// TIA Portal V19 export
FUNCTION_BLOCK "A0301_Manager_FB"   // FB45, LAD
TITLE = == A03 STATION RECIVE PRODUCT ==
// stored: MemoryReserve 100, SetENOAutomatically false
   VAR_INPUT
      AreaInterface : "AreaInterface";
      DataIn : Struct
         SemiAut_Pb : Bool;
         P1 : Struct
            Sens_Ing : Array[1..3] of Bool;
            Sens_Out : Array[1..3] of Bool;
         END_STRUCT;
         P2 : Struct
            Sens_Ing : Array[1..3] of Bool;
            Sens_Out : Array[1..3] of Bool;
         END_STRUCT;
         P3 : Struct
            Sens_Ing : Array[1..3] of Bool;
            Sens_Out : Array[1..3] of Bool;
         END_STRUCT;
         P4 : Struct
            Sens_Ing : Array[1..3] of Bool;
            Sens_Out : Array[1..3] of Bool;
         END_STRUCT;
         P5 : Struct
            Sens_Fuori_Ingombro_A0301 : Bool;
         END_STRUCT;
      END_STRUCT;
      CIn : Struct
         Trasporto : "SpeedMachine_COut";
         P1 : Struct
            Fermi : "ValveMachine_COut";
            Sfalsatore : "ValveMachine_COut";
         END_STRUCT;
         P2 : Struct
            Fermi : "ValveMachine_COut";
            Sollevatore : "ValveMachine_COut";
         END_STRUCT;
         P3 : Struct
            Fermi : "ValveMachine_COut";
         END_STRUCT;
         P4 : Struct
            Fermi : "ValveMachine_COut";
         END_STRUCT;
         P5 : Struct
            Sollevatori { ExternalAccessible := 'False'; ExternalVisible := 'False'; ExternalWritable := 'False'} : "ValveMachine_COut";
            Spintore_Lat : Struct
               Spin_Lat1 : Struct
                  Standstill : Bool;
                  Rest_CheckNext : Bool;
                  Work_CheckNext : Bool;
                  Rest : Bool;
                  Work : Bool;
               END_STRUCT;
               Spin_Lat2 : Struct
                  Standstill : Bool;
                  Rest_CheckNext : Bool;
                  Work_CheckNext : Bool;
                  Rest : Bool;
                  Work : Bool;
               END_STRUCT;
               Vrt_1 : "ValveMachine_COut";
               Orz_1 : "ValveMachine_COut";
               Vrt_2 : "ValveMachine_COut";
               Orz_2 : "ValveMachine_COut";
            END_STRUCT;
            SpintoreLong { ExternalAccessible := 'False'; ExternalVisible := 'False'; ExternalWritable := 'False'} : Struct   // Spintore Longitudinale
               Ax : "Positioning_EPOS_Machine_COut";
               Vert : "ValveMachine_COut";
            END_STRUCT;
            SensUscitaBanco : Bool;
         END_STRUCT;
         Ribaltatore : Struct
            Solleva_Rib : "ValveMachine_COut";
            Ax : "Positioning_EPOS_Machine_COut";
            Sts_Ribaltatore : Struct
               Pos0_Reached : Bool;
               Pos1_Reached : Bool;
               Pos2_Reached : Bool;
               Pos3_Reached : Bool;
            END_STRUCT;
         END_STRUCT;
         SpintoreLong : Struct
            Ax_Sts { ExternalAccessible := 'False'; ExternalVisible := 'False'; ExternalWritable := 'False'} : Struct
               PosAttesa_Reached : Bool;
               PosFineSpinta_Reached : Bool;
            END_STRUCT;
            Spin_Ev : "ValveMachine_COut";
         END_STRUCT;
         ProdManager : "Prod_Beam_Ctrl";
      END_STRUCT;
   END_VAR
   VAR_OUTPUT
      MachineInterface : "MachineInterface";
      COut : Struct
         P1 : Struct
            Fermi : "ValveMachine_Manager";
            Pareggiatore : "ValveMachine_Manager";
            ReqPTrk_A02 : Bool;   // Richiesta pezzo ad Area 02
         END_STRUCT;
         P2 : Struct
            Fermi : "ValveMachine_Manager";
            Sollevatore : "ValveMachine_Manager";
         END_STRUCT;
         P3 : Struct
            Fermi : "ValveMachine_Manager";
         END_STRUCT;
         P4 : Struct
            Fermi : "ValveMachine_Manager";
         END_STRUCT;
         P5 : Struct
            Spintore_Lat_1 { ExternalAccessible := 'False'; ExternalVisible := 'False'; ExternalWritable := 'False'} : "ValveMachine_Manager";
            Spintore_Lat_2 { ExternalAccessible := 'False'; ExternalVisible := 'False'; ExternalWritable := 'False'} : "ValveMachine_Manager";
            Sollevatori : "ValveMachine_Manager";
         END_STRUCT;
         Trasporto : "SpeedMachine_CIn_Manager";
         Trasporto_Brw_Req : Bool;
         Trasporto_Frw_Req : Bool;
         Ribaltatore : Struct
            Solleva : "ValveMachine_Manager";
            Ax : "Positioning_EPOS_Machine_Manager";
            Ax_Req : Struct
               Pos0 : Bool;
               Pos1 : Bool;
               Pos2 : Bool;
               Pos3 : Bool;
            END_STRUCT;
            Solleva_REST_Req : Bool;
            Solleva_WORK_Req : Bool;
         END_STRUCT;
      END_STRUCT;
   END_VAR
   VAR_IN_OUT
      Par : Struct
         DlySensorsON : Time;   // [ms] Ritrado ON sensori prima e dopo fermi
         DlySensorsOFF : Time;   // [ms] Ritrado OFF sensori prima e dopo fermi
         TRK : Struct
            BTrk_MoveP4Exit : Time;
            BTrk_MoveToP5 : Time;
         END_STRUCT;
      END_STRUCT;
      Data : Struct
         LastCounter_PartMove_P2toP4 : LReal;
         LastCounter_PartMove_P1toP2 : LReal;
         LastCounter_PartMove_P1toP3 : LReal;
      END_STRUCT;
   END_VAR
   VAR
      Alarm : Struct
         WrongShiftDone { S7_SetPoint := 'True'} : Bool;
         P2toP4_NotReached : Bool;
         P1toP2_NotReached : Bool;
         P1toP3_NotReached : Bool;
         PTrk_TO_BTrk : Struct
            Status : USInt;
         END_STRUCT;
         STOP_FineTurno : Bool;
         STOP_End_Of_Proroduction : Bool;
         STOP_ControlloQualita : Bool;
      END_STRUCT;
      Sts : Struct
         SemiAut : Struct
            ON : Bool;
            Request : Bool;
            MaterialFrw : Bool;
         END_STRUCT;
         P1 : Struct
            Fermi : Struct
               Sens_Ing : Bool;   // 1= Sensori attivati in base alla selezione attiva in base alla lunghezza del pezzo
               Sens_Out : Bool;   // 1= Sensori attivati in base alla selezione attiva in base alla lunghezza del pezzo
            END_STRUCT;
            Sfalsatura_OK : Bool;
         END_STRUCT;
         P2 : Struct
            Fermi : Struct
               Some_Sens_Ing : Bool;   // 1= Alcuni sensori in ingresso alla stanzione sono attivi, ma non tutti
               Sens_Ing : Bool;   // 1= Sensori attivati in base alla selezione attiva in base alla lunghezza del pezzo
               Sens_Out : Bool;   // 1= Sensori attivati in base alla selezione attiva in base alla lunghezza del pezzo
            END_STRUCT;
         END_STRUCT;
         P3 : Struct
            Fermi : Struct
               Some_Sens_Ing : Bool;   // 1= Alcuni sensori in ingresso alla stanzione sono attivi, ma non tutti
               Sens_Ing : Bool;   // 1= Sensori attivati in base alla selezione attiva in base alla lunghezza del pezzo
               Sens_Out : Bool;   // 1= Sensori attivati in base alla selezione attiva in base alla lunghezza del pezzo
            END_STRUCT;
         END_STRUCT;
         P4 : Struct
            Fermi : Struct
               Some_Sens_Ing : Bool;   // 1= Alcuni sensori in ingresso alla stanzione sono attivi, ma non tutti
               Sens_Ing : Bool;   // 1= Sensori attivati in base alla selezione attiva in base alla lunghezza del pezzo
               Sens_Out : Bool;   // 1= Sensori attivati in base alla selezione attiva in base alla lunghezza del pezzo
            END_STRUCT;
         END_STRUCT;
         A0301_Station1 : Struct
            ZoneEmpty { ExternalAccessible := 'False'; ExternalVisible := 'False'; ExternalWritable := 'False'} : Bool;
            Trk { ExternalAccessible := 'False'; ExternalVisible := 'False'; ExternalWritable := 'False'} : Struct
               Actual_O_ID : DInt;
               OLD_OID : DInt;
               A0301_PTrk_Absence : Bool;
               A0301_BTrk_Absence : Bool;
               Wait_A0301_Recive : Bool;   // Attesa ricevimento nuovo O_ID in ingresso su Pos.1 fino a che la Stazione non è vuota dal OLD_ID
            END_STRUCT;
         END_STRUCT;
         Attrezzamento : Struct
            Ready : Bool;
            FindNewID : Bool;
            RequestNewPosition : Bool;
            OLD_OID : DInt;
         END_STRUCT;
         AlarmsPresence : Bool;
         WarningsPresence : Bool;
         IsStandstill : Bool;
      END_STRUCT;
      Ctrl : Struct
         Stop : Bool;
         TRK : Struct
            PTrk : Struct
               Start_Brw : Bool;
               Start_Frw : Bool;
               Pos1_TO_Pos3 : Bool;
               Pos1_TO_Pos2 : Bool;
               Pos2Entry_TO_Pos2Solleva : Bool;
               Paregg_Pos1_to_Pos2 : Bool;
               Paregg_Pos1_to_Pos3 : Bool;
            END_STRUCT;
            BTrk : Struct
               Pos2Up_TO_Pos2Down : Bool;
               WritePos2Up_TO_Pos2Down : Bool;
               Pos4_Entry_TO_Pos4_Exit : Bool;
               Pos4_Entry_Cndz_To_Exit : Bool;
               Pos4_Exit_TO_Pos4_to_Pos5 : Bool;
               Pos4_to_Pos5_TO_Pos5_Lat_Spin_Orz : Struct
                  Exe : Bool;
                  Solleva : Bool;
                  Trasla : Bool;
               END_STRUCT;
               Pos5_SpinLat_TO_Pos5_SpinLong : Bool;
            END_STRUCT;
            Ribaltatore : Struct
               MoveToPos0 : Bool;
               MoveToPos1 : Bool;
               MoveToPos2 : Bool;
               MoveToPos3 : Bool;
            END_STRUCT;
         END_STRUCT;
         P1 : Struct
            Fermi : Struct
               Rest : Bool;
               Work : Bool;
            END_STRUCT;
            Pareggiatore : Struct
               Rest : Bool;
               Work : Bool;
            END_STRUCT;
            PartMove_P1toP3_Init : Bool;
            PartMove_P1toP2_Init : Bool;
         END_STRUCT;
         P2 : Struct
            Fermi : Struct
               Rest : Bool;
               Work : Bool;
            END_STRUCT;
            Sollevatore : Struct
               EnableMove : Bool;
               Rest : Bool;
               Work : Bool;
            END_STRUCT;
            PartMove_P2toP4_Init : Bool;
         END_STRUCT;
         P3 : Struct
            Fermi : Struct
               Rest : Bool;
               Work : Bool;
            END_STRUCT;
         END_STRUCT;
         P4 : Struct
            Fermi : Struct
               Rest : Bool;
               Work : Bool;
            END_STRUCT;
            Part_Move_P2toP4_Init : Bool;
         END_STRUCT;
         P5 : Struct
            Spintore_Lat_1 : Struct
               Rest : Bool;
               Work : Bool;
            END_STRUCT;
            Spintore_Lat_2 : Struct
               Rest : Bool;
               Work : Bool;
            END_STRUCT;
            Sollevatori : Struct
               Rest : Bool;
               Work : Bool;
            END_STRUCT;
         END_STRUCT;
         Ribaltatore : Struct
            Solleva : Struct
               EnableMove : Bool;
               Rest : Bool;
               Work : Bool;
            END_STRUCT;
         END_STRUCT;
      END_STRUCT;
      Ctrl_Part_Move_P1toP2 : "Check_Part_Movement";
      Ctrl_Part_Move_P1toP3 { S7_SetPoint := 'True'} : "Check_Part_Movement";
      Ctrl_Part_Move_P2toP4 : "Check_Part_Movement";
      TON_Stop { S7_SetPoint := 'True'} : IEC_TIMER;
      TON : Struct
         BTrk_MoveP4Exit : TON_TIME;
         BTrk_MoveToP5 : TON_TIME;
         Delay_Pos1Ribalta { S7_SetPoint := 'True'} : TON_TIME;
         P1 : Struct
            Sens_Ing : Struct
               DelayOn : TON_TIME;
            END_STRUCT;
            Sens_Out : Struct
               DelayOff : TOF_TIME;
            END_STRUCT;
         END_STRUCT;
         P2 : Struct
            Sens_Ing : Struct
               DelayOn : TON_TIME;
            END_STRUCT;
            Sens_Out : Struct
               DelayOff : TOF_TIME;
            END_STRUCT;
         END_STRUCT;
         P3 : Struct
            Sens_Ing : Struct
               DelayOn : TON_TIME;
            END_STRUCT;
            Sens_Out : Struct
               DelayOff : TOF_TIME;
            END_STRUCT;
         END_STRUCT;
         P4 : Struct
            Sens_Ing : Struct
               DelayOn : TON_TIME;
            END_STRUCT;
            Sens_Out : Struct
               DelayOff : TOF_TIME;
            END_STRUCT;
         END_STRUCT;
         P1_Exit_P3 : IEC_TIMER;
         P1_Exit_P2 : IEC_TIMER;
      END_STRUCT;
      HMI : Struct
         B_ResetShiftDone : Bool;
      END_STRUCT;
      AUX : Struct
         SemiAut_Pb : Bool;
         B_ResetShiftDone : Bool;
      END_STRUCT;
      BTrk_Item : Struct   // Appoggio dati che servolo alla Stazione dopo lettura dal MES
         O_ID : DInt;
         BLean : Real;
         W_A : Real;
         H_B : Real;
         Tol_Max : Real;
         Tol_Min : Real;
         Good { ExternalAccessible := 'False'; ExternalVisible := 'False'; ExternalWritable := 'False'} : Bool;
         Bad { ExternalAccessible := 'False'; ExternalVisible := 'False'; ExternalWritable := 'False'} : Bool;
      END_STRUCT;
      PLen_Pos1 : Real;
      PLen_Pos3 : Real;
   END_VAR
   VAR_TEMP
      i : Int;   // Indice BTrk
      j : Int;   // Indice PTrk
      SensorToUse : Struct
         P1_In : Array[1..3] of Bool;
         P1_Out : Array[1..3] of Bool;   // Sensori presenza
         P2_In : Array[1..3] of Bool;
         P2_Out : Array[1..3] of Bool;   // Fotocellule
         P3_In : Array[1..3] of Bool;
         P3_Out : Array[1..3] of Bool;   // Fotocellule
         P4_In : Array[1..3] of Bool;
         P4_Out : Array[1..3] of Bool;   // Fotocellule
      END_STRUCT;
      P1 : Struct
         Cndz1_P1toP3 : Bool;
         Cndz2_P1toP3 : Bool;
      END_STRUCT;
      Trk_GetData : Struct   // Struttura dati per lettura dal MES di tutti i dati
         indx : Int;   // Se trovato tra i TODO / ENDING / OUT questo è l'indice dove sono stati prelevati i dati
         Sts : Int;   // 0 = Non Trovato; 0 = ACT; 1 = TODO; 2=ENDING; 3 = OUT
         Item : "Prod_Item_small";
      END_STRUCT;
      Sens : Struct
         P1_IngOn : Bool;
         P1_OutOn : Bool;
         P2_IngOn : Bool;
         P3_IngOn : Bool;
         P3_OutOn : Bool;
         P4_IngOn : Bool;
         P4_OutOn : Bool;
      END_STRUCT;
   END_VAR
   VAR_TEMP   // added for the SCL form of the ladder/FBD networks
      _w1 : Bool;
      _w2 : Bool;
      _w3 : Bool;
      _w4 : Bool;
      _w5 : Bool;
      _w6 : Bool;
      _w7 : Bool;
      _w8 : Bool;
      _w9 : Bool;
      _w10 : Bool;
      _w11 : Bool;
      _w12 : Bool;
      _w13 : Bool;
      _w14 : Bool;
      _w15 : Bool;
      _w16 : Bool;
      _w17 : Bool;
      _w18 : Bool;
      _w19 : Bool;
      _w20 : Bool;
      _w21 : Bool;
      _w22 : Bool;
      _w23 : Bool;
      _w24 : Bool;
      _w25 : Bool;
   END_VAR
BEGIN

REGION Network 1: °°°°°° FORZATURA PTrk °°°°°°°°°
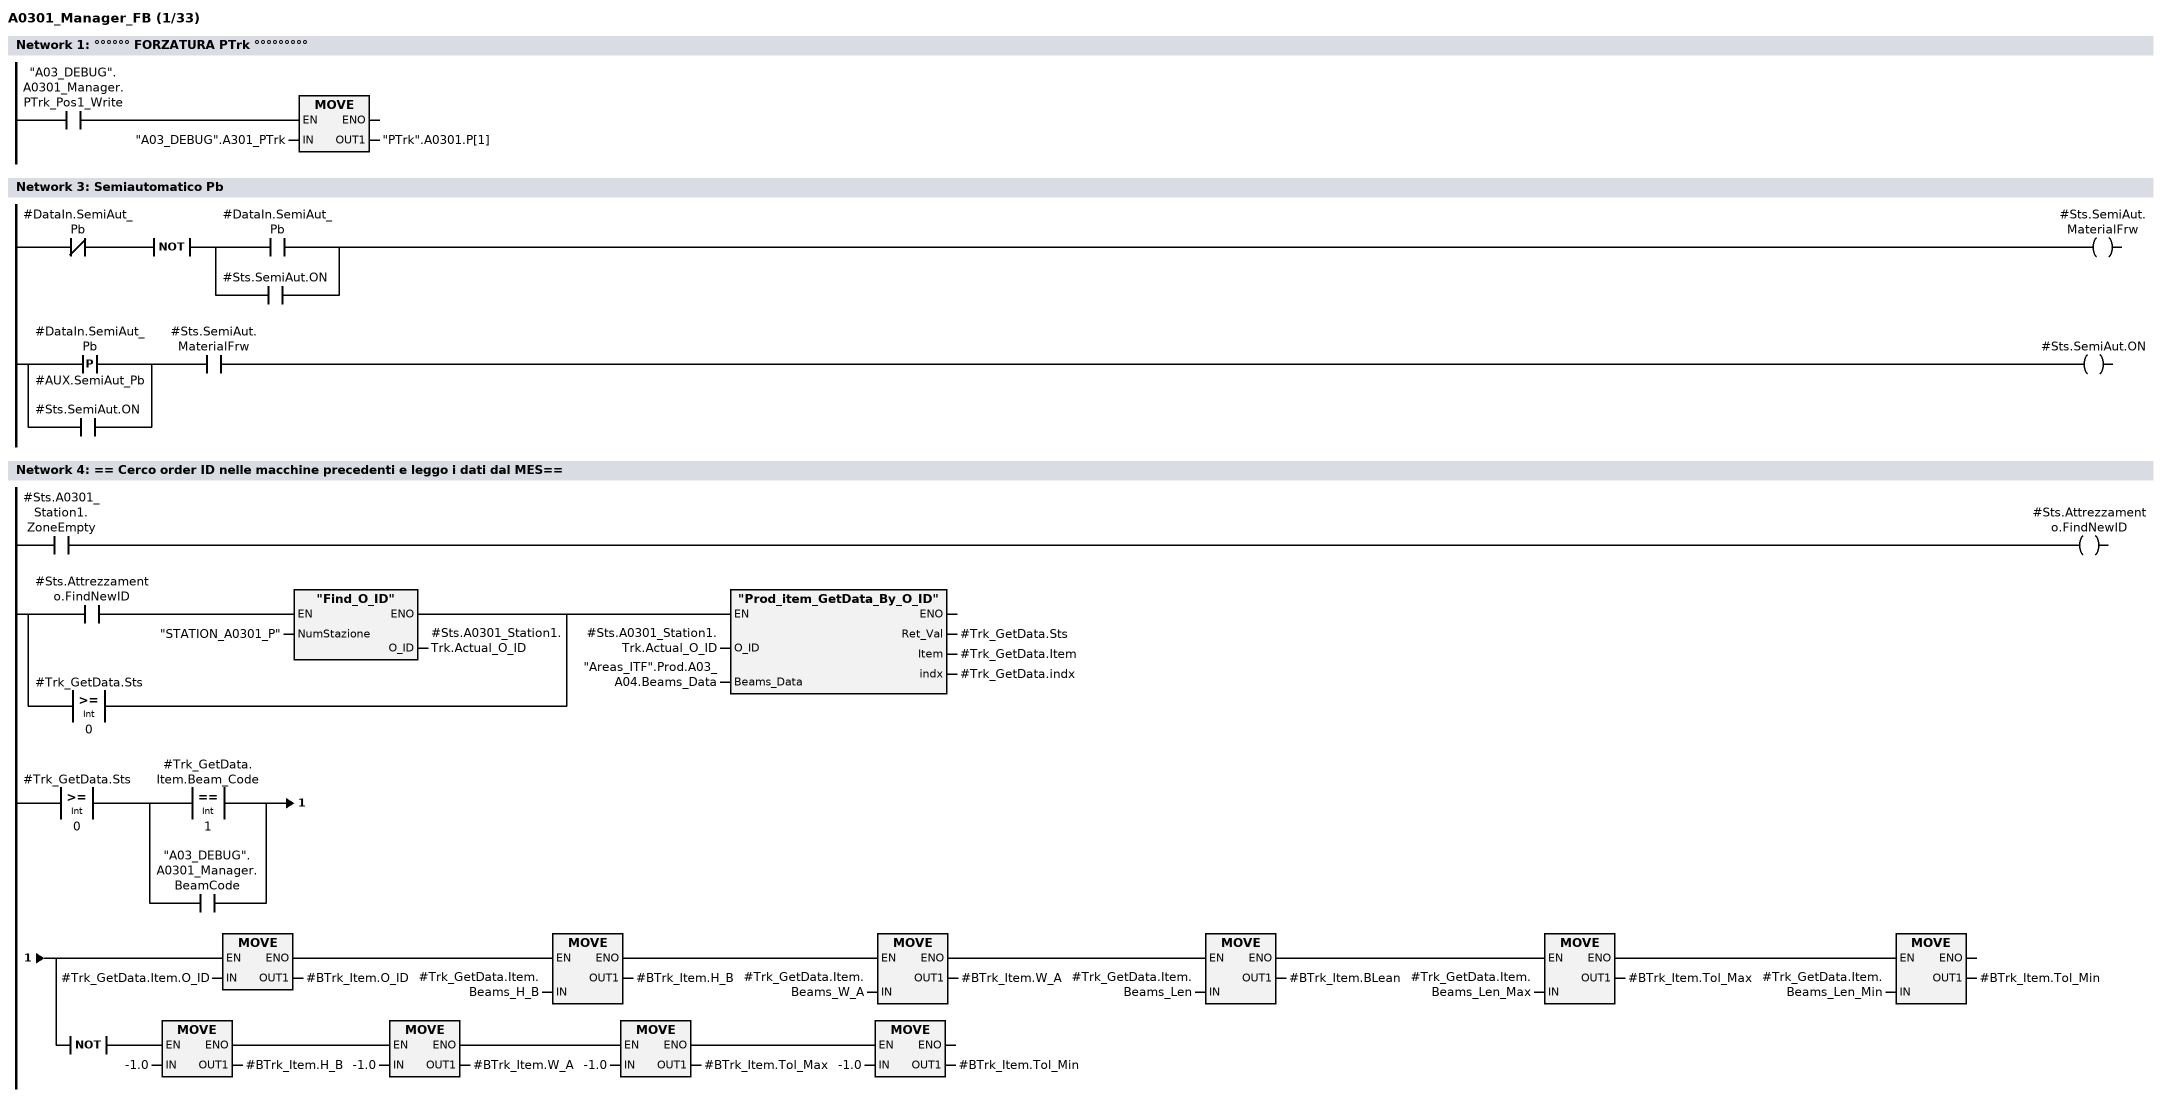
   RUNG wire#powerrail
      Contact( "A03_DEBUG".A0301_Manager.PTrk_Pos1_Write )
      Move(in := "A03_DEBUG".A301_PTrk, out1 => "PTrk".A0301.P[1])
   END_RUNG
   // the same network as SCL:
   IF "A03_DEBUG".A0301_Manager.PTrk_Pos1_Write THEN "PTrk".A0301.P[1] := "A03_DEBUG".A301_PTrk; END_IF;
END_REGION

REGION Network 2 (SCL): = Area - Rst =
   IF #AreaInterface.RstAlarms THEN
       #Alarm.WrongShiftDone := FALSE;
       #Alarm.P2toP4_NotReached:= FALSE;
       #Alarm.P1toP2_NotReached:=FALSE;
       #Alarm.P1toP3_NotReached := FALSE;
       //
       #Alarm.STOP_ControlloQualita := FALSE;
       #Alarm.STOP_FineTurno := FALSE;
       #Alarm.STOP_End_Of_Proroduction := FALSE;
   END_IF;
END_REGION

REGION Network 3: Semiautomatico Pb
   RUNG wire#powerrail
      I_Contact( #DataIn.SemiAut_Pb )
      Not()
      wire#w1
      Contact( #DataIn.SemiAut_Pb )
      wire#w2
      Coil( #Sts.SemiAut.MaterialFrw )
   END_RUNG
   RUNG wire#w1
      Contact( #Sts.SemiAut.ON )
   END_RUNG wire#w2
   RUNG wire#powerrail
      P_Contact(operand := #DataIn.SemiAut_Pb, bit := #AUX.SemiAut_Pb)
      wire#w3
      Contact( #Sts.SemiAut.MaterialFrw )
      Coil( #Sts.SemiAut.ON )
   END_RUNG
   RUNG wire#powerrail
      Contact( #Sts.SemiAut.ON )
   END_RUNG wire#w3
   // the same network as SCL:
   #Sts.SemiAut.MaterialFrw := NOT (NOT #DataIn.SemiAut_Pb) AND (#DataIn.SemiAut_Pb OR #Sts.SemiAut.ON);
   #_w1 := #DataIn.SemiAut_Pb AND NOT #AUX.SemiAut_Pb;   // rising edge of #DataIn.SemiAut_Pb
   #AUX.SemiAut_Pb := #DataIn.SemiAut_Pb;
   #Sts.SemiAut.ON := (#_w1 OR #Sts.SemiAut.ON) AND #Sts.SemiAut.MaterialFrw;
END_REGION

REGION Network 4: == Cerco order ID nelle macchine precedenti e leggo i dati dal MES==
   RUNG wire#powerrail
      Contact( #Sts.A0301_Station1.ZoneEmpty )
      Coil( #Sts.Attrezzamento.FindNewID )
   END_RUNG
   RUNG wire#powerrail
      Contact( #Sts.Attrezzamento.FindNewID )
      "Find_O_ID"(NumStazione := "STATION_A0301_P", O_ID => #Sts.A0301_Station1.Trk.Actual_O_ID)
      wire#w1
      "Prod_item_GetData_By_O_ID"(O_ID := #Sts.A0301_Station1.Trk.Actual_O_ID, Beams_Data := "Areas_ITF".Prod.A03_A04.Beams_Data, Ret_Val => #Trk_GetData.Sts, Item => #Trk_GetData.Item, indx => #Trk_GetData.indx)
   END_RUNG
   RUNG wire#powerrail
      { S7_Templates := "SrcType := Int" } GE_Contact(in1 := #Trk_GetData.Sts, in2 := 0)
   END_RUNG wire#w1
   RUNG wire#powerrail
      { S7_Templates := "SrcType := Int" } GE_Contact(in1 := #Trk_GetData.Sts, in2 := 0)
      wire#w2
      { S7_Templates := "SrcType := Int" } EQ_Contact(in1 := #Trk_GetData.Item.Beam_Code, in2 := 1)
      wire#w3
      Move(in := #Trk_GetData.Item.O_ID, out1 => #BTrk_Item.O_ID)
      Move(in := #Trk_GetData.Item.Beams_H_B, out1 => #BTrk_Item.H_B)
      Move(in := #Trk_GetData.Item.Beams_W_A, out1 => #BTrk_Item.W_A)
      Move(in := #Trk_GetData.Item.Beams_Len, out1 => #BTrk_Item.BLean)
      Move(in := #Trk_GetData.Item.Beams_Len_Max, out1 => #BTrk_Item.Tol_Max)
      Move(in := #Trk_GetData.Item.Beams_Len_Min, out1 => #BTrk_Item.Tol_Min)
   END_RUNG
   RUNG wire#w2
      Contact( "A03_DEBUG".A0301_Manager.BeamCode )
   END_RUNG wire#w3
   RUNG wire#w3
      Not()
      Move(in := -1.0, out1 => #BTrk_Item.H_B)
      Move(in := -1.0, out1 => #BTrk_Item.W_A)
      Move(in := -1.0, out1 => #BTrk_Item.Tol_Max)
      Move(in := -1.0, out1 => #BTrk_Item.Tol_Min)
   END_RUNG
   // the same network as SCL:
   #Sts.Attrezzamento.FindNewID := #Sts.A0301_Station1.ZoneEmpty;
   "Find_O_ID"(EN := #Sts.Attrezzamento.FindNewID,
               NumStazione := "STATION_A0301_P",
               O_ID => #Sts.A0301_Station1.Trk.Actual_O_ID,
               ENO => #_w1);
   IF #_w1 OR (#Trk_GetData.Sts >= 0) THEN
       #Trk_GetData.Sts := "Prod_item_GetData_By_O_ID"(O_ID := #Sts.A0301_Station1.Trk.Actual_O_ID,
                               Beams_Data := "Areas_ITF".Prod.A03_A04.Beams_Data,
                               Item => #Trk_GetData.Item,
                               indx => #Trk_GetData.indx);
   END_IF;
   #_w2 := (#Trk_GetData.Sts >= 0) AND ((#Trk_GetData.Item.Beam_Code = 1) OR "A03_DEBUG".A0301_Manager.BeamCode);
   IF #_w2 THEN
       #BTrk_Item.O_ID := #Trk_GetData.Item.O_ID;
       #BTrk_Item.H_B := #Trk_GetData.Item.Beams_H_B;
       #BTrk_Item.W_A := #Trk_GetData.Item.Beams_W_A;
       #BTrk_Item.BLean := #Trk_GetData.Item.Beams_Len;
       #BTrk_Item.Tol_Max := #Trk_GetData.Item.Beams_Len_Max;
       #BTrk_Item.Tol_Min := #Trk_GetData.Item.Beams_Len_Min;
   END_IF;
   IF NOT #_w2 THEN
       #BTrk_Item.H_B := -1.0;
       #BTrk_Item.W_A := -1.0;
       #BTrk_Item.Tol_Max := -1.0;
       #BTrk_Item.Tol_Min := -1.0;
   END_IF;
END_REGION

REGION Network 5 (SCL): == CONTROLLO TRACKING E STAZIONE PER AVANZAMENTO O_ID ==
   REGION CONTROLLO (TRK EMPTY) SU STAZIONE 1 RIBALTAMENTO A0301 
       // Controllo zona libera dai traking e sensori non in lettura su stazione A0301
       // 
       FOR #i := 1 TO "BTRK_A0301_ITEMS" DO
           IF "BTrk".A0301.B[#i].B_ID = 0 THEN
               #Sts.A0301_Station1.Trk.A0301_BTrk_Absence := TRUE;
           ELSE
               #Sts.A0301_Station1.Trk.A0301_BTrk_Absence := FALSE;
               EXIT;
           END_IF;
       END_FOR;
       //
       FOR #j := 2 TO "PTRK_A0301_ITEMS" DO
           IF "PTrk".A0301.P[#j].P_ID = 0 THEN
               #Sts.A0301_Station1.Trk.A0301_PTrk_Absence := TRUE;
           ELSE
               #Sts.A0301_Station1.Trk.A0301_PTrk_Absence := FALSE;
               EXIT;
           END_IF;
       END_FOR;

   END_REGION

   REGION CONTROLLO CHE CI SIANO LE CONDIZIONI PER MANDARE AVANTI IL NUOVO ID SU STAZIONE 1 RIBALTAMENTO A0301 (TRK EMPTY)

       // Verifica A0301 VUOTA se PTrk o BTrk assente e sensori su Stazione 1 non in lettura
       #Sts.A0301_Station1.ZoneEmpty := #Sts.A0301_Station1.Trk.A0301_PTrk_Absence AND #Sts.A0301_Station1.Trk.A0301_BTrk_Absence AND
       (NOT #Sts.P1.Fermi.Sens_Out AND
       NOT #Sts.P2.Fermi.Sens_Ing AND NOT #Sts.P1.Fermi.Sens_Out AND
       NOT #Sts.P3.Fermi.Sens_Ing AND NOT #Sts.P3.Fermi.Sens_Out AND
       NOT #Sts.P4.Fermi.Sens_Ing AND NOT #Sts.P4.Fermi.Sens_Out);


       //Se ho O_ID <> e non sono vuoto attivo avviso di attesa zona A0302 vuota
       IF (#Sts.A0301_Station1.Trk.Actual_O_ID <> #Sts.A0301_Station1.Trk.OLD_OID) OR NOT #Sts.A0301_Station1.ZoneEmpty THEN
           #Sts.A0301_Station1.Trk.Wait_A0301_Recive := TRUE;
       ELSIF (#Sts.A0301_Station1.Trk.Actual_O_ID = #Sts.A0301_Station1.Trk.OLD_OID) OR #Sts.A0301_Station1.ZoneEmpty THEN
           #Sts.A0301_Station1.Trk.Wait_A0301_Recive := FALSE;
       END_IF;

       //Se ho O_ID <> e sono vuoto aggiorno vecchio O_ID 
       IF (#Sts.A0301_Station1.Trk.Actual_O_ID <> #Sts.A0301_Station1.Trk.OLD_OID) AND #Sts.A0301_Station1.ZoneEmpty THEN
           #Sts.A0301_Station1.Trk.OLD_OID := #Sts.A0301_Station1.Trk.Actual_O_ID;
       END_IF;

   END_REGION
END_REGION

REGION Network 6 (SCL): == Compilo i dati del BTrk in base all'order ID in arrivo ==

   IF #Trk_GetData.Sts >= 0 THEN

       "BTrk".A0301.O_ID :=   #Sts.A0301_Station1.Trk.OLD_OID;
       "BTrk".A0301.Beam_Len := #BTrk_Item.BLean;
       "BTrk".A0301.Beam_W_A := #BTrk_Item.W_A;
       "BTrk".A0301.Beam_H_B := #BTrk_Item.H_B;

   ELSE
            "BTrk".A0301.O_ID := -1;
            "BTrk".A0301.Beam_Len := -1.0;
            "BTrk".A0301.Beam_W_A := -1.0;
            "BTrk".A0301.Beam_H_B := -1.0;
   END_IF;
END_REGION

REGION Network 8: <<< GESTIONE DEI SENSORI SULLE STAZIONI IN BASE ALLA LUNGHEZZA DEL PEZZO >>>
END_REGION

REGION Network 9: [P1] = Enable/Disable Sensors Pin & Controllo e Stato dei sensori ==
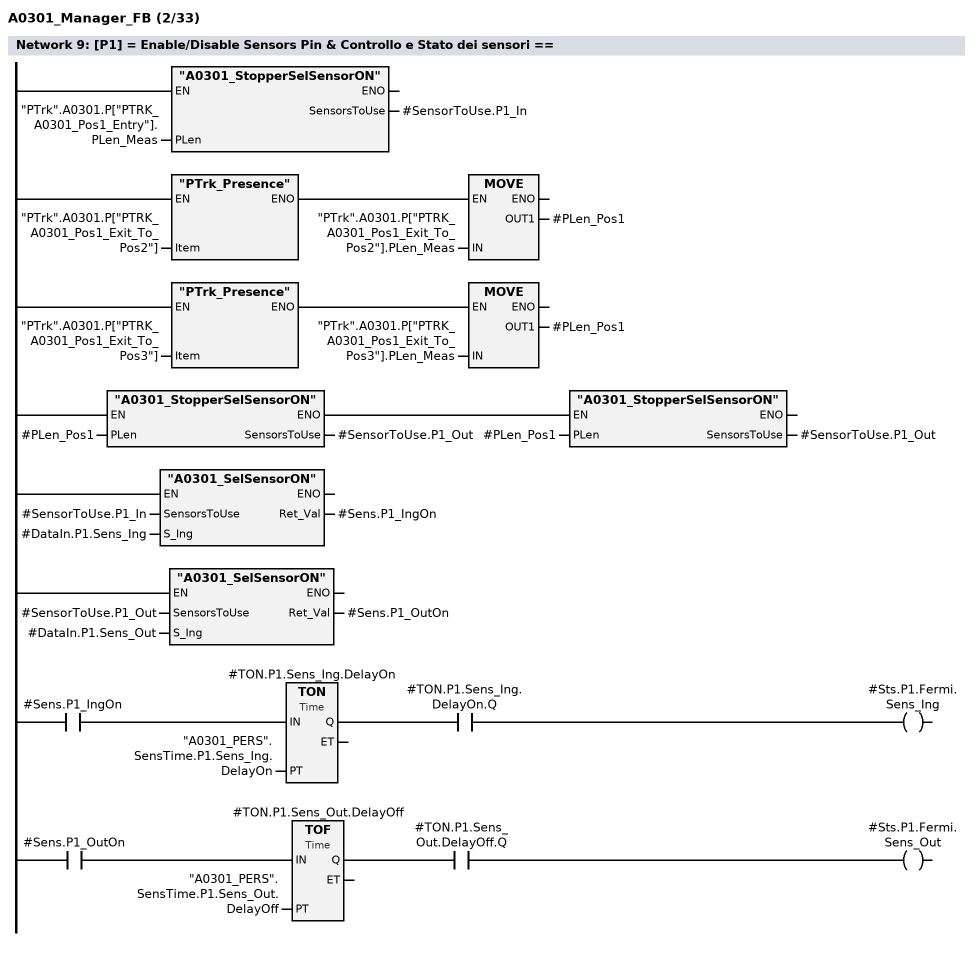
   RUNG wire#powerrail
      "A0301_StopperSelSensorON"(PLen := "PTrk".A0301.P["PTRK_A0301_Pos1_Entry"].PLen_Meas, SensorsToUse => #SensorToUse.P1_In)
   END_RUNG
   RUNG wire#powerrail
      "PTrk_Presence"(Item := "PTrk".A0301.P["PTRK_A0301_Pos1_Exit_To_Pos2"])
      Move(in := "PTrk".A0301.P["PTRK_A0301_Pos1_Exit_To_Pos2"].PLen_Meas, out1 => #PLen_Pos1)
   END_RUNG
   RUNG wire#powerrail
      "PTrk_Presence"(Item := "PTrk".A0301.P["PTRK_A0301_Pos1_Exit_To_Pos3"])
      Move(in := "PTrk".A0301.P["PTRK_A0301_Pos1_Exit_To_Pos3"].PLen_Meas, out1 => #PLen_Pos1)
   END_RUNG
   RUNG wire#powerrail
      "A0301_StopperSelSensorON"(PLen := #PLen_Pos1, SensorsToUse => #SensorToUse.P1_Out)
      "A0301_StopperSelSensorON"(PLen := #PLen_Pos1, SensorsToUse => #SensorToUse.P1_Out)
   END_RUNG
   RUNG wire#powerrail
      "A0301_SelSensorON"(SensorsToUse := #SensorToUse.P1_In, S_Ing := #DataIn.P1.Sens_Ing, Ret_Val => #Sens.P1_IngOn)
   END_RUNG
   RUNG wire#powerrail
      "A0301_SelSensorON"(SensorsToUse := #SensorToUse.P1_Out, S_Ing := #DataIn.P1.Sens_Out, Ret_Val => #Sens.P1_OutOn)
   END_RUNG
   RUNG wire#powerrail
      Contact( #Sens.P1_IngOn )
      { S7_Templates := "time_type := Time" } #TON.P1.Sens_Ing.DelayOn.TON(pt := "A0301_PERS".SensTime.P1.Sens_Ing.DelayOn, et =>)
      Contact( #TON.P1.Sens_Ing.DelayOn.Q )
      Coil( #Sts.P1.Fermi.Sens_Ing )
   END_RUNG
   RUNG wire#powerrail
      Contact( #Sens.P1_OutOn )
      { S7_Templates := "time_type := Time" } #TON.P1.Sens_Out.DelayOff.TOF(pt := "A0301_PERS".SensTime.P1.Sens_Out.DelayOff, et =>)
      Contact( #TON.P1.Sens_Out.DelayOff.Q )
      Coil( #Sts.P1.Fermi.Sens_Out )
   END_RUNG
   // the same network as SCL:
   "A0301_StopperSelSensorON"(PLen := "PTrk".A0301.P["PTRK_A0301_Pos1_Entry"].PLen_Meas,
                           SensorsToUse => #SensorToUse.P1_In);
   "PTrk_Presence"(Item := "PTrk".A0301.P["PTRK_A0301_Pos1_Exit_To_Pos2"], ENO => #_w1);
   IF #_w1 THEN #PLen_Pos1 := "PTrk".A0301.P["PTRK_A0301_Pos1_Exit_To_Pos2"].PLen_Meas; END_IF;
   "PTrk_Presence"(Item := "PTrk".A0301.P["PTRK_A0301_Pos1_Exit_To_Pos3"], ENO => #_w2);
   IF #_w2 THEN #PLen_Pos1 := "PTrk".A0301.P["PTRK_A0301_Pos1_Exit_To_Pos3"].PLen_Meas; END_IF;
   "A0301_StopperSelSensorON"(PLen := #PLen_Pos1, SensorsToUse => #SensorToUse.P1_Out, ENO => #_w3);
   IF #_w3 THEN "A0301_StopperSelSensorON"(PLen := #PLen_Pos1, SensorsToUse => #SensorToUse.P1_Out); END_IF;
   #Sens.P1_IngOn := "A0301_SelSensorON"(SensorsToUse := #SensorToUse.P1_In, S_Ing := #DataIn.P1.Sens_Ing);
   #Sens.P1_OutOn := "A0301_SelSensorON"(SensorsToUse := #SensorToUse.P1_Out, S_Ing := #DataIn.P1.Sens_Out);
   #TON.P1.Sens_Ing.DelayOn.TON(IN := #Sens.P1_IngOn, PT := "A0301_PERS".SensTime.P1.Sens_Ing.DelayOn);
   #Sts.P1.Fermi.Sens_Ing := #TON.P1.Sens_Ing.DelayOn.Q AND #TON.P1.Sens_Ing.DelayOn.Q;
   #TON.P1.Sens_Out.DelayOff.TOF(IN := #Sens.P1_OutOn, PT := "A0301_PERS".SensTime.P1.Sens_Out.DelayOff);
   #Sts.P1.Fermi.Sens_Out := #TON.P1.Sens_Out.DelayOff.Q AND #TON.P1.Sens_Out.DelayOff.Q;
END_REGION

REGION Network 10: [P2] = Enable/Disable Sensors Pin & Controllo e Stato dei sensori ==
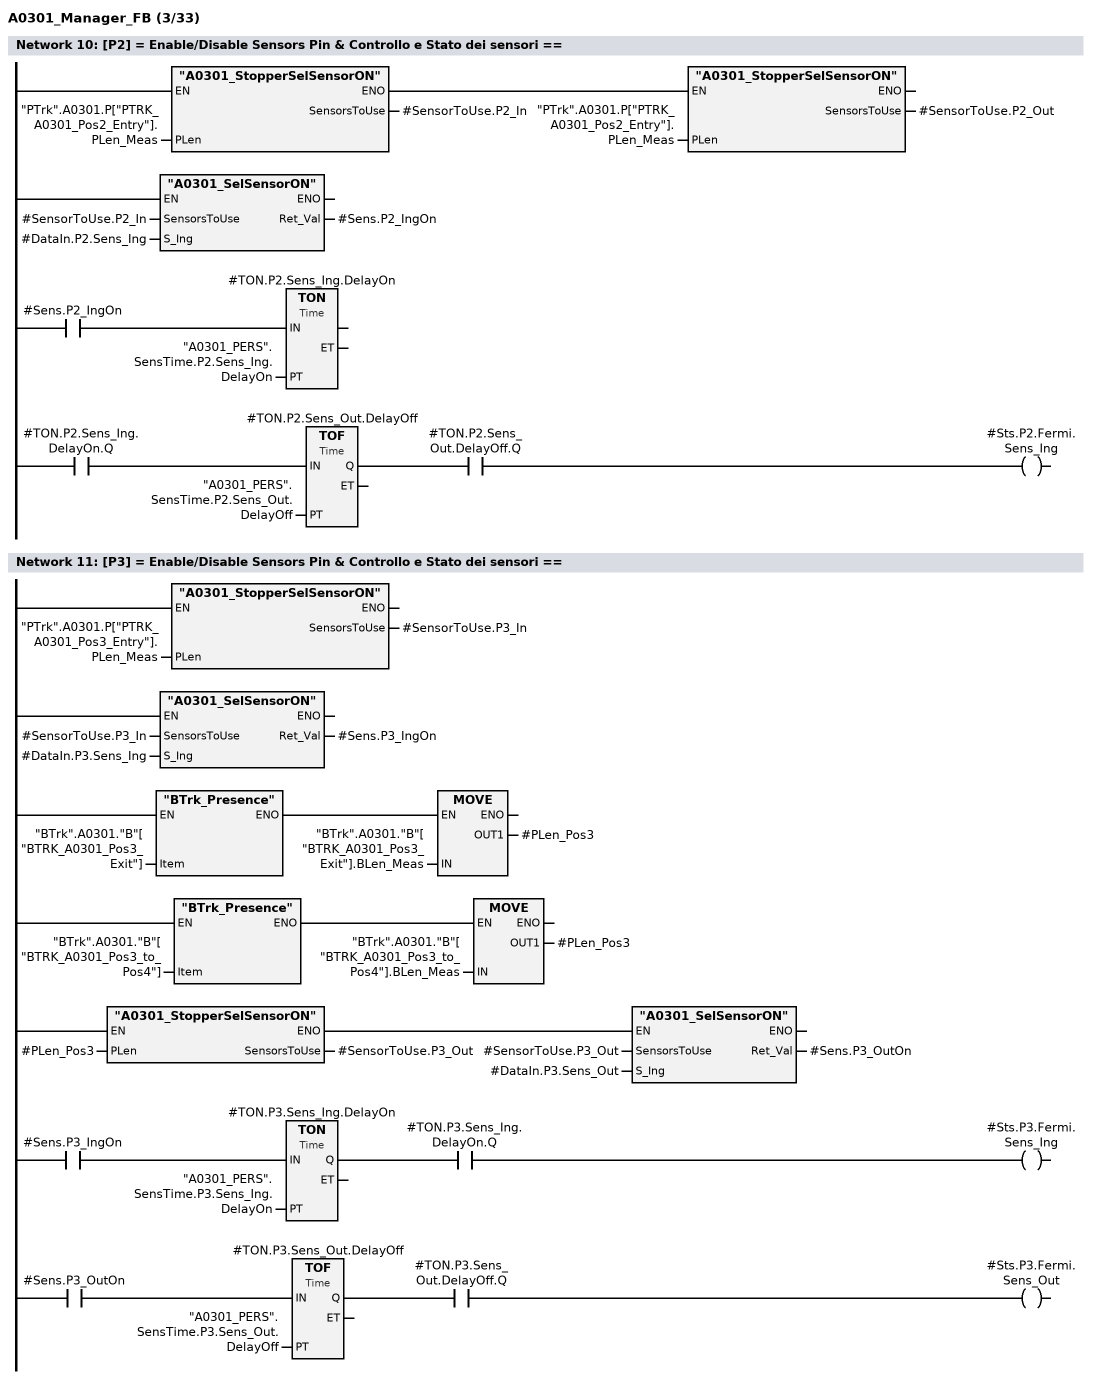
   RUNG wire#powerrail
      "A0301_StopperSelSensorON"(PLen := "PTrk".A0301.P["PTRK_A0301_Pos2_Entry"].PLen_Meas, SensorsToUse => #SensorToUse.P2_In)
      "A0301_StopperSelSensorON"(PLen := "PTrk".A0301.P["PTRK_A0301_Pos2_Entry"].PLen_Meas, SensorsToUse => #SensorToUse.P2_Out)
   END_RUNG
   RUNG wire#powerrail
      "A0301_SelSensorON"(SensorsToUse := #SensorToUse.P2_In, S_Ing := #DataIn.P2.Sens_Ing, Ret_Val => #Sens.P2_IngOn)
   END_RUNG
   RUNG wire#powerrail
      Contact( #Sens.P2_IngOn )
      { S7_Templates := "time_type := Time" } #TON.P2.Sens_Ing.DelayOn.TON(pt := "A0301_PERS".SensTime.P2.Sens_Ing.DelayOn, et =>)
   END_RUNG
   RUNG wire#powerrail
      Contact( #TON.P2.Sens_Ing.DelayOn.Q )
      { S7_Templates := "time_type := Time" } #TON.P2.Sens_Out.DelayOff.TOF(pt := "A0301_PERS".SensTime.P2.Sens_Out.DelayOff, et =>)
      Contact( #TON.P2.Sens_Out.DelayOff.Q )
      Coil( #Sts.P2.Fermi.Sens_Ing )
   END_RUNG
   // the same network as SCL:
   "A0301_StopperSelSensorON"(PLen := "PTrk".A0301.P["PTRK_A0301_Pos2_Entry"].PLen_Meas,
                           SensorsToUse => #SensorToUse.P2_In,
                           ENO => #_w1);
   IF #_w1 THEN
       "A0301_StopperSelSensorON"(PLen := "PTrk".A0301.P["PTRK_A0301_Pos2_Entry"].PLen_Meas,
                               SensorsToUse => #SensorToUse.P2_Out);
   END_IF;
   #Sens.P2_IngOn := "A0301_SelSensorON"(SensorsToUse := #SensorToUse.P2_In, S_Ing := #DataIn.P2.Sens_Ing);
   #TON.P2.Sens_Ing.DelayOn.TON(IN := #Sens.P2_IngOn, PT := "A0301_PERS".SensTime.P2.Sens_Ing.DelayOn);
   #TON.P2.Sens_Out.DelayOff.TOF(IN := #TON.P2.Sens_Ing.DelayOn.Q,
                           PT := "A0301_PERS".SensTime.P2.Sens_Out.DelayOff);
   #Sts.P2.Fermi.Sens_Ing := #TON.P2.Sens_Out.DelayOff.Q AND #TON.P2.Sens_Out.DelayOff.Q;
END_REGION

REGION Network 11: [P3] = Enable/Disable Sensors Pin & Controllo e Stato dei sensori ==
   RUNG wire#powerrail
      "A0301_StopperSelSensorON"(PLen := "PTrk".A0301.P["PTRK_A0301_Pos3_Entry"].PLen_Meas, SensorsToUse => #SensorToUse.P3_In)
   END_RUNG
   RUNG wire#powerrail
      "A0301_SelSensorON"(SensorsToUse := #SensorToUse.P3_In, S_Ing := #DataIn.P3.Sens_Ing, Ret_Val => #Sens.P3_IngOn)
   END_RUNG
   RUNG wire#powerrail
      "BTrk_Presence"(Item := "BTrk".A0301."B"["BTRK_A0301_Pos3_Exit"])
      Move(in := "BTrk".A0301."B"["BTRK_A0301_Pos3_Exit"].BLen_Meas, out1 => #PLen_Pos3)
   END_RUNG
   RUNG wire#powerrail
      "BTrk_Presence"(Item := "BTrk".A0301."B"["BTRK_A0301_Pos3_to_Pos4"])
      Move(in := "BTrk".A0301."B"["BTRK_A0301_Pos3_to_Pos4"].BLen_Meas, out1 => #PLen_Pos3)
   END_RUNG
   RUNG wire#powerrail
      "A0301_StopperSelSensorON"(PLen := #PLen_Pos3, SensorsToUse => #SensorToUse.P3_Out)
      "A0301_SelSensorON"(SensorsToUse := #SensorToUse.P3_Out, S_Ing := #DataIn.P3.Sens_Out, Ret_Val => #Sens.P3_OutOn)
   END_RUNG
   RUNG wire#powerrail
      Contact( #Sens.P3_IngOn )
      { S7_Templates := "time_type := Time" } #TON.P3.Sens_Ing.DelayOn.TON(pt := "A0301_PERS".SensTime.P3.Sens_Ing.DelayOn, et =>)
      Contact( #TON.P3.Sens_Ing.DelayOn.Q )
      Coil( #Sts.P3.Fermi.Sens_Ing )
   END_RUNG
   RUNG wire#powerrail
      Contact( #Sens.P3_OutOn )
      { S7_Templates := "time_type := Time" } #TON.P3.Sens_Out.DelayOff.TOF(pt := "A0301_PERS".SensTime.P3.Sens_Out.DelayOff, et =>)
      Contact( #TON.P3.Sens_Out.DelayOff.Q )
      Coil( #Sts.P3.Fermi.Sens_Out )
   END_RUNG
   // the same network as SCL:
   "A0301_StopperSelSensorON"(PLen := "PTrk".A0301.P["PTRK_A0301_Pos3_Entry"].PLen_Meas,
                           SensorsToUse => #SensorToUse.P3_In);
   #Sens.P3_IngOn := "A0301_SelSensorON"(SensorsToUse := #SensorToUse.P3_In, S_Ing := #DataIn.P3.Sens_Ing);
   "BTrk_Presence"(Item := "BTrk".A0301."B"["BTRK_A0301_Pos3_Exit"], ENO => #_w1);
   IF #_w1 THEN #PLen_Pos3 := "BTrk".A0301."B"["BTRK_A0301_Pos3_Exit"].BLen_Meas; END_IF;
   "BTrk_Presence"(Item := "BTrk".A0301."B"["BTRK_A0301_Pos3_to_Pos4"], ENO => #_w2);
   IF #_w2 THEN #PLen_Pos3 := "BTrk".A0301."B"["BTRK_A0301_Pos3_to_Pos4"].BLen_Meas; END_IF;
   "A0301_StopperSelSensorON"(PLen := #PLen_Pos3, SensorsToUse => #SensorToUse.P3_Out, ENO => #_w3);
   IF #_w3 THEN
       #Sens.P3_OutOn := "A0301_SelSensorON"(SensorsToUse := #SensorToUse.P3_Out, S_Ing := #DataIn.P3.Sens_Out);
   END_IF;
   #TON.P3.Sens_Ing.DelayOn.TON(IN := #Sens.P3_IngOn, PT := "A0301_PERS".SensTime.P3.Sens_Ing.DelayOn);
   #Sts.P3.Fermi.Sens_Ing := #TON.P3.Sens_Ing.DelayOn.Q AND #TON.P3.Sens_Ing.DelayOn.Q;
   #TON.P3.Sens_Out.DelayOff.TOF(IN := #Sens.P3_OutOn, PT := "A0301_PERS".SensTime.P3.Sens_Out.DelayOff);
   #Sts.P3.Fermi.Sens_Out := #TON.P3.Sens_Out.DelayOff.Q AND #TON.P3.Sens_Out.DelayOff.Q;
END_REGION

REGION Network 12: [P4] = Enable/Disable Sensors Pin & Controllo e Stato dei sensori ==
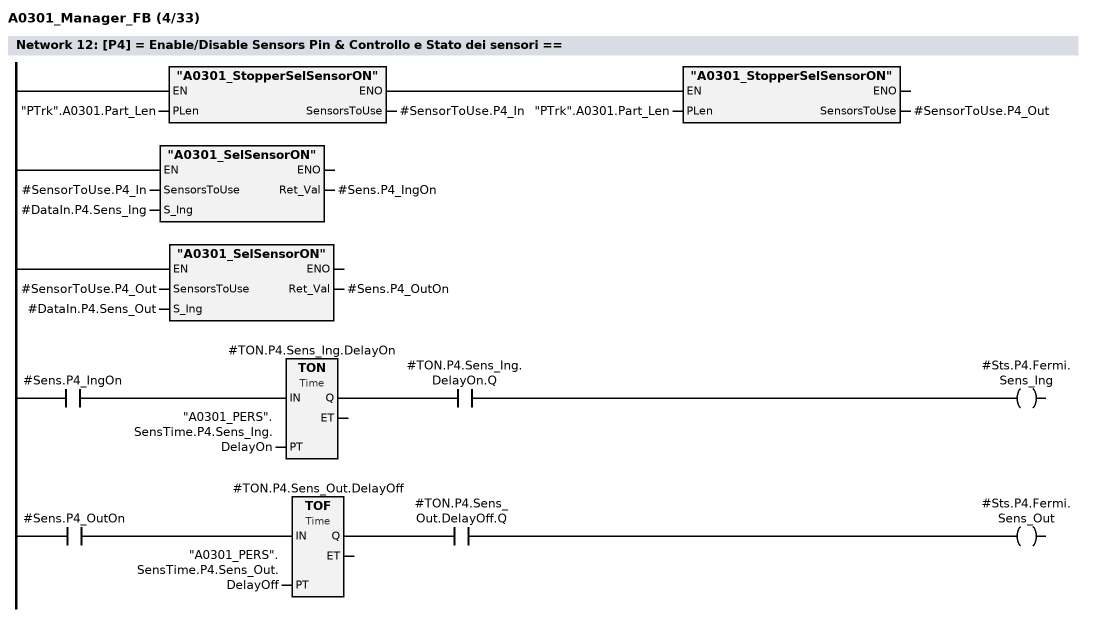
   RUNG wire#powerrail
      "A0301_StopperSelSensorON"(PLen := "PTrk".A0301.Part_Len, SensorsToUse => #SensorToUse.P4_In)
      "A0301_StopperSelSensorON"(PLen := "PTrk".A0301.Part_Len, SensorsToUse => #SensorToUse.P4_Out)
   END_RUNG
   RUNG wire#powerrail
      "A0301_SelSensorON"(SensorsToUse := #SensorToUse.P4_In, S_Ing := #DataIn.P4.Sens_Ing, Ret_Val => #Sens.P4_IngOn)
   END_RUNG
   RUNG wire#powerrail
      "A0301_SelSensorON"(SensorsToUse := #SensorToUse.P4_Out, S_Ing := #DataIn.P4.Sens_Out, Ret_Val => #Sens.P4_OutOn)
   END_RUNG
   RUNG wire#powerrail
      Contact( #Sens.P4_IngOn )
      { S7_Templates := "time_type := Time" } #TON.P4.Sens_Ing.DelayOn.TON(pt := "A0301_PERS".SensTime.P4.Sens_Ing.DelayOn, et =>)
      Contact( #TON.P4.Sens_Ing.DelayOn.Q )
      Coil( #Sts.P4.Fermi.Sens_Ing )
   END_RUNG
   RUNG wire#powerrail
      Contact( #Sens.P4_OutOn )
      { S7_Templates := "time_type := Time" } #TON.P4.Sens_Out.DelayOff.TOF(pt := "A0301_PERS".SensTime.P4.Sens_Out.DelayOff, et =>)
      Contact( #TON.P4.Sens_Out.DelayOff.Q )
      Coil( #Sts.P4.Fermi.Sens_Out )
   END_RUNG
   // the same network as SCL:
   "A0301_StopperSelSensorON"(PLen := "PTrk".A0301.Part_Len, SensorsToUse => #SensorToUse.P4_In, ENO => #_w1);
   IF #_w1 THEN
       "A0301_StopperSelSensorON"(PLen := "PTrk".A0301.Part_Len, SensorsToUse => #SensorToUse.P4_Out);
   END_IF;
   #Sens.P4_IngOn := "A0301_SelSensorON"(SensorsToUse := #SensorToUse.P4_In, S_Ing := #DataIn.P4.Sens_Ing);
   #Sens.P4_OutOn := "A0301_SelSensorON"(SensorsToUse := #SensorToUse.P4_Out, S_Ing := #DataIn.P4.Sens_Out);
   #TON.P4.Sens_Ing.DelayOn.TON(IN := #Sens.P4_IngOn, PT := "A0301_PERS".SensTime.P4.Sens_Ing.DelayOn);
   #Sts.P4.Fermi.Sens_Ing := #TON.P4.Sens_Ing.DelayOn.Q AND #TON.P4.Sens_Ing.DelayOn.Q;
   #TON.P4.Sens_Out.DelayOff.TOF(IN := #Sens.P4_OutOn, PT := "A0301_PERS".SensTime.P4.Sens_Out.DelayOff);
   #Sts.P4.Fermi.Sens_Out := #TON.P4.Sens_Out.DelayOff.Q AND #TON.P4.Sens_Out.DelayOff.Q;
END_REGION

REGION Network 14: <<<<<<<<<<<<<<< TRASPORTO >>>>>>>>>>>>>
END_REGION

REGION Network 15: [Ax] Trasporto - Controllo condizioni di START - Fwd
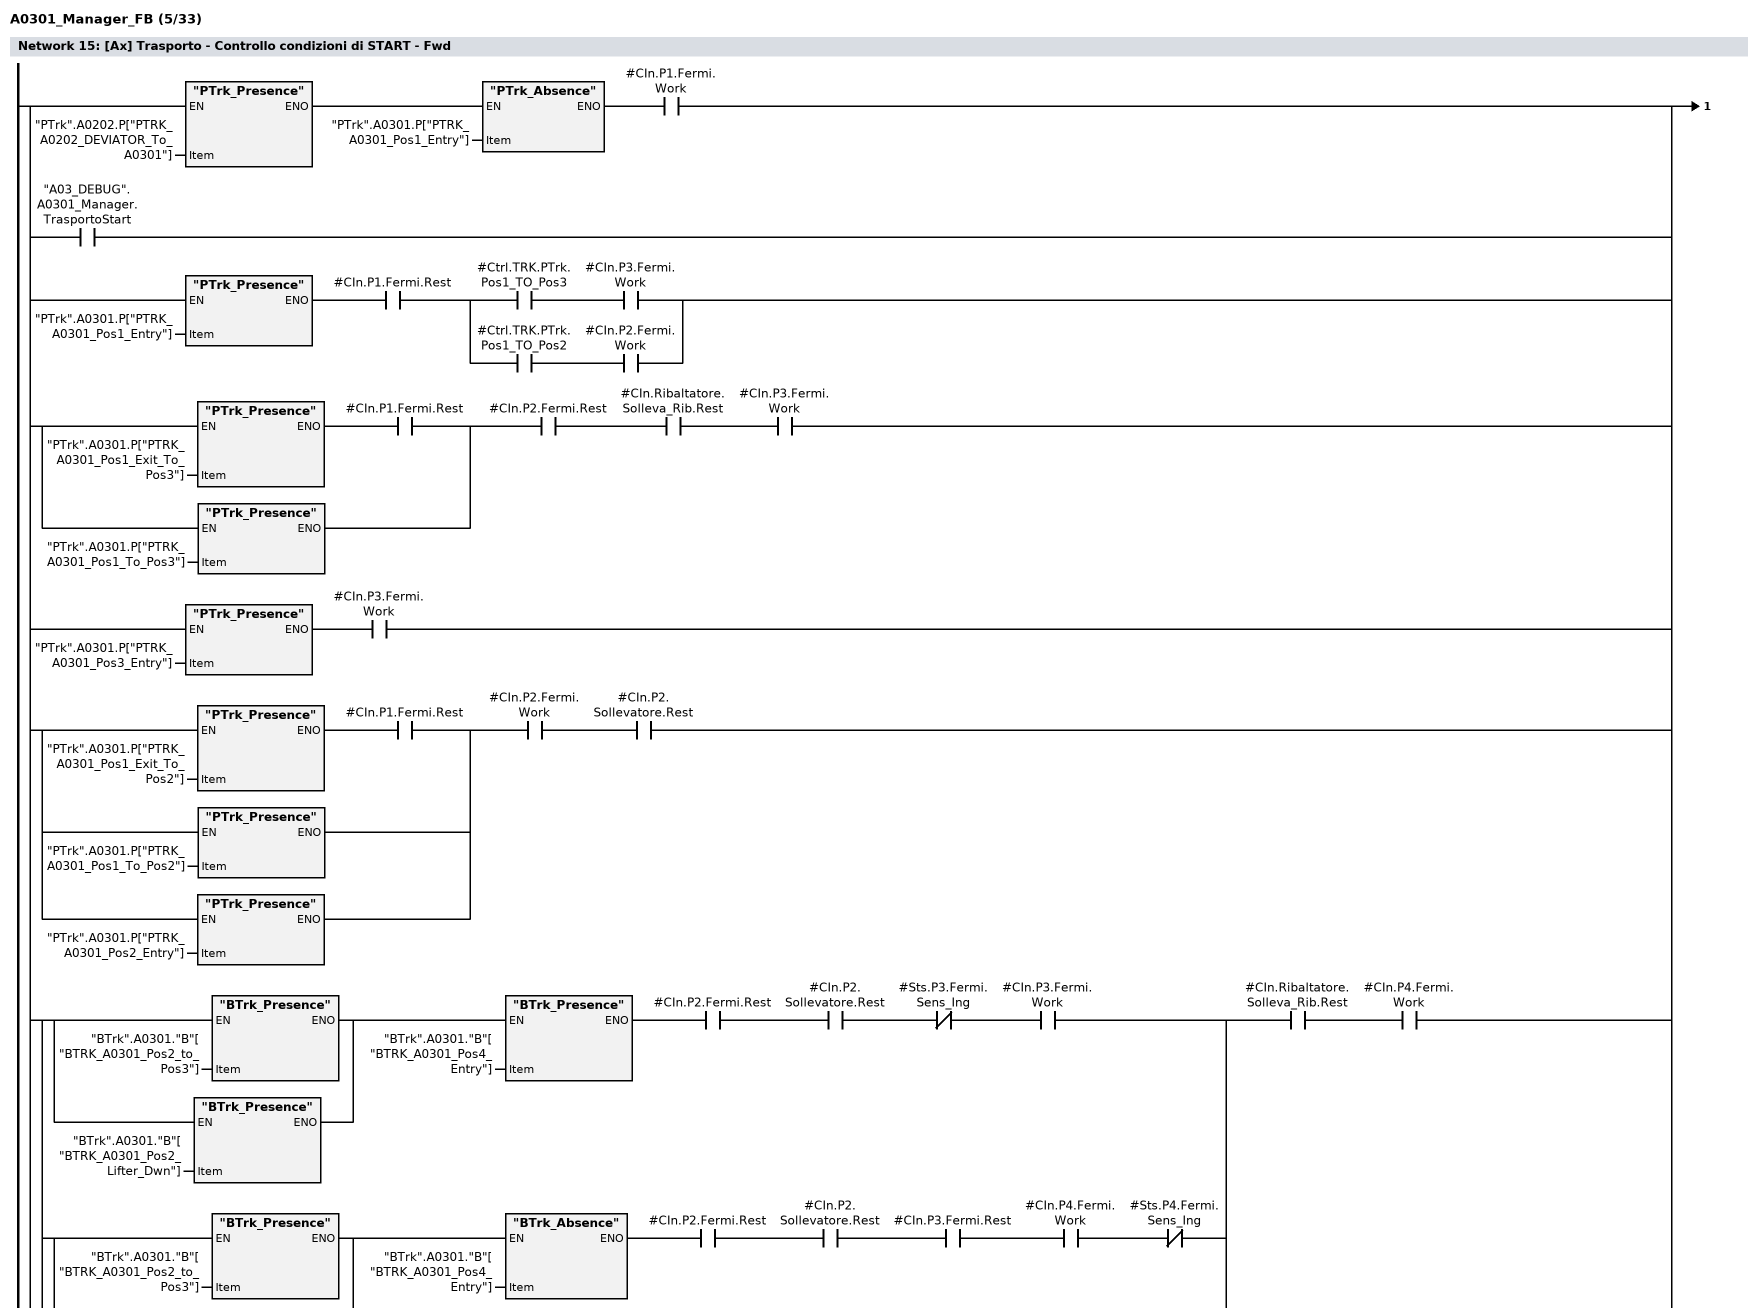
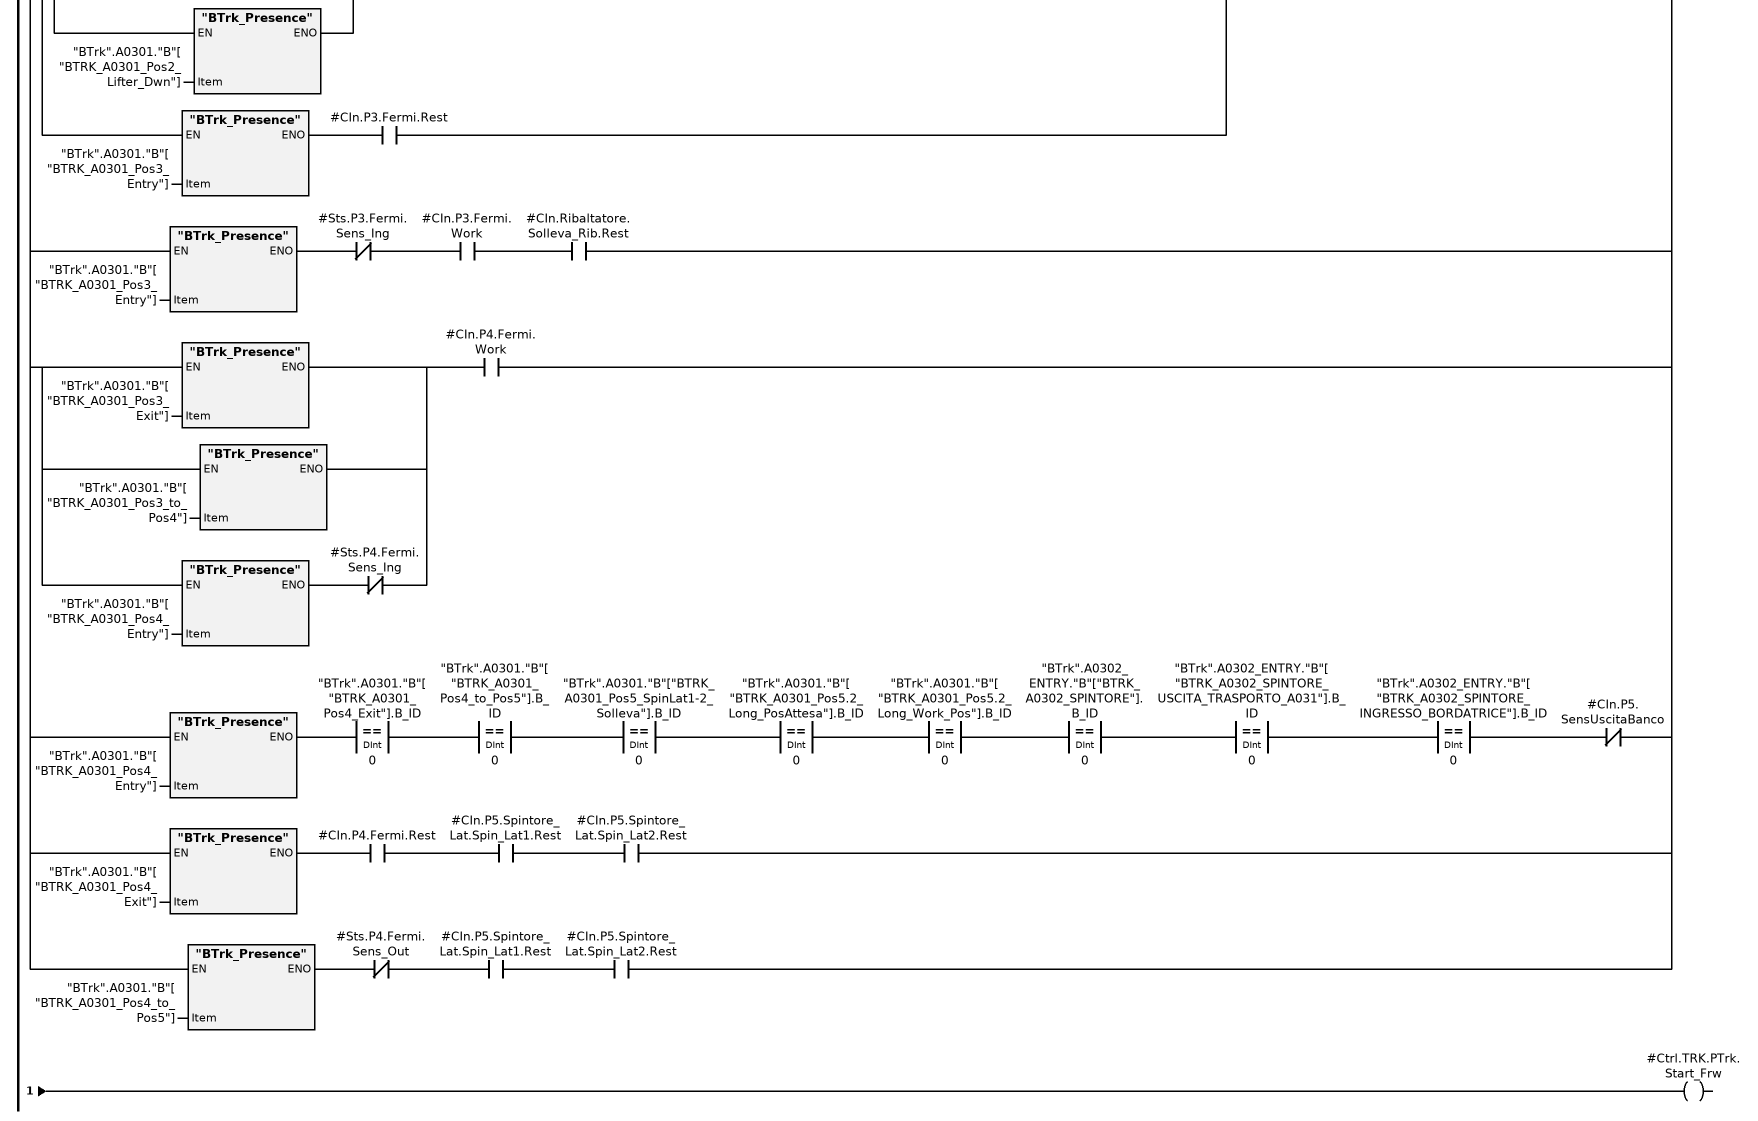
   RUNG wire#powerrail
      "PTrk_Presence"(Item := "PTrk".A0202.P["PTRK_A0202_DEVIATOR_To_A0301"])
      "PTrk_Absence"(Item := "PTrk".A0301.P["PTRK_A0301_Pos1_Entry"])
      Contact( #CIn.P1.Fermi.Work )
      wire#w1
      Coil( #Ctrl.TRK.PTrk.Start_Frw )
   END_RUNG
   RUNG wire#powerrail
      Contact( "A03_DEBUG".A0301_Manager.TrasportoStart )
   END_RUNG wire#w1
   RUNG wire#powerrail
      "PTrk_Presence"(Item := "PTrk".A0301.P["PTRK_A0301_Pos1_Entry"])
      Contact( #CIn.P1.Fermi.Rest )
      wire#w2
      Contact( #Ctrl.TRK.PTrk.Pos1_TO_Pos3 )
      Contact( #CIn.P3.Fermi.Work )
   END_RUNG wire#w1
   RUNG wire#w2
      Contact( #Ctrl.TRK.PTrk.Pos1_TO_Pos2 )
      Contact( #CIn.P2.Fermi.Work )
   END_RUNG wire#w1
   RUNG wire#powerrail
      "PTrk_Presence"(Item := "PTrk".A0301.P["PTRK_A0301_Pos1_Exit_To_Pos3"])
      Contact( #CIn.P1.Fermi.Rest )
      wire#w3
      Contact( #CIn.P2.Fermi.Rest )
      Contact( #CIn.Ribaltatore.Solleva_Rib.Rest )
      Contact( #CIn.P3.Fermi.Work )
   END_RUNG wire#w1
   RUNG wire#powerrail
      "PTrk_Presence"(Item := "PTrk".A0301.P["PTRK_A0301_Pos1_To_Pos3"])
   END_RUNG wire#w3
   RUNG wire#powerrail
      "PTrk_Presence"(Item := "PTrk".A0301.P["PTRK_A0301_Pos3_Entry"])
      Contact( #CIn.P3.Fermi.Work )
   END_RUNG wire#w1
   RUNG wire#powerrail
      "PTrk_Presence"(Item := "PTrk".A0301.P["PTRK_A0301_Pos1_Exit_To_Pos2"])
      Contact( #CIn.P1.Fermi.Rest )
      wire#w4
      Contact( #CIn.P2.Fermi.Work )
      Contact( #CIn.P2.Sollevatore.Rest )
   END_RUNG wire#w1
   RUNG wire#powerrail
      "PTrk_Presence"(Item := "PTrk".A0301.P["PTRK_A0301_Pos1_To_Pos2"])
   END_RUNG wire#w4
   RUNG wire#powerrail
      "PTrk_Presence"(Item := "PTrk".A0301.P["PTRK_A0301_Pos2_Entry"])
   END_RUNG wire#w4
   RUNG wire#powerrail
      "BTrk_Presence"(Item := "BTrk".A0301."B"["BTRK_A0301_Pos2_to_Pos3"])
      wire#w5
      "BTrk_Presence"(Item := "BTrk".A0301."B"["BTRK_A0301_Pos4_Entry"])
      Contact( #CIn.P2.Fermi.Rest )
      Contact( #CIn.P2.Sollevatore.Rest )
      I_Contact( #Sts.P3.Fermi.Sens_Ing )
      Contact( #CIn.P3.Fermi.Work )
      wire#w6
      Contact( #CIn.Ribaltatore.Solleva_Rib.Rest )
      Contact( #CIn.P4.Fermi.Work )
   END_RUNG wire#w1
   RUNG wire#powerrail
      "BTrk_Presence"(Item := "BTrk".A0301."B"["BTRK_A0301_Pos2_Lifter_Dwn"])
   END_RUNG wire#w5
   RUNG wire#powerrail
      "BTrk_Presence"(Item := "BTrk".A0301."B"["BTRK_A0301_Pos2_to_Pos3"])
      wire#w7
      "BTrk_Absence"(Item := "BTrk".A0301."B"["BTRK_A0301_Pos4_Entry"])
      Contact( #CIn.P2.Fermi.Rest )
      Contact( #CIn.P2.Sollevatore.Rest )
      Contact( #CIn.P3.Fermi.Rest )
      Contact( #CIn.P4.Fermi.Work )
      I_Contact( #Sts.P4.Fermi.Sens_Ing )
   END_RUNG wire#w6
   RUNG wire#powerrail
      "BTrk_Presence"(Item := "BTrk".A0301."B"["BTRK_A0301_Pos2_Lifter_Dwn"])
   END_RUNG wire#w7
   RUNG wire#powerrail
      "BTrk_Presence"(Item := "BTrk".A0301."B"["BTRK_A0301_Pos3_Entry"])
      Contact( #CIn.P3.Fermi.Rest )
   END_RUNG wire#w6
   RUNG wire#powerrail
      "BTrk_Presence"(Item := "BTrk".A0301."B"["BTRK_A0301_Pos3_Entry"])
      I_Contact( #Sts.P3.Fermi.Sens_Ing )
      Contact( #CIn.P3.Fermi.Work )
      Contact( #CIn.Ribaltatore.Solleva_Rib.Rest )
   END_RUNG wire#w1
   RUNG wire#powerrail
      "BTrk_Presence"(Item := "BTrk".A0301."B"["BTRK_A0301_Pos3_Exit"])
      wire#w8
      Contact( #CIn.P4.Fermi.Work )
   END_RUNG wire#w1
   RUNG wire#powerrail
      "BTrk_Presence"(Item := "BTrk".A0301."B"["BTRK_A0301_Pos3_to_Pos4"])
   END_RUNG wire#w8
   RUNG wire#powerrail
      "BTrk_Presence"(Item := "BTrk".A0301."B"["BTRK_A0301_Pos4_Entry"])
      I_Contact( #Sts.P4.Fermi.Sens_Ing )
   END_RUNG wire#w8
   RUNG wire#powerrail
      "BTrk_Presence"(Item := "BTrk".A0301."B"["BTRK_A0301_Pos4_Entry"])
      { S7_Templates := "SrcType := DInt" } EQ_Contact(in1 := "BTrk".A0301."B"["BTRK_A0301_Pos4_Exit"].B_ID, in2 := 0)
      { S7_Templates := "SrcType := DInt" } EQ_Contact(in1 := "BTrk".A0301."B"["BTRK_A0301_Pos4_to_Pos5"].B_ID, in2 := 0)
      { S7_Templates := "SrcType := DInt" } EQ_Contact(in1 := "BTrk".A0301."B"["BTRK_A0301_Pos5_SpinLat1-2_Solleva"].B_ID, in2 := 0)
      { S7_Templates := "SrcType := DInt" } EQ_Contact(in1 := "BTrk".A0301."B"["BTRK_A0301_Pos5.2_Long_PosAttesa"].B_ID, in2 := 0)
      { S7_Templates := "SrcType := DInt" } EQ_Contact(in1 := "BTrk".A0301."B"["BTRK_A0301_Pos5.2_Long_Work_Pos"].B_ID, in2 := 0)
      { S7_Templates := "SrcType := DInt" } EQ_Contact(in1 := "BTrk".A0302_ENTRY."B"["BTRK_A0302_SPINTORE"].B_ID, in2 := 0)
      { S7_Templates := "SrcType := DInt" } EQ_Contact(in1 := "BTrk".A0302_ENTRY."B"["BTRK_A0302_SPINTORE_USCITA_TRASPORTO_A031"].B_ID, in2 := 0)
      { S7_Templates := "SrcType := DInt" } EQ_Contact(in1 := "BTrk".A0302_ENTRY."B"["BTRK_A0302_SPINTORE_INGRESSO_BORDATRICE"].B_ID, in2 := 0)
      I_Contact( #CIn.P5.SensUscitaBanco )
   END_RUNG wire#w1
   RUNG wire#powerrail
      "BTrk_Presence"(Item := "BTrk".A0301."B"["BTRK_A0301_Pos4_Exit"])
      Contact( #CIn.P4.Fermi.Rest )
      Contact( #CIn.P5.Spintore_Lat.Spin_Lat1.Rest )
      Contact( #CIn.P5.Spintore_Lat.Spin_Lat2.Rest )
   END_RUNG wire#w1
   RUNG wire#powerrail
      "BTrk_Presence"(Item := "BTrk".A0301."B"["BTRK_A0301_Pos4_to_Pos5"])
      I_Contact( #Sts.P4.Fermi.Sens_Out )
      Contact( #CIn.P5.Spintore_Lat.Spin_Lat1.Rest )
      Contact( #CIn.P5.Spintore_Lat.Spin_Lat2.Rest )
   END_RUNG wire#w1
   // the same network as SCL:
   "PTrk_Presence"(Item := "PTrk".A0202.P["PTRK_A0202_DEVIATOR_To_A0301"], ENO => #_w1);
   "PTrk_Absence"(EN := #_w1, Item := "PTrk".A0301.P["PTRK_A0301_Pos1_Entry"], ENO => #_w2);
   #_w4 := "A03_DEBUG".A0301_Manager.TrasportoStart;
   "PTrk_Presence"(Item := "PTrk".A0301.P["PTRK_A0301_Pos1_Entry"], ENO => #_w3);
   "PTrk_Presence"(Item := "PTrk".A0301.P["PTRK_A0301_Pos1_Exit_To_Pos3"], ENO => #_w5);
   "PTrk_Presence"(Item := "PTrk".A0301.P["PTRK_A0301_Pos1_To_Pos3"], ENO => #_w6);
   "PTrk_Presence"(Item := "PTrk".A0301.P["PTRK_A0301_Pos3_Entry"], ENO => #_w7);
   "PTrk_Presence"(Item := "PTrk".A0301.P["PTRK_A0301_Pos1_Exit_To_Pos2"], ENO => #_w8);
   "PTrk_Presence"(Item := "PTrk".A0301.P["PTRK_A0301_Pos1_To_Pos2"], ENO => #_w9);
   "PTrk_Presence"(Item := "PTrk".A0301.P["PTRK_A0301_Pos2_Entry"], ENO => #_w10);
   "BTrk_Presence"(Item := "BTrk".A0301."B"["BTRK_A0301_Pos2_to_Pos3"], ENO => #_w11);
   "BTrk_Presence"(Item := "BTrk".A0301."B"["BTRK_A0301_Pos2_Lifter_Dwn"], ENO => #_w12);
   "BTrk_Presence"(EN := #_w11 OR #_w12, Item := "BTrk".A0301."B"["BTRK_A0301_Pos4_Entry"], ENO => #_w13);
   "BTrk_Presence"(Item := "BTrk".A0301."B"["BTRK_A0301_Pos2_to_Pos3"], ENO => #_w14);
   "BTrk_Presence"(Item := "BTrk".A0301."B"["BTRK_A0301_Pos2_Lifter_Dwn"], ENO => #_w15);
   "BTrk_Absence"(EN := #_w14 OR #_w15, Item := "BTrk".A0301."B"["BTRK_A0301_Pos4_Entry"], ENO => #_w16);
   "BTrk_Presence"(Item := "BTrk".A0301."B"["BTRK_A0301_Pos3_Entry"], ENO => #_w17);
   "BTrk_Presence"(Item := "BTrk".A0301."B"["BTRK_A0301_Pos3_Entry"], ENO => #_w18);
   "BTrk_Presence"(Item := "BTrk".A0301."B"["BTRK_A0301_Pos3_Exit"], ENO => #_w19);
   "BTrk_Presence"(Item := "BTrk".A0301."B"["BTRK_A0301_Pos3_to_Pos4"], ENO => #_w20);
   "BTrk_Presence"(Item := "BTrk".A0301."B"["BTRK_A0301_Pos4_Entry"], ENO => #_w21);
   "BTrk_Presence"(Item := "BTrk".A0301."B"["BTRK_A0301_Pos4_Entry"], ENO => #_w22);
   #_w24 := #_w22 AND ("BTrk".A0301."B"["BTRK_A0301_Pos4_Exit"].B_ID = 0) AND ("BTrk".A0301."B"["BTRK_A0301_Pos4_to_Pos5"].B_ID = 0) AND ("BTrk".A0301."B"["BTRK_A0301_Pos5_SpinLat1-2_Solleva"].B_ID = 0) AND ("BTrk".A0301."B"["BTRK_A0301_Pos5.2_Long_PosAttesa"].B_ID = 0) AND ("BTrk".A0301."B"["BTRK_A0301_Pos5.2_Long_Work_Pos"].B_ID = 0) AND ("BTrk".A0302_ENTRY."B"["BTRK_A0302_SPINTORE"].B_ID = 0) AND ("BTrk".A0302_ENTRY."B"["BTRK_A0302_SPINTORE_USCITA_TRASPORTO_A031"].B_ID = 0) AND ("BTrk".A0302_ENTRY."B"["BTRK_A0302_SPINTORE_INGRESSO_BORDATRICE"].B_ID = 0) AND NOT #CIn.P5.SensUscitaBanco;
   "BTrk_Presence"(Item := "BTrk".A0301."B"["BTRK_A0301_Pos4_Exit"], ENO => #_w23);
   "BTrk_Presence"(Item := "BTrk".A0301."B"["BTRK_A0301_Pos4_to_Pos5"], ENO => #_w25);
   #Ctrl.TRK.PTrk.Start_Frw := (#_w2 AND #CIn.P1.Fermi.Work) OR #_w4 OR (#_w3 AND #CIn.P1.Fermi.Rest AND ((#Ctrl.TRK.PTrk.Pos1_TO_Pos3 AND #CIn.P3.Fermi.Work) OR (#Ctrl.TRK.PTrk.Pos1_TO_Pos2 AND #CIn.P2.Fermi.Work))) OR (((#_w5 AND #CIn.P1.Fermi.Rest) OR #_w6) AND #CIn.P2.Fermi.Rest AND #CIn.Ribaltatore.Solleva_Rib.Rest AND #CIn.P3.Fermi.Work) OR (#_w7 AND #CIn.P3.Fermi.Work) OR (((#_w8 AND #CIn.P1.Fermi.Rest) OR #_w9 OR #_w10) AND #CIn.P2.Fermi.Work AND #CIn.P2.Sollevatore.Rest) OR (((#_w13 AND #CIn.P2.Fermi.Rest AND #CIn.P2.Sollevatore.Rest AND NOT #Sts.P3.Fermi.Sens_Ing AND #CIn.P3.Fermi.Work) OR (#_w16 AND #CIn.P2.Fermi.Rest AND #CIn.P2.Sollevatore.Rest AND #CIn.P3.Fermi.Rest AND #CIn.P4.Fermi.Work AND NOT #Sts.P4.Fermi.Sens_Ing) OR (#_w17 AND #CIn.P3.Fermi.Rest)) AND #CIn.Ribaltatore.Solleva_Rib.Rest AND #CIn.P4.Fermi.Work) OR (#_w18 AND NOT #Sts.P3.Fermi.Sens_Ing AND #CIn.P3.Fermi.Work AND #CIn.Ribaltatore.Solleva_Rib.Rest) OR ((#_w19 OR #_w20 OR (#_w21 AND NOT #Sts.P4.Fermi.Sens_Ing)) AND #CIn.P4.Fermi.Work) OR #_w24 OR (#_w23 AND #CIn.P4.Fermi.Rest AND #CIn.P5.Spintore_Lat.Spin_Lat1.Rest AND #CIn.P5.Spintore_Lat.Spin_Lat2.Rest) OR (#_w25 AND NOT #Sts.P4.Fermi.Sens_Out AND #CIn.P5.Spintore_Lat.Spin_Lat1.Rest AND #CIn.P5.Spintore_Lat.Spin_Lat2.Rest);
END_REGION

REGION Network 16: [Ax] Trasporto - COut Manager
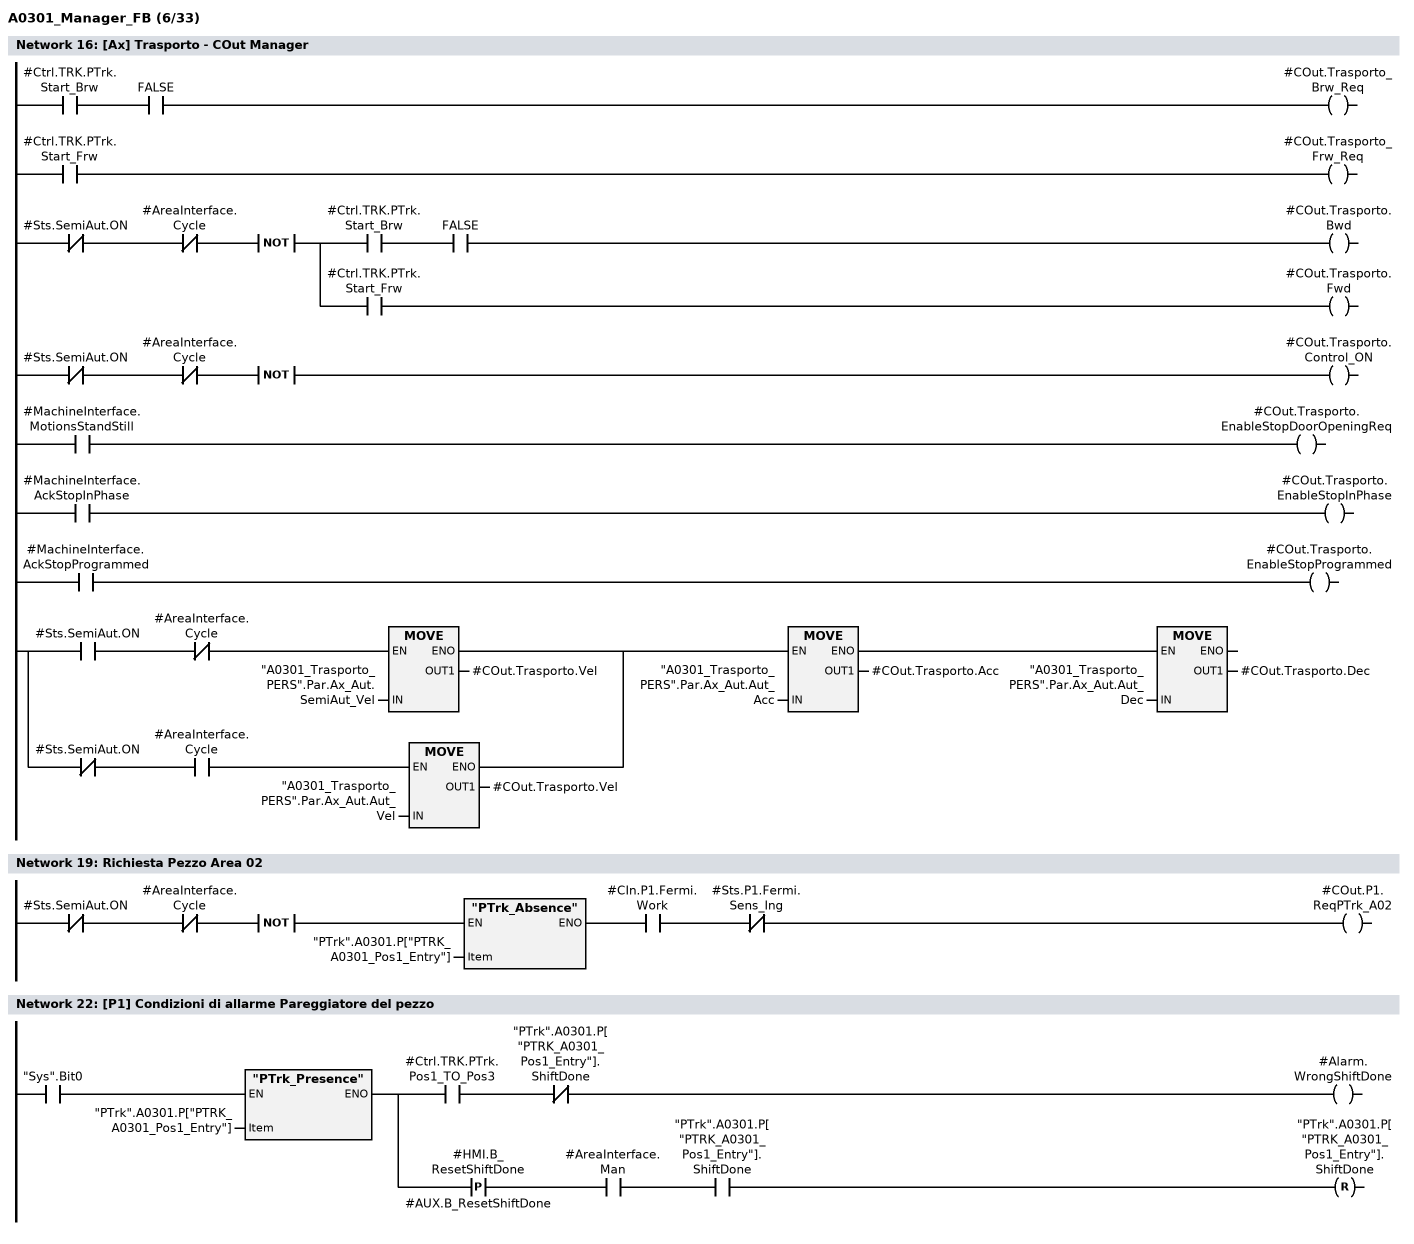
   RUNG wire#powerrail
      Contact( #Ctrl.TRK.PTrk.Start_Brw )
      Contact( FALSE )
      Coil( #COut.Trasporto_Brw_Req )
   END_RUNG
   RUNG wire#powerrail
      Contact( #Ctrl.TRK.PTrk.Start_Frw )
      Coil( #COut.Trasporto_Frw_Req )
   END_RUNG
   RUNG wire#powerrail
      I_Contact( #Sts.SemiAut.ON )
      I_Contact( #AreaInterface.Cycle )
      Not()
      wire#w1
      Contact( #Ctrl.TRK.PTrk.Start_Brw )
      Contact( FALSE )
      Coil( #COut.Trasporto.Bwd )
   END_RUNG
   RUNG wire#w1
      Contact( #Ctrl.TRK.PTrk.Start_Frw )
      Coil( #COut.Trasporto.Fwd )
   END_RUNG
   RUNG wire#powerrail
      I_Contact( #Sts.SemiAut.ON )
      I_Contact( #AreaInterface.Cycle )
      Not()
      Coil( #COut.Trasporto.Control_ON )
   END_RUNG
   RUNG wire#powerrail
      Contact( #MachineInterface.MotionsStandStill )
      Coil( #COut.Trasporto.EnableStopDoorOpeningReq )
   END_RUNG
   RUNG wire#powerrail
      Contact( #MachineInterface.AckStopInPhase )
      Coil( #COut.Trasporto.EnableStopInPhase )
   END_RUNG
   RUNG wire#powerrail
      Contact( #MachineInterface.AckStopProgrammed )
      Coil( #COut.Trasporto.EnableStopProgrammed )
   END_RUNG
   RUNG wire#powerrail
      Contact( #Sts.SemiAut.ON )
      I_Contact( #AreaInterface.Cycle )
      Move(in := "A0301_Trasporto_PERS".Par.Ax_Aut.SemiAut_Vel, out1 => #COut.Trasporto.Vel)
      wire#w2
      Move(in := "A0301_Trasporto_PERS".Par.Ax_Aut.Aut_Acc, out1 => #COut.Trasporto.Acc)
      Move(in := "A0301_Trasporto_PERS".Par.Ax_Aut.Aut_Dec, out1 => #COut.Trasporto.Dec)
   END_RUNG
   RUNG wire#powerrail
      I_Contact( #Sts.SemiAut.ON )
      Contact( #AreaInterface.Cycle )
      Move(in := "A0301_Trasporto_PERS".Par.Ax_Aut.Aut_Vel, out1 => #COut.Trasporto.Vel)
   END_RUNG wire#w2
   // the same network as SCL:
   #COut.Trasporto_Brw_Req := #Ctrl.TRK.PTrk.Start_Brw AND FALSE;
   #COut.Trasporto_Frw_Req := #Ctrl.TRK.PTrk.Start_Frw;
   #_w1 := NOT (NOT #Sts.SemiAut.ON AND NOT #AreaInterface.Cycle);
   #COut.Trasporto.Bwd := #_w1 AND #Ctrl.TRK.PTrk.Start_Brw AND FALSE;
   #COut.Trasporto.Fwd := #_w1 AND #Ctrl.TRK.PTrk.Start_Frw;
   #COut.Trasporto.Control_ON := NOT (NOT #Sts.SemiAut.ON AND NOT #AreaInterface.Cycle);
   #COut.Trasporto.EnableStopDoorOpeningReq := #MachineInterface.MotionsStandStill;
   #COut.Trasporto.EnableStopInPhase := #MachineInterface.AckStopInPhase;
   #COut.Trasporto.EnableStopProgrammed := #MachineInterface.AckStopProgrammed;
   #_w2 := #Sts.SemiAut.ON AND NOT #AreaInterface.Cycle;
   IF #_w2 THEN #COut.Trasporto.Vel := "A0301_Trasporto_PERS".Par.Ax_Aut.SemiAut_Vel; END_IF;
   #_w3 := NOT #Sts.SemiAut.ON AND #AreaInterface.Cycle;
   IF #_w3 THEN #COut.Trasporto.Vel := "A0301_Trasporto_PERS".Par.Ax_Aut.Aut_Vel; END_IF;
   IF #_w2 OR #_w3 THEN
       #COut.Trasporto.Acc := "A0301_Trasporto_PERS".Par.Ax_Aut.Aut_Acc;
       #COut.Trasporto.Dec := "A0301_Trasporto_PERS".Par.Ax_Aut.Aut_Dec;
   END_IF;
END_REGION

REGION Network 18: <<<<<<<<< MOVIMENTO TRAKING >>>>>>>>>
END_REGION

REGION Network 19: Richiesta Pezzo Area 02
   RUNG wire#powerrail
      I_Contact( #Sts.SemiAut.ON )
      I_Contact( #AreaInterface.Cycle )
      Not()
      "PTrk_Absence"(Item := "PTrk".A0301.P["PTRK_A0301_Pos1_Entry"])
      Contact( #CIn.P1.Fermi.Work )
      I_Contact( #Sts.P1.Fermi.Sens_Ing )
      Coil( #COut.P1.ReqPTrk_A02 )
   END_RUNG
   // the same network as SCL:
   "PTrk_Absence"(EN := NOT (NOT #Sts.SemiAut.ON AND NOT #AreaInterface.Cycle),
                  Item := "PTrk".A0301.P["PTRK_A0301_Pos1_Entry"],
                  ENO => #_w1);
   #COut.P1.ReqPTrk_A02 := #_w1 AND #CIn.P1.Fermi.Work AND NOT #Sts.P1.Fermi.Sens_Ing;
END_REGION

REGION Network 21: <<<<<<<<<<< POSIZIONE 1 >>>>>>>>>>>>>>
END_REGION

REGION Network 22: [P1] Condizioni di allarme Pareggiatore del pezzo
   RUNG wire#powerrail
      Contact( "Sys".Bit0 )
      "PTrk_Presence"(Item := "PTrk".A0301.P["PTRK_A0301_Pos1_Entry"])
      wire#w1
      Contact( #Ctrl.TRK.PTrk.Pos1_TO_Pos3 )
      I_Contact( "PTrk".A0301.P["PTRK_A0301_Pos1_Entry"].ShiftDone )
      Coil( #Alarm.WrongShiftDone )
   END_RUNG
   RUNG wire#w1
      P_Contact(operand := #HMI.B_ResetShiftDone, bit := #AUX.B_ResetShiftDone)
      Contact( #AreaInterface.Man )
      Contact( "PTrk".A0301.P["PTRK_A0301_Pos1_Entry"].ShiftDone )
      R_Coil( "PTrk".A0301.P["PTRK_A0301_Pos1_Entry"].ShiftDone )
   END_RUNG
   // the same network as SCL:
   "PTrk_Presence"(EN := "Sys".Bit0, Item := "PTrk".A0301.P["PTRK_A0301_Pos1_Entry"], ENO => #_w1);
   #Alarm.WrongShiftDone := #_w1 AND #Ctrl.TRK.PTrk.Pos1_TO_Pos3 AND NOT "PTrk".A0301.P["PTRK_A0301_Pos1_Entry"].ShiftDone;
   #_w2 := #_w1 AND #HMI.B_ResetShiftDone AND NOT #AUX.B_ResetShiftDone;   // rising edge of #HMI.B_ResetShiftDone
   #AUX.B_ResetShiftDone := #HMI.B_ResetShiftDone;
   IF #_w2 AND #AreaInterface.Man AND "PTrk".A0301.P["PTRK_A0301_Pos1_Entry"].ShiftDone THEN
       "PTrk".A0301.P["PTRK_A0301_Pos1_Entry"].ShiftDone := FALSE;
   END_IF;
END_REGION

REGION Network 24: << CONTROLLO RICHIESTE MOVIMENTO TRAKING PTrk >>
END_REGION

REGION Network 25: [P1] Richiesta movimento Part agli stopper P2
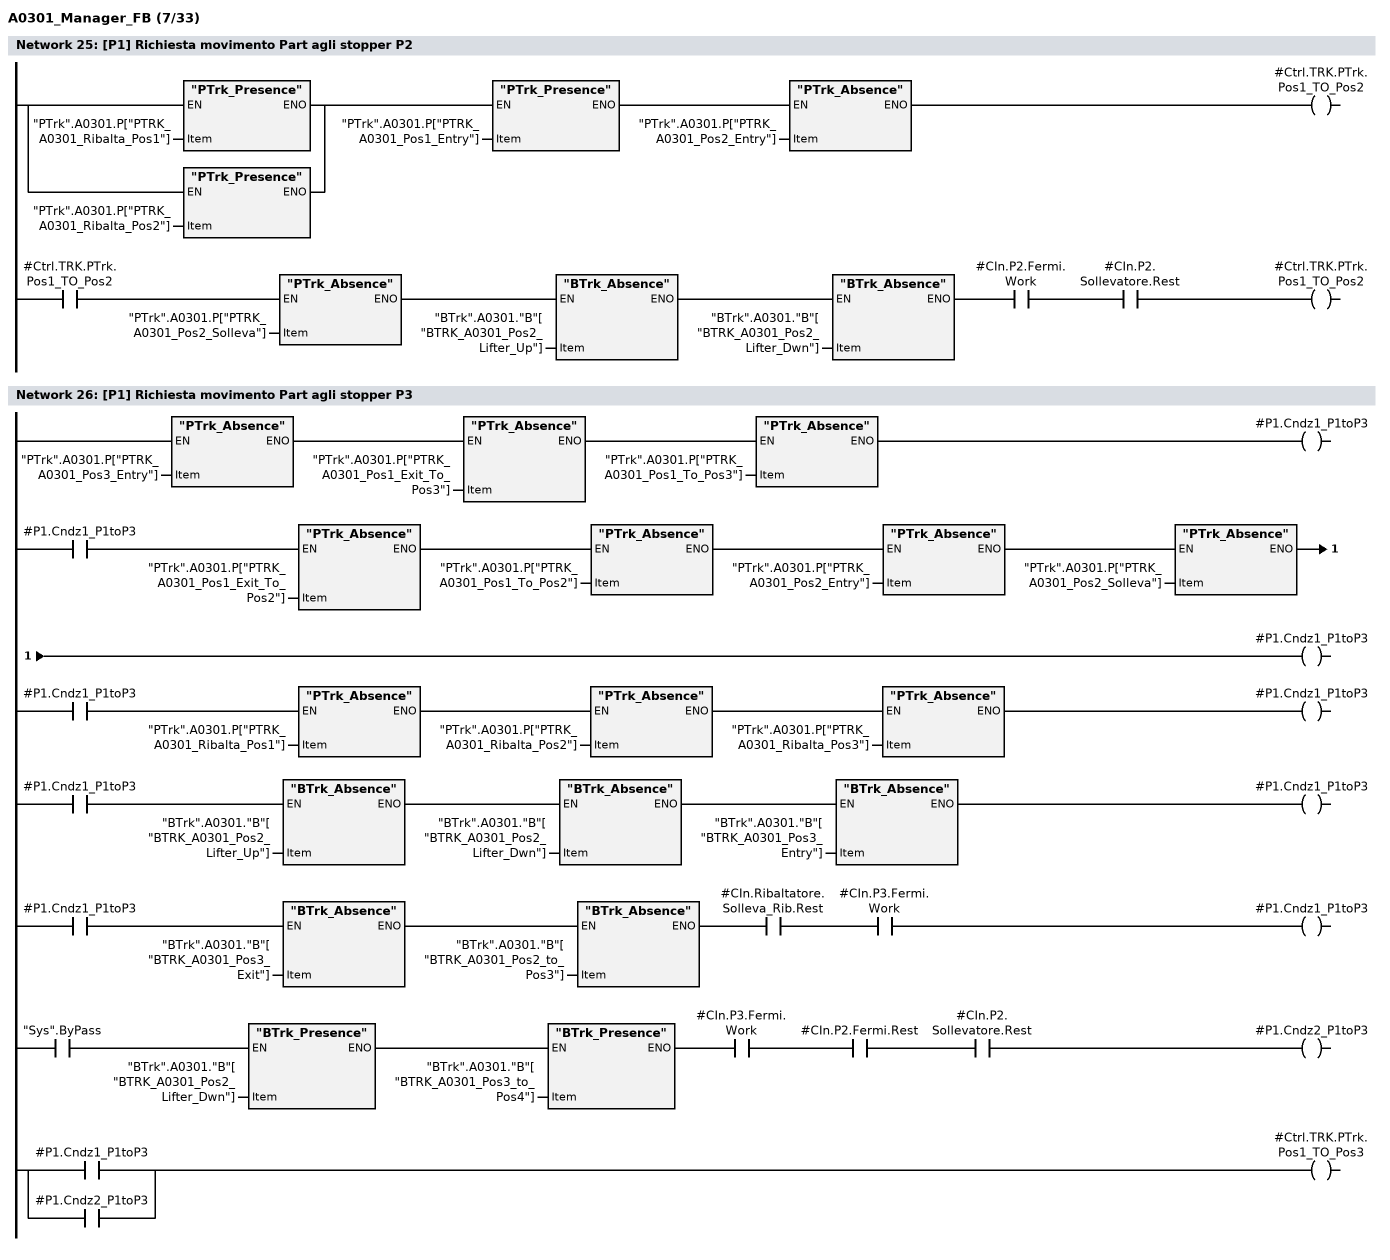
   RUNG wire#powerrail
      "PTrk_Presence"(Item := "PTrk".A0301.P["PTRK_A0301_Ribalta_Pos1"])
      wire#w1
      "PTrk_Presence"(Item := "PTrk".A0301.P["PTRK_A0301_Pos1_Entry"])
      "PTrk_Absence"(Item := "PTrk".A0301.P["PTRK_A0301_Pos2_Entry"])
      Coil( #Ctrl.TRK.PTrk.Pos1_TO_Pos2 )
   END_RUNG
   RUNG wire#powerrail
      "PTrk_Presence"(Item := "PTrk".A0301.P["PTRK_A0301_Ribalta_Pos2"])
   END_RUNG wire#w1
   RUNG wire#powerrail
      Contact( #Ctrl.TRK.PTrk.Pos1_TO_Pos2 )
      "PTrk_Absence"(Item := "PTrk".A0301.P["PTRK_A0301_Pos2_Solleva"])
      "BTrk_Absence"(Item := "BTrk".A0301."B"["BTRK_A0301_Pos2_Lifter_Up"])
      "BTrk_Absence"(Item := "BTrk".A0301."B"["BTRK_A0301_Pos2_Lifter_Dwn"])
      Contact( #CIn.P2.Fermi.Work )
      Contact( #CIn.P2.Sollevatore.Rest )
      Coil( #Ctrl.TRK.PTrk.Pos1_TO_Pos2 )
   END_RUNG
   // the same network as SCL:
   "PTrk_Presence"(Item := "PTrk".A0301.P["PTRK_A0301_Ribalta_Pos1"], ENO => #_w1);
   "PTrk_Presence"(Item := "PTrk".A0301.P["PTRK_A0301_Ribalta_Pos2"], ENO => #_w2);
   "PTrk_Presence"(EN := #_w1 OR #_w2, Item := "PTrk".A0301.P["PTRK_A0301_Pos1_Entry"], ENO => #_w3);
   "PTrk_Absence"(EN := #_w3, Item := "PTrk".A0301.P["PTRK_A0301_Pos2_Entry"], ENO => #_w4);
   #Ctrl.TRK.PTrk.Pos1_TO_Pos2 := #_w4;
   "PTrk_Absence"(EN := #Ctrl.TRK.PTrk.Pos1_TO_Pos2,
                  Item := "PTrk".A0301.P["PTRK_A0301_Pos2_Solleva"],
                  ENO => #_w5);
   "BTrk_Absence"(EN := #_w5, Item := "BTrk".A0301."B"["BTRK_A0301_Pos2_Lifter_Up"], ENO => #_w6);
   "BTrk_Absence"(EN := #_w6, Item := "BTrk".A0301."B"["BTRK_A0301_Pos2_Lifter_Dwn"], ENO => #_w7);
   #Ctrl.TRK.PTrk.Pos1_TO_Pos2 := #_w7 AND #CIn.P2.Fermi.Work AND #CIn.P2.Sollevatore.Rest;
END_REGION

REGION Network 26: [P1] Richiesta movimento Part agli stopper P3
   RUNG wire#powerrail
      "PTrk_Absence"(Item := "PTrk".A0301.P["PTRK_A0301_Pos3_Entry"])
      "PTrk_Absence"(Item := "PTrk".A0301.P["PTRK_A0301_Pos1_Exit_To_Pos3"])
      "PTrk_Absence"(Item := "PTrk".A0301.P["PTRK_A0301_Pos1_To_Pos3"])
      Coil( #P1.Cndz1_P1toP3 )
   END_RUNG
   RUNG wire#powerrail
      Contact( #P1.Cndz1_P1toP3 )
      "PTrk_Absence"(Item := "PTrk".A0301.P["PTRK_A0301_Pos1_Exit_To_Pos2"])
      "PTrk_Absence"(Item := "PTrk".A0301.P["PTRK_A0301_Pos1_To_Pos2"])
      "PTrk_Absence"(Item := "PTrk".A0301.P["PTRK_A0301_Pos2_Entry"])
      "PTrk_Absence"(Item := "PTrk".A0301.P["PTRK_A0301_Pos2_Solleva"])
      Coil( #P1.Cndz1_P1toP3 )
   END_RUNG
   RUNG wire#powerrail
      Contact( #P1.Cndz1_P1toP3 )
      "PTrk_Absence"(Item := "PTrk".A0301.P["PTRK_A0301_Ribalta_Pos1"])
      "PTrk_Absence"(Item := "PTrk".A0301.P["PTRK_A0301_Ribalta_Pos2"])
      "PTrk_Absence"(Item := "PTrk".A0301.P["PTRK_A0301_Ribalta_Pos3"])
      Coil( #P1.Cndz1_P1toP3 )
   END_RUNG
   RUNG wire#powerrail
      Contact( #P1.Cndz1_P1toP3 )
      "BTrk_Absence"(Item := "BTrk".A0301."B"["BTRK_A0301_Pos2_Lifter_Up"])
      "BTrk_Absence"(Item := "BTrk".A0301."B"["BTRK_A0301_Pos2_Lifter_Dwn"])
      "BTrk_Absence"(Item := "BTrk".A0301."B"["BTRK_A0301_Pos3_Entry"])
      Coil( #P1.Cndz1_P1toP3 )
   END_RUNG
   RUNG wire#powerrail
      Contact( #P1.Cndz1_P1toP3 )
      "BTrk_Absence"(Item := "BTrk".A0301."B"["BTRK_A0301_Pos3_Exit"])
      "BTrk_Absence"(Item := "BTrk".A0301."B"["BTRK_A0301_Pos2_to_Pos3"])
      Contact( #CIn.Ribaltatore.Solleva_Rib.Rest )
      Contact( #CIn.P3.Fermi.Work )
      Coil( #P1.Cndz1_P1toP3 )
   END_RUNG
   RUNG wire#powerrail
      Contact( "Sys".ByPass )
      "BTrk_Presence"(Item := "BTrk".A0301."B"["BTRK_A0301_Pos2_Lifter_Dwn"])
      "BTrk_Presence"(Item := "BTrk".A0301."B"["BTRK_A0301_Pos3_to_Pos4"])
      Contact( #CIn.P3.Fermi.Work )
      Contact( #CIn.P2.Fermi.Rest )
      Contact( #CIn.P2.Sollevatore.Rest )
      Coil( #P1.Cndz2_P1toP3 )
   END_RUNG
   RUNG wire#powerrail
      Contact( #P1.Cndz1_P1toP3 )
      wire#w1
      Coil( #Ctrl.TRK.PTrk.Pos1_TO_Pos3 )
   END_RUNG
   RUNG wire#powerrail
      Contact( #P1.Cndz2_P1toP3 )
   END_RUNG wire#w1
   // the same network as SCL:
   "PTrk_Absence"(Item := "PTrk".A0301.P["PTRK_A0301_Pos3_Entry"], ENO => #_w1);
   "PTrk_Absence"(EN := #_w1, Item := "PTrk".A0301.P["PTRK_A0301_Pos1_Exit_To_Pos3"], ENO => #_w2);
   "PTrk_Absence"(EN := #_w2, Item := "PTrk".A0301.P["PTRK_A0301_Pos1_To_Pos3"], ENO => #_w3);
   #P1.Cndz1_P1toP3 := #_w3;
   "PTrk_Absence"(EN := #P1.Cndz1_P1toP3, Item := "PTrk".A0301.P["PTRK_A0301_Pos1_Exit_To_Pos2"], ENO => #_w4);
   "PTrk_Absence"(EN := #_w4, Item := "PTrk".A0301.P["PTRK_A0301_Pos1_To_Pos2"], ENO => #_w5);
   "PTrk_Absence"(EN := #_w5, Item := "PTrk".A0301.P["PTRK_A0301_Pos2_Entry"], ENO => #_w6);
   "PTrk_Absence"(EN := #_w6, Item := "PTrk".A0301.P["PTRK_A0301_Pos2_Solleva"], ENO => #_w7);
   #P1.Cndz1_P1toP3 := #_w7;
   "PTrk_Absence"(EN := #P1.Cndz1_P1toP3, Item := "PTrk".A0301.P["PTRK_A0301_Ribalta_Pos1"], ENO => #_w8);
   "PTrk_Absence"(EN := #_w8, Item := "PTrk".A0301.P["PTRK_A0301_Ribalta_Pos2"], ENO => #_w9);
   "PTrk_Absence"(EN := #_w9, Item := "PTrk".A0301.P["PTRK_A0301_Ribalta_Pos3"], ENO => #_w10);
   #P1.Cndz1_P1toP3 := #_w10;
   "BTrk_Absence"(EN := #P1.Cndz1_P1toP3, Item := "BTrk".A0301."B"["BTRK_A0301_Pos2_Lifter_Up"], ENO => #_w11);
   "BTrk_Absence"(EN := #_w11, Item := "BTrk".A0301."B"["BTRK_A0301_Pos2_Lifter_Dwn"], ENO => #_w12);
   "BTrk_Absence"(EN := #_w12, Item := "BTrk".A0301."B"["BTRK_A0301_Pos3_Entry"], ENO => #_w13);
   #P1.Cndz1_P1toP3 := #_w13;
   "BTrk_Absence"(EN := #P1.Cndz1_P1toP3, Item := "BTrk".A0301."B"["BTRK_A0301_Pos3_Exit"], ENO => #_w14);
   "BTrk_Absence"(EN := #_w14, Item := "BTrk".A0301."B"["BTRK_A0301_Pos2_to_Pos3"], ENO => #_w15);
   #P1.Cndz1_P1toP3 := #_w15 AND #CIn.Ribaltatore.Solleva_Rib.Rest AND #CIn.P3.Fermi.Work;
   "BTrk_Presence"(EN := "Sys".ByPass, Item := "BTrk".A0301."B"["BTRK_A0301_Pos2_Lifter_Dwn"], ENO => #_w16);
   "BTrk_Presence"(EN := #_w16, Item := "BTrk".A0301."B"["BTRK_A0301_Pos3_to_Pos4"], ENO => #_w17);
   #P1.Cndz2_P1toP3 := #_w17 AND #CIn.P3.Fermi.Work AND #CIn.P2.Fermi.Rest AND #CIn.P2.Sollevatore.Rest;
   #Ctrl.TRK.PTrk.Pos1_TO_Pos3 := #P1.Cndz1_P1toP3 OR #P1.Cndz2_P1toP3;
END_REGION

REGION Network 28: <<<<< SPOSTAMENTO TRAKING PTrk >>>>>>
END_REGION

REGION Network 30: P[Pareggiatore] Pareggiamento su A03 Pos.1 eseguito
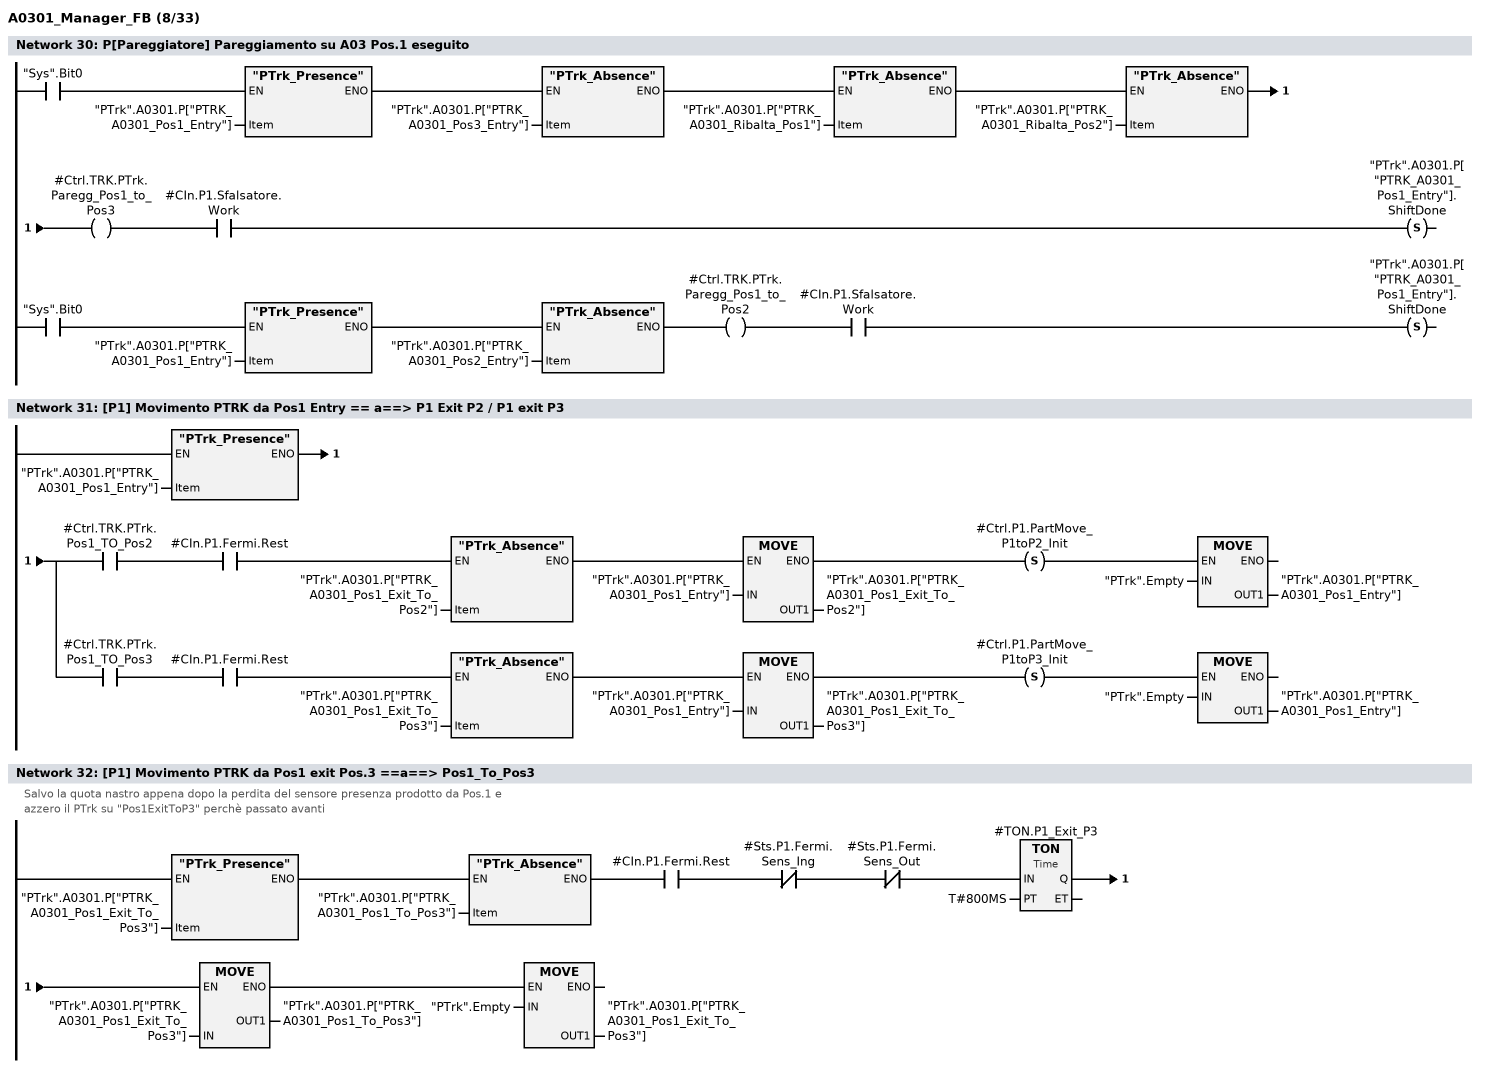
   RUNG wire#powerrail
      Contact( "Sys".Bit0 )
      "PTrk_Presence"(Item := "PTrk".A0301.P["PTRK_A0301_Pos1_Entry"])
      "PTrk_Absence"(Item := "PTrk".A0301.P["PTRK_A0301_Pos3_Entry"])
      "PTrk_Absence"(Item := "PTrk".A0301.P["PTRK_A0301_Ribalta_Pos1"])
      "PTrk_Absence"(Item := "PTrk".A0301.P["PTRK_A0301_Ribalta_Pos2"])
      Coil( #Ctrl.TRK.PTrk.Paregg_Pos1_to_Pos3 )
      Contact( #CIn.P1.Sfalsatore.Work )
      S_Coil( "PTrk".A0301.P["PTRK_A0301_Pos1_Entry"].ShiftDone )
   END_RUNG
   RUNG wire#powerrail
      Contact( "Sys".Bit0 )
      "PTrk_Presence"(Item := "PTrk".A0301.P["PTRK_A0301_Pos1_Entry"])
      "PTrk_Absence"(Item := "PTrk".A0301.P["PTRK_A0301_Pos2_Entry"])
      Coil( #Ctrl.TRK.PTrk.Paregg_Pos1_to_Pos2 )
      Contact( #CIn.P1.Sfalsatore.Work )
      S_Coil( "PTrk".A0301.P["PTRK_A0301_Pos1_Entry"].ShiftDone )
   END_RUNG
   // the same network as SCL:
   "PTrk_Presence"(EN := "Sys".Bit0, Item := "PTrk".A0301.P["PTRK_A0301_Pos1_Entry"], ENO => #_w1);
   "PTrk_Absence"(EN := #_w1, Item := "PTrk".A0301.P["PTRK_A0301_Pos3_Entry"], ENO => #_w2);
   "PTrk_Absence"(EN := #_w2, Item := "PTrk".A0301.P["PTRK_A0301_Ribalta_Pos1"], ENO => #_w3);
   "PTrk_Absence"(EN := #_w3, Item := "PTrk".A0301.P["PTRK_A0301_Ribalta_Pos2"], ENO => #_w4);
   #Ctrl.TRK.PTrk.Paregg_Pos1_to_Pos3 := #_w4;
   IF #_w4 AND #CIn.P1.Sfalsatore.Work THEN
       "PTrk".A0301.P["PTRK_A0301_Pos1_Entry"].ShiftDone := TRUE;
   END_IF;
   "PTrk_Presence"(EN := "Sys".Bit0, Item := "PTrk".A0301.P["PTRK_A0301_Pos1_Entry"], ENO => #_w5);
   "PTrk_Absence"(EN := #_w5, Item := "PTrk".A0301.P["PTRK_A0301_Pos2_Entry"], ENO => #_w6);
   #Ctrl.TRK.PTrk.Paregg_Pos1_to_Pos2 := #_w6;
   IF #_w6 AND #CIn.P1.Sfalsatore.Work THEN
       "PTrk".A0301.P["PTRK_A0301_Pos1_Entry"].ShiftDone := TRUE;
   END_IF;
END_REGION

REGION Network 31: [P1] Movimento PTRK da Pos1 Entry == a==> P1 Exit P2 / P1 exit P3
   RUNG wire#powerrail
      "PTrk_Presence"(Item := "PTrk".A0301.P["PTRK_A0301_Pos1_Entry"])
      wire#w1
      Contact( #Ctrl.TRK.PTrk.Pos1_TO_Pos2 )
      Contact( #CIn.P1.Fermi.Rest )
      "PTrk_Absence"(Item := "PTrk".A0301.P["PTRK_A0301_Pos1_Exit_To_Pos2"])
      Move(in := "PTrk".A0301.P["PTRK_A0301_Pos1_Entry"], out1 => "PTrk".A0301.P["PTRK_A0301_Pos1_Exit_To_Pos2"])
      S_Coil( #Ctrl.P1.PartMove_P1toP2_Init )
      Move(in := "PTrk".Empty, out1 => "PTrk".A0301.P["PTRK_A0301_Pos1_Entry"])
   END_RUNG
   RUNG wire#w1
      Contact( #Ctrl.TRK.PTrk.Pos1_TO_Pos3 )
      Contact( #CIn.P1.Fermi.Rest )
      "PTrk_Absence"(Item := "PTrk".A0301.P["PTRK_A0301_Pos1_Exit_To_Pos3"])
      Move(in := "PTrk".A0301.P["PTRK_A0301_Pos1_Entry"], out1 => "PTrk".A0301.P["PTRK_A0301_Pos1_Exit_To_Pos3"])
      S_Coil( #Ctrl.P1.PartMove_P1toP3_Init )
      Move(in := "PTrk".Empty, out1 => "PTrk".A0301.P["PTRK_A0301_Pos1_Entry"])
   END_RUNG
   // the same network as SCL:
   "PTrk_Presence"(Item := "PTrk".A0301.P["PTRK_A0301_Pos1_Entry"], ENO => #_w1);
   "PTrk_Absence"(EN := #_w1 AND #Ctrl.TRK.PTrk.Pos1_TO_Pos2 AND #CIn.P1.Fermi.Rest,
                  Item := "PTrk".A0301.P["PTRK_A0301_Pos1_Exit_To_Pos2"],
                  ENO => #_w2);
   IF #_w2 THEN
       "PTrk".A0301.P["PTRK_A0301_Pos1_Exit_To_Pos2"] := "PTrk".A0301.P["PTRK_A0301_Pos1_Entry"];
       #Ctrl.P1.PartMove_P1toP2_Init := TRUE;
       "PTrk".A0301.P["PTRK_A0301_Pos1_Entry"] := "PTrk".Empty;
   END_IF;
   "PTrk_Absence"(EN := #_w1 AND #Ctrl.TRK.PTrk.Pos1_TO_Pos3 AND #CIn.P1.Fermi.Rest,
                  Item := "PTrk".A0301.P["PTRK_A0301_Pos1_Exit_To_Pos3"],
                  ENO => #_w3);
   IF #_w3 THEN
       "PTrk".A0301.P["PTRK_A0301_Pos1_Exit_To_Pos3"] := "PTrk".A0301.P["PTRK_A0301_Pos1_Entry"];
       #Ctrl.P1.PartMove_P1toP3_Init := TRUE;
       "PTrk".A0301.P["PTRK_A0301_Pos1_Entry"] := "PTrk".Empty;
   END_IF;
END_REGION

REGION Network 32: [P1] Movimento PTRK da Pos1 exit Pos.3 ==a==> Pos1_To_Pos3
   // Salvo la quota nastro appena dopo la perdita del sensore presenza prodotto da Pos.1 e
   // azzero il PTrk su "Pos1ExitToP3" perchè passato avanti
   RUNG wire#powerrail
      "PTrk_Presence"(Item := "PTrk".A0301.P["PTRK_A0301_Pos1_Exit_To_Pos3"])
      "PTrk_Absence"(Item := "PTrk".A0301.P["PTRK_A0301_Pos1_To_Pos3"])
      Contact( #CIn.P1.Fermi.Rest )
      I_Contact( #Sts.P1.Fermi.Sens_Ing )
      I_Contact( #Sts.P1.Fermi.Sens_Out )
      { S7_Templates := "time_type := Time" } #TON.P1_Exit_P3.TON(pt := T#800MS, et =>)
      Move(in := "PTrk".A0301.P["PTRK_A0301_Pos1_Exit_To_Pos3"], out1 => "PTrk".A0301.P["PTRK_A0301_Pos1_To_Pos3"])
      Move(in := "PTrk".Empty, out1 => "PTrk".A0301.P["PTRK_A0301_Pos1_Exit_To_Pos3"])
   END_RUNG
   // the same network as SCL:
   "PTrk_Presence"(Item := "PTrk".A0301.P["PTRK_A0301_Pos1_Exit_To_Pos3"], ENO => #_w1);
   "PTrk_Absence"(EN := #_w1, Item := "PTrk".A0301.P["PTRK_A0301_Pos1_To_Pos3"], ENO => #_w2);
   #TON.P1_Exit_P3.TON(IN := #_w2 AND #CIn.P1.Fermi.Rest AND NOT #Sts.P1.Fermi.Sens_Ing AND NOT #Sts.P1.Fermi.Sens_Out,
                       PT := T#800MS);
   IF #TON.P1_Exit_P3.Q THEN
       "PTrk".A0301.P["PTRK_A0301_Pos1_To_Pos3"] := "PTrk".A0301.P["PTRK_A0301_Pos1_Exit_To_Pos3"];
       "PTrk".A0301.P["PTRK_A0301_Pos1_Exit_To_Pos3"] := "PTrk".Empty;
   END_IF;
END_REGION

REGION Network 33: == Monitoraggio spazio di trasporto del movimento PTrk da Pos.1 a Pos.3 ==
   // Controllo la posizione salvata da Pos.1 exit + Distanza sensori Pos.1 / Pos.3 = Target da raggiungere
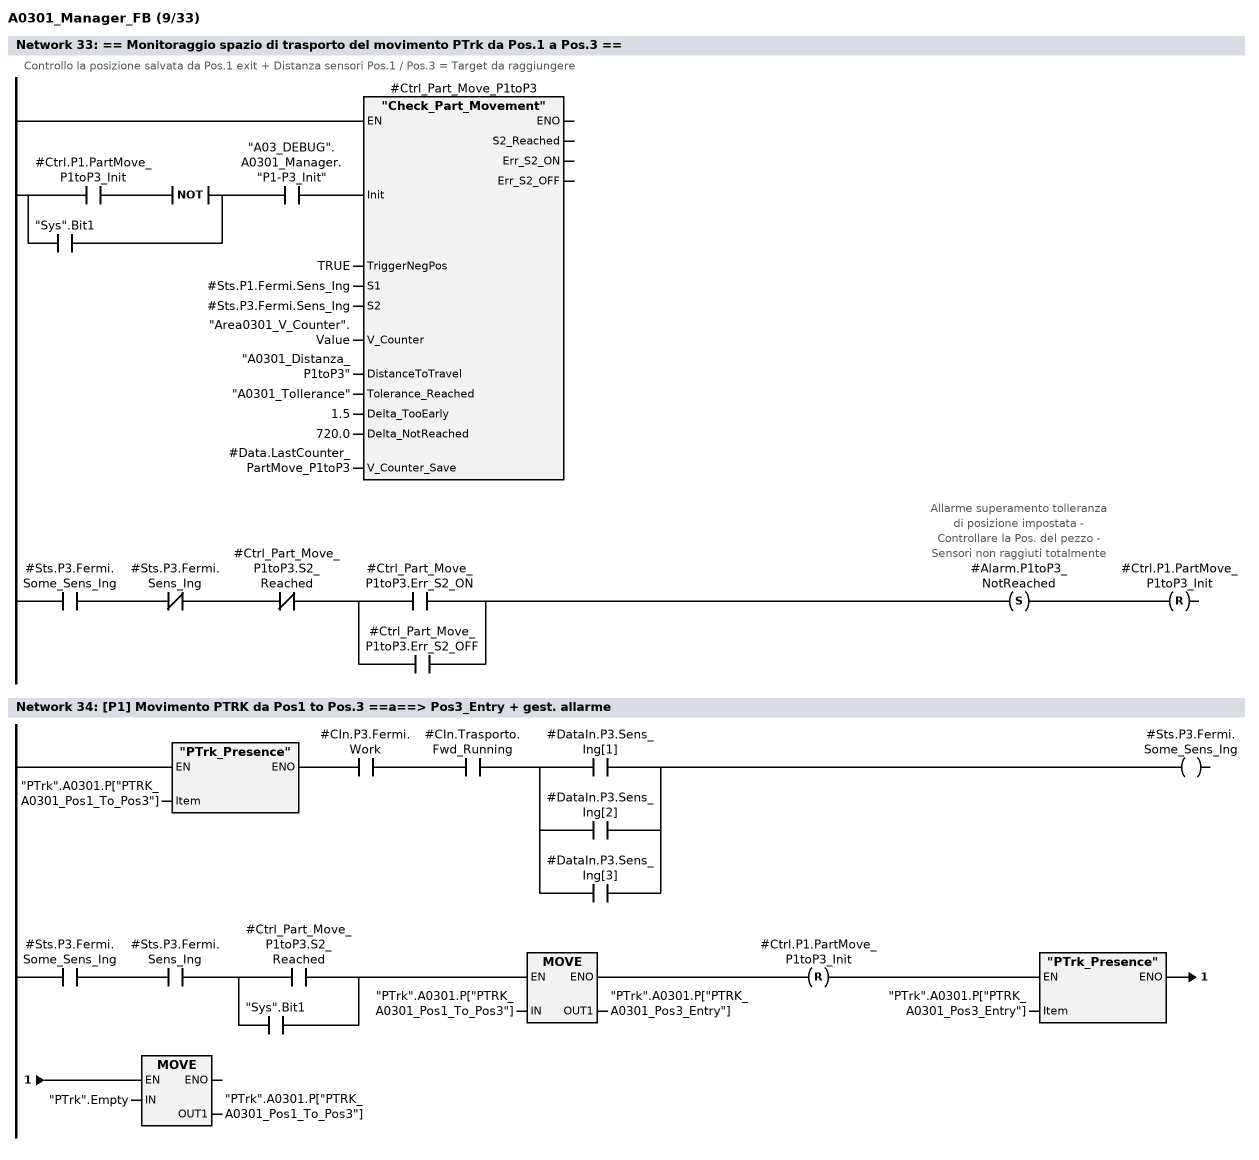
   RUNG wire#powerrail
      #Ctrl_Part_Move_P1toP3(Init := wire#w2, TriggerNegPos := TRUE, S1 := #Sts.P1.Fermi.Sens_Ing, S2 := #Sts.P3.Fermi.Sens_Ing, V_Counter := "Area0301_V_Counter".Value, DistanceToTravel := "A0301_Distanza_P1toP3", Tolerance_Reached := "A0301_Tollerance", Delta_TooEarly := 1.5, Delta_NotReached := 720.0, V_Counter_Save := #Data.LastCounter_PartMove_P1toP3, S2_Reached =>, Err_S2_ON =>, Err_S2_OFF =>)
   END_RUNG
   RUNG wire#powerrail
      Contact( #Ctrl.P1.PartMove_P1toP3_Init )
      Not()
      wire#w1
      Contact( "A03_DEBUG".A0301_Manager."P1-P3_Init" )
   END_RUNG wire#w2
   RUNG wire#powerrail
      Contact( "Sys".Bit1 )
   END_RUNG wire#w1
   RUNG wire#powerrail
      Contact( #Sts.P3.Fermi.Some_Sens_Ing )
      I_Contact( #Sts.P3.Fermi.Sens_Ing )
      I_Contact( #Ctrl_Part_Move_P1toP3.S2_Reached )
      wire#w3
      Contact( #Ctrl_Part_Move_P1toP3.Err_S2_ON )
      wire#w4
      S_Coil( #Alarm.P1toP3_NotReached )   // Allarme superamento tolleranza di posizione impostata - Controllare la Pos. del pezzo - Sensori non raggiuti totalmente
      R_Coil( #Ctrl.P1.PartMove_P1toP3_Init )
   END_RUNG
   RUNG wire#w3
      Contact( #Ctrl_Part_Move_P1toP3.Err_S2_OFF )
   END_RUNG wire#w4
   // the same network as SCL:
   #Ctrl_Part_Move_P1toP3(Init := (NOT #Ctrl.P1.PartMove_P1toP3_Init OR "Sys".Bit1) AND "A03_DEBUG".A0301_Manager."P1-P3_Init",   // "Check_Part_Movement"
                          TriggerNegPos := TRUE,
                          S1 := #Sts.P1.Fermi.Sens_Ing,
                          S2 := #Sts.P3.Fermi.Sens_Ing,
                          V_Counter := "Area0301_V_Counter".Value,
                          DistanceToTravel := "A0301_Distanza_P1toP3",
                          Tolerance_Reached := "A0301_Tollerance",
                          Delta_TooEarly := 1.5,
                          Delta_NotReached := 720.0,
                          V_Counter_Save := #Data.LastCounter_PartMove_P1toP3);
   IF #Sts.P3.Fermi.Some_Sens_Ing AND NOT #Sts.P3.Fermi.Sens_Ing AND NOT #Ctrl_Part_Move_P1toP3.S2_Reached AND (#Ctrl_Part_Move_P1toP3.Err_S2_ON OR #Ctrl_Part_Move_P1toP3.Err_S2_OFF) THEN
       #Alarm.P1toP3_NotReached := TRUE;   // Allarme superamento tolleranza di posizione impostata - Controllare la Pos. del pezzo - Sensori non raggiuti totalmente
       #Ctrl.P1.PartMove_P1toP3_Init := FALSE;
   END_IF;
END_REGION

REGION Network 34: [P1] Movimento PTRK da Pos1 to Pos.3 ==a==> Pos3_Entry + gest. allarme
   RUNG wire#powerrail
      "PTrk_Presence"(Item := "PTrk".A0301.P["PTRK_A0301_Pos1_To_Pos3"])
      Contact( #CIn.P3.Fermi.Work )
      Contact( #CIn.Trasporto.Fwd_Running )
      wire#w1
      Contact( #DataIn.P3.Sens_Ing[1] )
      wire#w2
      Coil( #Sts.P3.Fermi.Some_Sens_Ing )
   END_RUNG
   RUNG wire#w1
      Contact( #DataIn.P3.Sens_Ing[2] )
   END_RUNG wire#w2
   RUNG wire#w1
      Contact( #DataIn.P3.Sens_Ing[3] )
   END_RUNG wire#w2
   RUNG wire#powerrail
      Contact( #Sts.P3.Fermi.Some_Sens_Ing )
      Contact( #Sts.P3.Fermi.Sens_Ing )
      wire#w3
      Contact( #Ctrl_Part_Move_P1toP3.S2_Reached )
      wire#w4
      Move(in := "PTrk".A0301.P["PTRK_A0301_Pos1_To_Pos3"], out1 => "PTrk".A0301.P["PTRK_A0301_Pos3_Entry"])
      R_Coil( #Ctrl.P1.PartMove_P1toP3_Init )
      "PTrk_Presence"(Item := "PTrk".A0301.P["PTRK_A0301_Pos3_Entry"])
      Move(in := "PTrk".Empty, out1 => "PTrk".A0301.P["PTRK_A0301_Pos1_To_Pos3"])
   END_RUNG
   RUNG wire#w3
      Contact( "Sys".Bit1 )
   END_RUNG wire#w4
   // the same network as SCL:
   "PTrk_Presence"(Item := "PTrk".A0301.P["PTRK_A0301_Pos1_To_Pos3"], ENO => #_w1);
   #Sts.P3.Fermi.Some_Sens_Ing := #_w1 AND #CIn.P3.Fermi.Work AND #CIn.Trasporto.Fwd_Running AND (#DataIn.P3.Sens_Ing[1] OR #DataIn.P3.Sens_Ing[2] OR #DataIn.P3.Sens_Ing[3]);
   IF #Sts.P3.Fermi.Some_Sens_Ing AND #Sts.P3.Fermi.Sens_Ing AND (#Ctrl_Part_Move_P1toP3.S2_Reached OR "Sys".Bit1) THEN
       "PTrk".A0301.P["PTRK_A0301_Pos3_Entry"] := "PTrk".A0301.P["PTRK_A0301_Pos1_To_Pos3"];
       #Ctrl.P1.PartMove_P1toP3_Init := FALSE;
   END_IF;
   "PTrk_Presence"(EN := #Sts.P3.Fermi.Some_Sens_Ing AND #Sts.P3.Fermi.Sens_Ing AND (#Ctrl_Part_Move_P1toP3.S2_Reached OR "Sys".Bit1),
                   Item := "PTrk".A0301.P["PTRK_A0301_Pos3_Entry"],
                   ENO => #_w2);
   IF #_w2 THEN "PTrk".A0301.P["PTRK_A0301_Pos1_To_Pos3"] := "PTrk".Empty; END_IF;
END_REGION

REGION Network 35: [P1] Movimento PTRK da Pos1 exit Pos.2 ==a==> Pos1_To_Pos2
   // Salvo la quota nastro appena dopo la perdita del sensore presenza prodotto da Pos.1 e
   // azzero il PTrk su "Pos1ExitToP2" perchè passato avanti
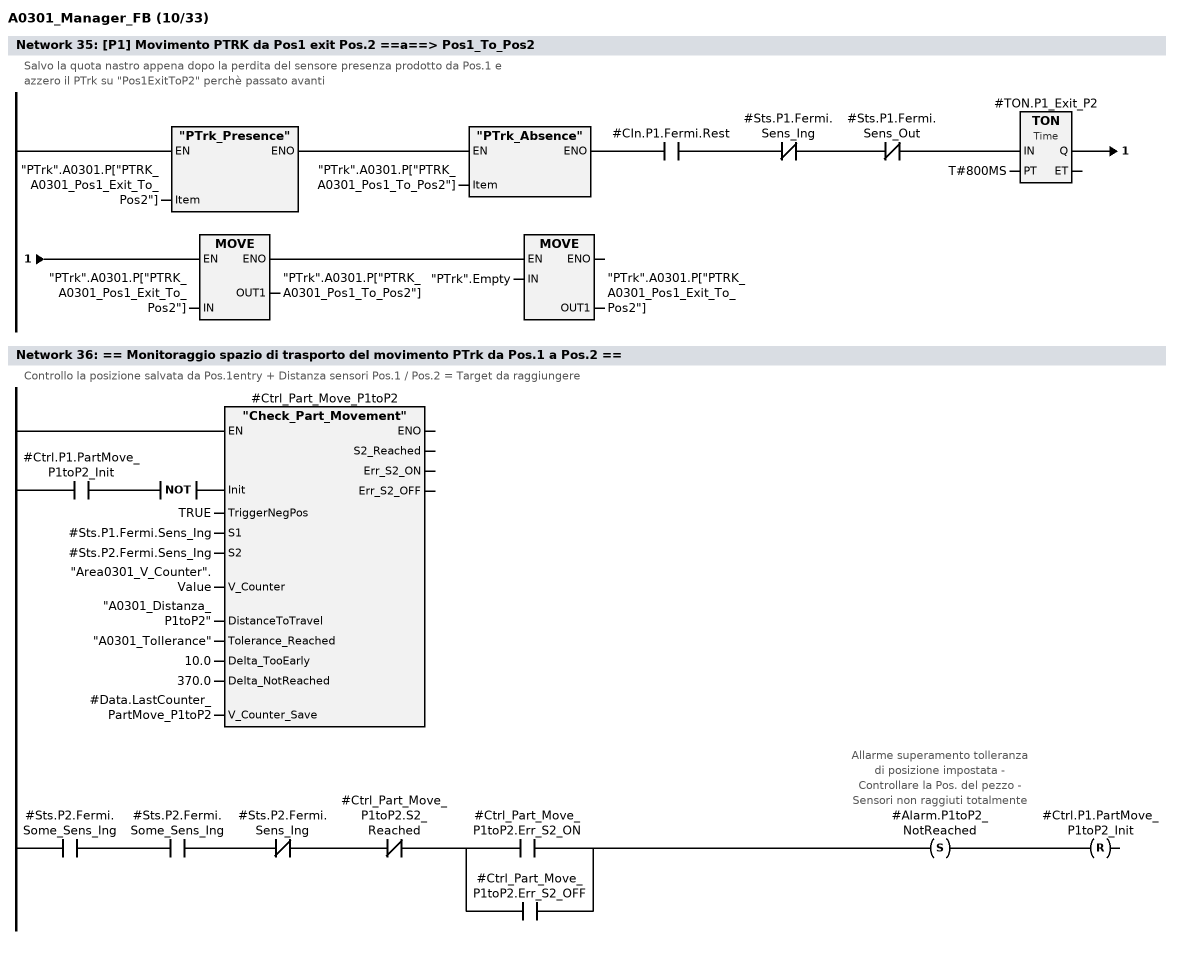
   RUNG wire#powerrail
      "PTrk_Presence"(Item := "PTrk".A0301.P["PTRK_A0301_Pos1_Exit_To_Pos2"])
      "PTrk_Absence"(Item := "PTrk".A0301.P["PTRK_A0301_Pos1_To_Pos2"])
      Contact( #CIn.P1.Fermi.Rest )
      I_Contact( #Sts.P1.Fermi.Sens_Ing )
      I_Contact( #Sts.P1.Fermi.Sens_Out )
      { S7_Templates := "time_type := Time" } #TON.P1_Exit_P2.TON(pt := T#800MS, et =>)
      Move(in := "PTrk".A0301.P["PTRK_A0301_Pos1_Exit_To_Pos2"], out1 => "PTrk".A0301.P["PTRK_A0301_Pos1_To_Pos2"])
      Move(in := "PTrk".Empty, out1 => "PTrk".A0301.P["PTRK_A0301_Pos1_Exit_To_Pos2"])
   END_RUNG
   // the same network as SCL:
   "PTrk_Presence"(Item := "PTrk".A0301.P["PTRK_A0301_Pos1_Exit_To_Pos2"], ENO => #_w1);
   "PTrk_Absence"(EN := #_w1, Item := "PTrk".A0301.P["PTRK_A0301_Pos1_To_Pos2"], ENO => #_w2);
   #TON.P1_Exit_P2.TON(IN := #_w2 AND #CIn.P1.Fermi.Rest AND NOT #Sts.P1.Fermi.Sens_Ing AND NOT #Sts.P1.Fermi.Sens_Out,
                       PT := T#800MS);
   IF #TON.P1_Exit_P2.Q THEN
       "PTrk".A0301.P["PTRK_A0301_Pos1_To_Pos2"] := "PTrk".A0301.P["PTRK_A0301_Pos1_Exit_To_Pos2"];
       "PTrk".A0301.P["PTRK_A0301_Pos1_Exit_To_Pos2"] := "PTrk".Empty;
   END_IF;
END_REGION

REGION Network 36: == Monitoraggio spazio di trasporto del movimento PTrk da Pos.1 a Pos.2 ==
   // Controllo la posizione salvata da Pos.1entry + Distanza sensori Pos.1 / Pos.2 = Target da raggiungere
   RUNG wire#powerrail
      #Ctrl_Part_Move_P1toP2(Init := wire#w1, TriggerNegPos := TRUE, S1 := #Sts.P1.Fermi.Sens_Ing, S2 := #Sts.P2.Fermi.Sens_Ing, V_Counter := "Area0301_V_Counter".Value, DistanceToTravel := "A0301_Distanza_P1toP2", Tolerance_Reached := "A0301_Tollerance", Delta_TooEarly := 10.0, Delta_NotReached := 370.0, V_Counter_Save := #Data.LastCounter_PartMove_P1toP2, S2_Reached =>, Err_S2_ON =>, Err_S2_OFF =>)
   END_RUNG
   RUNG wire#powerrail
      Contact( #Ctrl.P1.PartMove_P1toP2_Init )
      Not()
   END_RUNG wire#w1
   RUNG wire#powerrail
      Contact( #Sts.P2.Fermi.Some_Sens_Ing )
      Contact( #Sts.P2.Fermi.Some_Sens_Ing )
      I_Contact( #Sts.P2.Fermi.Sens_Ing )
      I_Contact( #Ctrl_Part_Move_P1toP2.S2_Reached )
      wire#w2
      Contact( #Ctrl_Part_Move_P1toP2.Err_S2_ON )
      wire#w3
      S_Coil( #Alarm.P1toP2_NotReached )   // Allarme superamento tolleranza di posizione impostata - Controllare la Pos. del pezzo - Sensori non raggiuti totalmente
      R_Coil( #Ctrl.P1.PartMove_P1toP2_Init )
   END_RUNG
   RUNG wire#w2
      Contact( #Ctrl_Part_Move_P1toP2.Err_S2_OFF )
   END_RUNG wire#w3
   // the same network as SCL:
   #Ctrl_Part_Move_P1toP2(Init := NOT #Ctrl.P1.PartMove_P1toP2_Init,   // "Check_Part_Movement"
                          TriggerNegPos := TRUE,
                          S1 := #Sts.P1.Fermi.Sens_Ing,
                          S2 := #Sts.P2.Fermi.Sens_Ing,
                          V_Counter := "Area0301_V_Counter".Value,
                          DistanceToTravel := "A0301_Distanza_P1toP2",
                          Tolerance_Reached := "A0301_Tollerance",
                          Delta_TooEarly := 10.0,
                          Delta_NotReached := 370.0,
                          V_Counter_Save := #Data.LastCounter_PartMove_P1toP2);
   IF #Sts.P2.Fermi.Some_Sens_Ing AND #Sts.P2.Fermi.Some_Sens_Ing AND NOT #Sts.P2.Fermi.Sens_Ing AND NOT #Ctrl_Part_Move_P1toP2.S2_Reached AND (#Ctrl_Part_Move_P1toP2.Err_S2_ON OR #Ctrl_Part_Move_P1toP2.Err_S2_OFF) THEN
       #Alarm.P1toP2_NotReached := TRUE;   // Allarme superamento tolleranza di posizione impostata - Controllare la Pos. del pezzo - Sensori non raggiuti totalmente
       #Ctrl.P1.PartMove_P1toP2_Init := FALSE;
   END_IF;
END_REGION

REGION Network 37: [P1] Movimento PTRK da Pos1 to Pos.2 ==a==> Pos2_Entry + gest. allarme
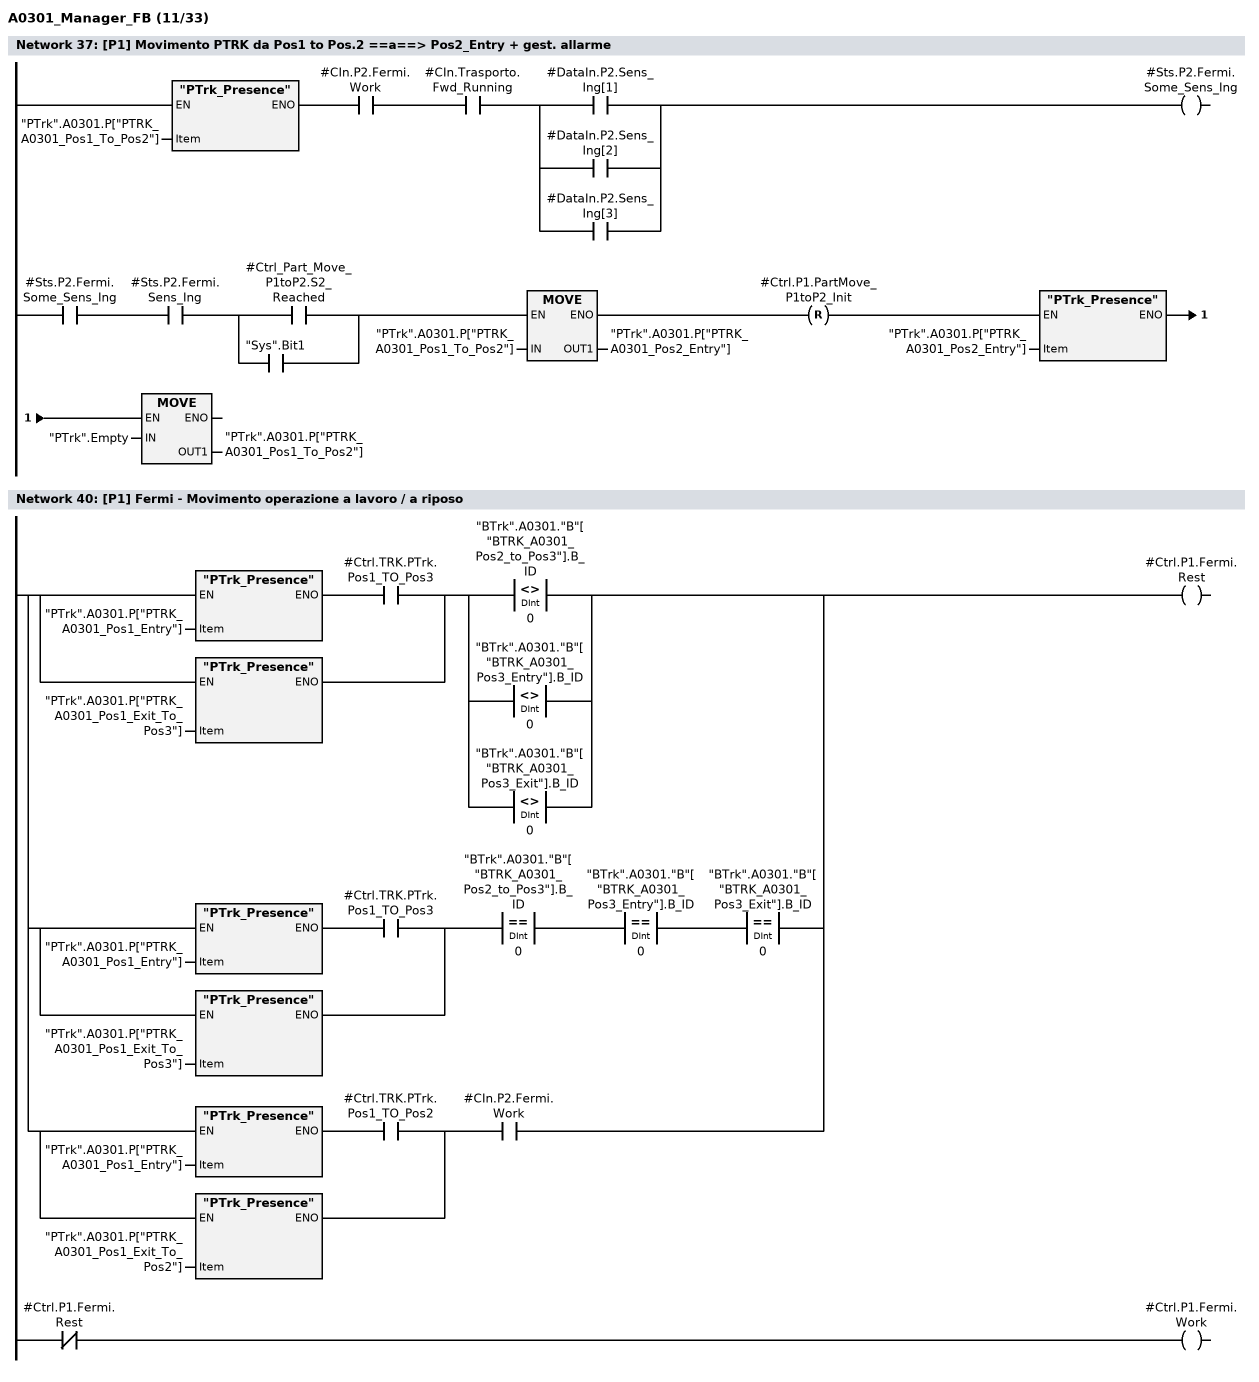
   RUNG wire#powerrail
      "PTrk_Presence"(Item := "PTrk".A0301.P["PTRK_A0301_Pos1_To_Pos2"])
      Contact( #CIn.P2.Fermi.Work )
      Contact( #CIn.Trasporto.Fwd_Running )
      wire#w1
      Contact( #DataIn.P2.Sens_Ing[1] )
      wire#w2
      Coil( #Sts.P2.Fermi.Some_Sens_Ing )
   END_RUNG
   RUNG wire#w1
      Contact( #DataIn.P2.Sens_Ing[2] )
   END_RUNG wire#w2
   RUNG wire#w1
      Contact( #DataIn.P2.Sens_Ing[3] )
   END_RUNG wire#w2
   RUNG wire#powerrail
      Contact( #Sts.P2.Fermi.Some_Sens_Ing )
      Contact( #Sts.P2.Fermi.Sens_Ing )
      wire#w3
      Contact( #Ctrl_Part_Move_P1toP2.S2_Reached )
      wire#w4
      Move(in := "PTrk".A0301.P["PTRK_A0301_Pos1_To_Pos2"], out1 => "PTrk".A0301.P["PTRK_A0301_Pos2_Entry"])
      R_Coil( #Ctrl.P1.PartMove_P1toP2_Init )
      "PTrk_Presence"(Item := "PTrk".A0301.P["PTRK_A0301_Pos2_Entry"])
      Move(in := "PTrk".Empty, out1 => "PTrk".A0301.P["PTRK_A0301_Pos1_To_Pos2"])
   END_RUNG
   RUNG wire#w3
      Contact( "Sys".Bit1 )
   END_RUNG wire#w4
   // the same network as SCL:
   "PTrk_Presence"(Item := "PTrk".A0301.P["PTRK_A0301_Pos1_To_Pos2"], ENO => #_w1);
   #Sts.P2.Fermi.Some_Sens_Ing := #_w1 AND #CIn.P2.Fermi.Work AND #CIn.Trasporto.Fwd_Running AND (#DataIn.P2.Sens_Ing[1] OR #DataIn.P2.Sens_Ing[2] OR #DataIn.P2.Sens_Ing[3]);
   IF #Sts.P2.Fermi.Some_Sens_Ing AND #Sts.P2.Fermi.Sens_Ing AND (#Ctrl_Part_Move_P1toP2.S2_Reached OR "Sys".Bit1) THEN
       "PTrk".A0301.P["PTRK_A0301_Pos2_Entry"] := "PTrk".A0301.P["PTRK_A0301_Pos1_To_Pos2"];
       #Ctrl.P1.PartMove_P1toP2_Init := FALSE;
   END_IF;
   "PTrk_Presence"(EN := #Sts.P2.Fermi.Some_Sens_Ing AND #Sts.P2.Fermi.Sens_Ing AND (#Ctrl_Part_Move_P1toP2.S2_Reached OR "Sys".Bit1),
                   Item := "PTrk".A0301.P["PTRK_A0301_Pos2_Entry"],
                   ENO => #_w2);
   IF #_w2 THEN "PTrk".A0301.P["PTRK_A0301_Pos1_To_Pos2"] := "PTrk".Empty; END_IF;
END_REGION

REGION Network 39: [P1] << GESTIONE MOVIMENTO FERMI / PAREGGIATORE >>
END_REGION

REGION Network 40: [P1] Fermi - Movimento operazione a lavoro / a riposo
   RUNG wire#powerrail
      "PTrk_Presence"(Item := "PTrk".A0301.P["PTRK_A0301_Pos1_Entry"])
      Contact( #Ctrl.TRK.PTrk.Pos1_TO_Pos3 )
      wire#w1
      { S7_Templates := "SrcType := DInt" } NE_Contact(in1 := "BTrk".A0301."B"["BTRK_A0301_Pos2_to_Pos3"].B_ID, in2 := 0)
      wire#w2
      Coil( #Ctrl.P1.Fermi.Rest )
   END_RUNG
   RUNG wire#powerrail
      "PTrk_Presence"(Item := "PTrk".A0301.P["PTRK_A0301_Pos1_Exit_To_Pos3"])
   END_RUNG wire#w1
   RUNG wire#w1
      { S7_Templates := "SrcType := DInt" } NE_Contact(in1 := "BTrk".A0301."B"["BTRK_A0301_Pos3_Entry"].B_ID, in2 := 0)
   END_RUNG wire#w2
   RUNG wire#w1
      { S7_Templates := "SrcType := DInt" } NE_Contact(in1 := "BTrk".A0301."B"["BTRK_A0301_Pos3_Exit"].B_ID, in2 := 0)
   END_RUNG wire#w2
   RUNG wire#powerrail
      "PTrk_Presence"(Item := "PTrk".A0301.P["PTRK_A0301_Pos1_Entry"])
      Contact( #Ctrl.TRK.PTrk.Pos1_TO_Pos3 )
      wire#w3
      { S7_Templates := "SrcType := DInt" } EQ_Contact(in1 := "BTrk".A0301."B"["BTRK_A0301_Pos2_to_Pos3"].B_ID, in2 := 0)
      { S7_Templates := "SrcType := DInt" } EQ_Contact(in1 := "BTrk".A0301."B"["BTRK_A0301_Pos3_Entry"].B_ID, in2 := 0)
      { S7_Templates := "SrcType := DInt" } EQ_Contact(in1 := "BTrk".A0301."B"["BTRK_A0301_Pos3_Exit"].B_ID, in2 := 0)
   END_RUNG wire#w2
   RUNG wire#powerrail
      "PTrk_Presence"(Item := "PTrk".A0301.P["PTRK_A0301_Pos1_Exit_To_Pos3"])
   END_RUNG wire#w3
   RUNG wire#powerrail
      "PTrk_Presence"(Item := "PTrk".A0301.P["PTRK_A0301_Pos1_Entry"])
      Contact( #Ctrl.TRK.PTrk.Pos1_TO_Pos2 )
      wire#w4
      Contact( #CIn.P2.Fermi.Work )
   END_RUNG wire#w2
   RUNG wire#powerrail
      "PTrk_Presence"(Item := "PTrk".A0301.P["PTRK_A0301_Pos1_Exit_To_Pos2"])
   END_RUNG wire#w4
   RUNG wire#powerrail
      I_Contact( #Ctrl.P1.Fermi.Rest )
      Coil( #Ctrl.P1.Fermi.Work )
   END_RUNG
   // the same network as SCL:
   "PTrk_Presence"(Item := "PTrk".A0301.P["PTRK_A0301_Pos1_Entry"], ENO => #_w1);
   "PTrk_Presence"(Item := "PTrk".A0301.P["PTRK_A0301_Pos1_Exit_To_Pos3"], ENO => #_w2);
   #_w4 := ((#_w1 AND #Ctrl.TRK.PTrk.Pos1_TO_Pos3) OR #_w2) AND ("BTrk".A0301."B"["BTRK_A0301_Pos2_to_Pos3"].B_ID <> 0);
   #_w5 := ((#_w1 AND #Ctrl.TRK.PTrk.Pos1_TO_Pos3) OR #_w2) AND ("BTrk".A0301."B"["BTRK_A0301_Pos3_Entry"].B_ID <> 0);
   #_w6 := ((#_w1 AND #Ctrl.TRK.PTrk.Pos1_TO_Pos3) OR #_w2) AND ("BTrk".A0301."B"["BTRK_A0301_Pos3_Exit"].B_ID <> 0);
   "PTrk_Presence"(Item := "PTrk".A0301.P["PTRK_A0301_Pos1_Entry"], ENO => #_w3);
   "PTrk_Presence"(Item := "PTrk".A0301.P["PTRK_A0301_Pos1_Exit_To_Pos3"], ENO => #_w7);
   #_w9 := ((#_w3 AND #Ctrl.TRK.PTrk.Pos1_TO_Pos3) OR #_w7) AND ("BTrk".A0301."B"["BTRK_A0301_Pos2_to_Pos3"].B_ID = 0) AND ("BTrk".A0301."B"["BTRK_A0301_Pos3_Entry"].B_ID = 0) AND ("BTrk".A0301."B"["BTRK_A0301_Pos3_Exit"].B_ID = 0);
   "PTrk_Presence"(Item := "PTrk".A0301.P["PTRK_A0301_Pos1_Entry"], ENO => #_w8);
   "PTrk_Presence"(Item := "PTrk".A0301.P["PTRK_A0301_Pos1_Exit_To_Pos2"], ENO => #_w10);
   #Ctrl.P1.Fermi.Rest := #_w4 OR #_w5 OR #_w6 OR #_w9 OR (((#_w8 AND #Ctrl.TRK.PTrk.Pos1_TO_Pos2) OR #_w10) AND #CIn.P2.Fermi.Work);
   #Ctrl.P1.Fermi.Work := NOT #Ctrl.P1.Fermi.Rest;
END_REGION

REGION Network 41: [P1] Pareggiatore - Movimento operazione a lavoro / a riposo
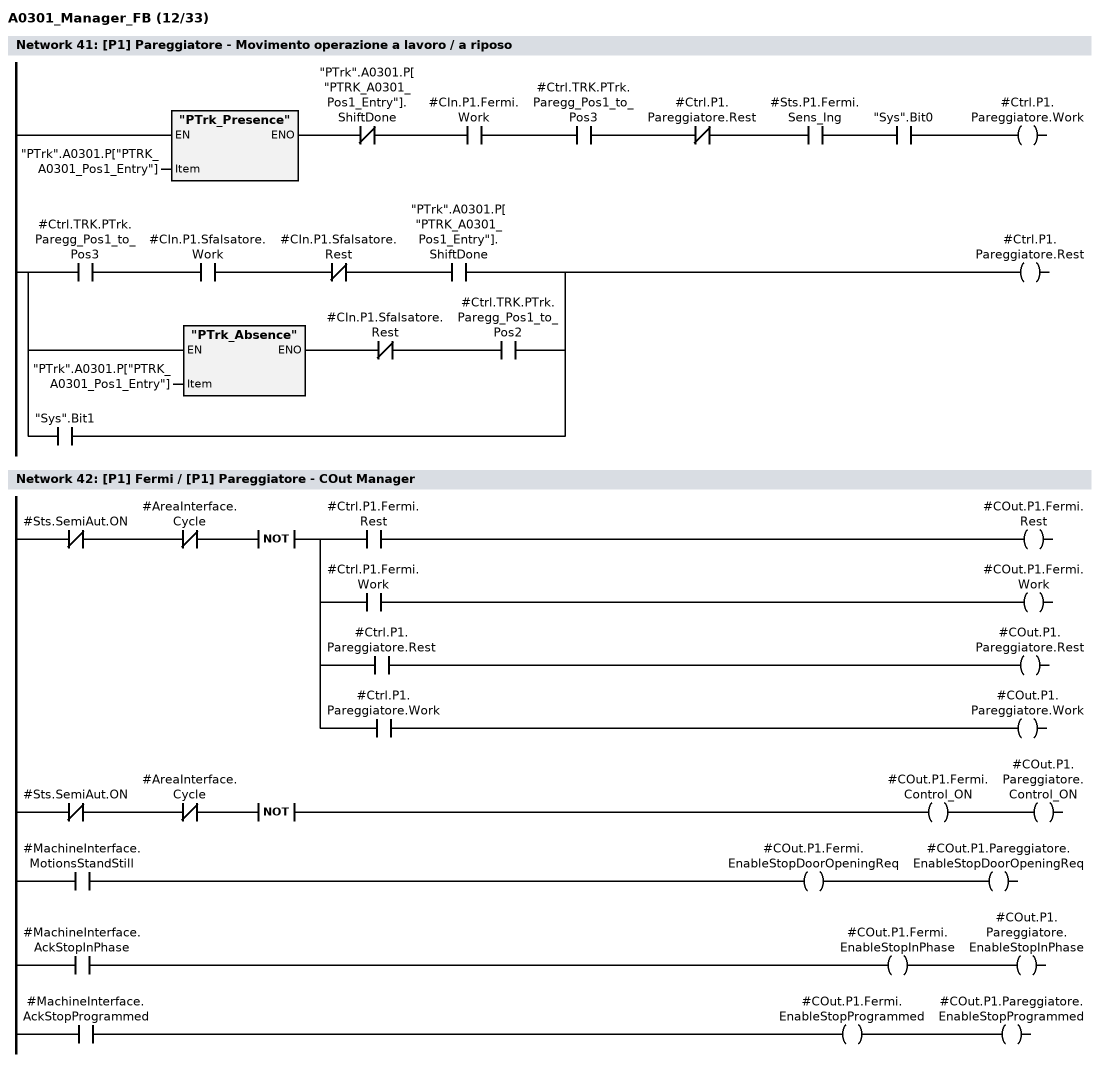
   RUNG wire#powerrail
      "PTrk_Presence"(Item := "PTrk".A0301.P["PTRK_A0301_Pos1_Entry"])
      I_Contact( "PTrk".A0301.P["PTRK_A0301_Pos1_Entry"].ShiftDone )
      Contact( #CIn.P1.Fermi.Work )
      Contact( #Ctrl.TRK.PTrk.Paregg_Pos1_to_Pos3 )
      I_Contact( #Ctrl.P1.Pareggiatore.Rest )
      Contact( #Sts.P1.Fermi.Sens_Ing )
      Contact( "Sys".Bit0 )
      Coil( #Ctrl.P1.Pareggiatore.Work )
   END_RUNG
   RUNG wire#powerrail
      Contact( #Ctrl.TRK.PTrk.Paregg_Pos1_to_Pos3 )
      Contact( #CIn.P1.Sfalsatore.Work )
      I_Contact( #CIn.P1.Sfalsatore.Rest )
      Contact( "PTrk".A0301.P["PTRK_A0301_Pos1_Entry"].ShiftDone )
      wire#w1
      Coil( #Ctrl.P1.Pareggiatore.Rest )
   END_RUNG
   RUNG wire#powerrail
      "PTrk_Absence"(Item := "PTrk".A0301.P["PTRK_A0301_Pos1_Entry"])
      I_Contact( #CIn.P1.Sfalsatore.Rest )
      Contact( #Ctrl.TRK.PTrk.Paregg_Pos1_to_Pos2 )
   END_RUNG wire#w1
   RUNG wire#powerrail
      Contact( "Sys".Bit1 )
   END_RUNG wire#w1
   // the same network as SCL:
   "PTrk_Presence"(Item := "PTrk".A0301.P["PTRK_A0301_Pos1_Entry"], ENO => #_w1);
   #Ctrl.P1.Pareggiatore.Work := #_w1 AND NOT "PTrk".A0301.P["PTRK_A0301_Pos1_Entry"].ShiftDone AND #CIn.P1.Fermi.Work AND #Ctrl.TRK.PTrk.Paregg_Pos1_to_Pos3 AND NOT #Ctrl.P1.Pareggiatore.Rest AND #Sts.P1.Fermi.Sens_Ing AND "Sys".Bit0;
   #_w3 := #Ctrl.TRK.PTrk.Paregg_Pos1_to_Pos3 AND #CIn.P1.Sfalsatore.Work AND NOT #CIn.P1.Sfalsatore.Rest AND "PTrk".A0301.P["PTRK_A0301_Pos1_Entry"].ShiftDone;
   "PTrk_Absence"(Item := "PTrk".A0301.P["PTRK_A0301_Pos1_Entry"], ENO => #_w2);
   #Ctrl.P1.Pareggiatore.Rest := #_w3 OR (#_w2 AND NOT #CIn.P1.Sfalsatore.Rest AND #Ctrl.TRK.PTrk.Paregg_Pos1_to_Pos2) OR "Sys".Bit1;
END_REGION

REGION Network 42: [P1] Fermi / [P1] Pareggiatore - COut Manager
   RUNG wire#powerrail
      I_Contact( #Sts.SemiAut.ON )
      I_Contact( #AreaInterface.Cycle )
      Not()
      wire#w1
      Contact( #Ctrl.P1.Fermi.Rest )
      Coil( #COut.P1.Fermi.Rest )
   END_RUNG
   RUNG wire#w1
      Contact( #Ctrl.P1.Fermi.Work )
      Coil( #COut.P1.Fermi.Work )
   END_RUNG
   RUNG wire#w1
      Contact( #Ctrl.P1.Pareggiatore.Rest )
      Coil( #COut.P1.Pareggiatore.Rest )
   END_RUNG
   RUNG wire#w1
      Contact( #Ctrl.P1.Pareggiatore.Work )
      Coil( #COut.P1.Pareggiatore.Work )
   END_RUNG
   RUNG wire#powerrail
      I_Contact( #Sts.SemiAut.ON )
      I_Contact( #AreaInterface.Cycle )
      Not()
      Coil( #COut.P1.Fermi.Control_ON )
      Coil( #COut.P1.Pareggiatore.Control_ON )
   END_RUNG
   RUNG wire#powerrail
      Contact( #MachineInterface.MotionsStandStill )
      Coil( #COut.P1.Fermi.EnableStopDoorOpeningReq )
      Coil( #COut.P1.Pareggiatore.EnableStopDoorOpeningReq )
   END_RUNG
   RUNG wire#powerrail
      Contact( #MachineInterface.AckStopInPhase )
      Coil( #COut.P1.Fermi.EnableStopInPhase )
      Coil( #COut.P1.Pareggiatore.EnableStopInPhase )
   END_RUNG
   RUNG wire#powerrail
      Contact( #MachineInterface.AckStopProgrammed )
      Coil( #COut.P1.Fermi.EnableStopProgrammed )
      Coil( #COut.P1.Pareggiatore.EnableStopProgrammed )
   END_RUNG
   // the same network as SCL:
   #_w1 := NOT (NOT #Sts.SemiAut.ON AND NOT #AreaInterface.Cycle);
   #COut.P1.Fermi.Rest := #_w1 AND #Ctrl.P1.Fermi.Rest;
   #COut.P1.Fermi.Work := #_w1 AND #Ctrl.P1.Fermi.Work;
   #COut.P1.Pareggiatore.Rest := #_w1 AND #Ctrl.P1.Pareggiatore.Rest;
   #COut.P1.Pareggiatore.Work := #_w1 AND #Ctrl.P1.Pareggiatore.Work;
   #COut.P1.Fermi.Control_ON := NOT (NOT #Sts.SemiAut.ON AND NOT #AreaInterface.Cycle);
   #COut.P1.Pareggiatore.Control_ON := #COut.P1.Fermi.Control_ON;
   #COut.P1.Fermi.EnableStopDoorOpeningReq := #MachineInterface.MotionsStandStill;
   #COut.P1.Pareggiatore.EnableStopDoorOpeningReq := #MachineInterface.MotionsStandStill;
   #COut.P1.Fermi.EnableStopInPhase := #MachineInterface.AckStopInPhase;
   #COut.P1.Pareggiatore.EnableStopInPhase := #MachineInterface.AckStopInPhase;
   #COut.P1.Fermi.EnableStopProgrammed := #MachineInterface.AckStopProgrammed;
   #COut.P1.Pareggiatore.EnableStopProgrammed := #MachineInterface.AckStopProgrammed;
END_REGION

REGION Network 44: <<<<<<<<<<< POSIZIONE 2 >>>>>>>>>>>
END_REGION

REGION Network 45: [P2] Movimento PTRK da Pos2 Entry ==a==> Pos2 Solleva
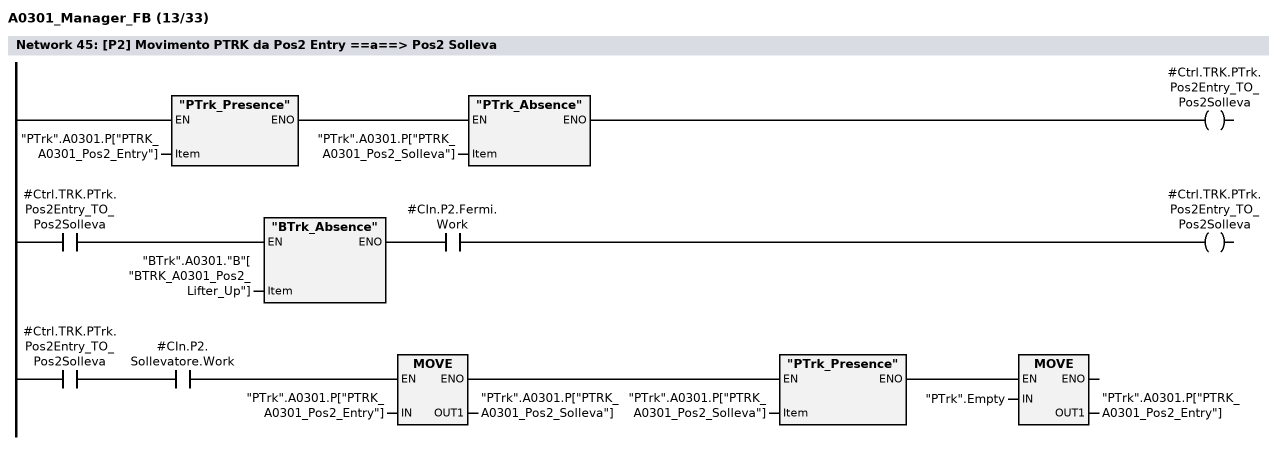
   RUNG wire#powerrail
      "PTrk_Presence"(Item := "PTrk".A0301.P["PTRK_A0301_Pos2_Entry"])
      "PTrk_Absence"(Item := "PTrk".A0301.P["PTRK_A0301_Pos2_Solleva"])
      Coil( #Ctrl.TRK.PTrk.Pos2Entry_TO_Pos2Solleva )
   END_RUNG
   RUNG wire#powerrail
      Contact( #Ctrl.TRK.PTrk.Pos2Entry_TO_Pos2Solleva )
      "BTrk_Absence"(Item := "BTrk".A0301."B"["BTRK_A0301_Pos2_Lifter_Up"])
      Contact( #CIn.P2.Fermi.Work )
      Coil( #Ctrl.TRK.PTrk.Pos2Entry_TO_Pos2Solleva )
   END_RUNG
   RUNG wire#powerrail
      Contact( #Ctrl.TRK.PTrk.Pos2Entry_TO_Pos2Solleva )
      Contact( #CIn.P2.Sollevatore.Work )
      Move(in := "PTrk".A0301.P["PTRK_A0301_Pos2_Entry"], out1 => "PTrk".A0301.P["PTRK_A0301_Pos2_Solleva"])
      "PTrk_Presence"(Item := "PTrk".A0301.P["PTRK_A0301_Pos2_Solleva"])
      Move(in := "PTrk".Empty, out1 => "PTrk".A0301.P["PTRK_A0301_Pos2_Entry"])
   END_RUNG
   // the same network as SCL:
   "PTrk_Presence"(Item := "PTrk".A0301.P["PTRK_A0301_Pos2_Entry"], ENO => #_w1);
   "PTrk_Absence"(EN := #_w1, Item := "PTrk".A0301.P["PTRK_A0301_Pos2_Solleva"], ENO => #_w2);
   #Ctrl.TRK.PTrk.Pos2Entry_TO_Pos2Solleva := #_w2;
   "BTrk_Absence"(EN := #Ctrl.TRK.PTrk.Pos2Entry_TO_Pos2Solleva,
                  Item := "BTrk".A0301."B"["BTRK_A0301_Pos2_Lifter_Up"],
                  ENO => #_w3);
   #Ctrl.TRK.PTrk.Pos2Entry_TO_Pos2Solleva := #_w3 AND #CIn.P2.Fermi.Work;
   IF #Ctrl.TRK.PTrk.Pos2Entry_TO_Pos2Solleva AND #CIn.P2.Sollevatore.Work THEN
       "PTrk".A0301.P["PTRK_A0301_Pos2_Solleva"] := "PTrk".A0301.P["PTRK_A0301_Pos2_Entry"];
   END_IF;
   "PTrk_Presence"(EN := #Ctrl.TRK.PTrk.Pos2Entry_TO_Pos2Solleva AND #CIn.P2.Sollevatore.Work,
                   Item := "PTrk".A0301.P["PTRK_A0301_Pos2_Solleva"],
                   ENO => #_w4);
   IF #_w4 THEN "PTrk".A0301.P["PTRK_A0301_Pos2_Entry"] := "PTrk".Empty; END_IF;
END_REGION

REGION Network 47: [P2] << GESTIONE MOVIMENTO FERMI >>
END_REGION

REGION Network 48: [P2] Fermi - Movimento operazione a lavoro / a riposo
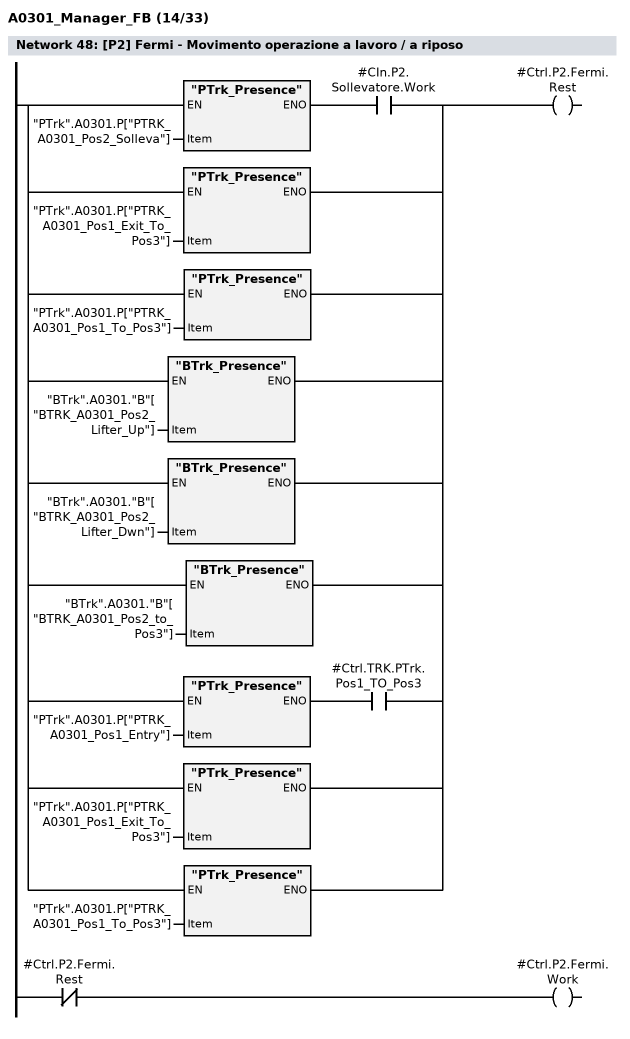
   RUNG wire#powerrail
      "PTrk_Presence"(Item := "PTrk".A0301.P["PTRK_A0301_Pos2_Solleva"])
      Contact( #CIn.P2.Sollevatore.Work )
      wire#w1
      Coil( #Ctrl.P2.Fermi.Rest )
   END_RUNG
   RUNG wire#powerrail
      "PTrk_Presence"(Item := "PTrk".A0301.P["PTRK_A0301_Pos1_Exit_To_Pos3"])
   END_RUNG wire#w1
   RUNG wire#powerrail
      "PTrk_Presence"(Item := "PTrk".A0301.P["PTRK_A0301_Pos1_To_Pos3"])
   END_RUNG wire#w1
   RUNG wire#powerrail
      "BTrk_Presence"(Item := "BTrk".A0301."B"["BTRK_A0301_Pos2_Lifter_Up"])
   END_RUNG wire#w1
   RUNG wire#powerrail
      "BTrk_Presence"(Item := "BTrk".A0301."B"["BTRK_A0301_Pos2_Lifter_Dwn"])
   END_RUNG wire#w1
   RUNG wire#powerrail
      "BTrk_Presence"(Item := "BTrk".A0301."B"["BTRK_A0301_Pos2_to_Pos3"])
   END_RUNG wire#w1
   RUNG wire#powerrail
      "PTrk_Presence"(Item := "PTrk".A0301.P["PTRK_A0301_Pos1_Entry"])
      Contact( #Ctrl.TRK.PTrk.Pos1_TO_Pos3 )
   END_RUNG wire#w1
   RUNG wire#powerrail
      "PTrk_Presence"(Item := "PTrk".A0301.P["PTRK_A0301_Pos1_Exit_To_Pos3"])
   END_RUNG wire#w1
   RUNG wire#powerrail
      "PTrk_Presence"(Item := "PTrk".A0301.P["PTRK_A0301_Pos1_To_Pos3"])
   END_RUNG wire#w1
   RUNG wire#powerrail
      I_Contact( #Ctrl.P2.Fermi.Rest )
      Coil( #Ctrl.P2.Fermi.Work )
   END_RUNG
   // the same network as SCL:
   "PTrk_Presence"(Item := "PTrk".A0301.P["PTRK_A0301_Pos2_Solleva"], ENO => #_w1);
   "PTrk_Presence"(Item := "PTrk".A0301.P["PTRK_A0301_Pos1_Exit_To_Pos3"], ENO => #_w2);
   "PTrk_Presence"(Item := "PTrk".A0301.P["PTRK_A0301_Pos1_To_Pos3"], ENO => #_w3);
   "BTrk_Presence"(Item := "BTrk".A0301."B"["BTRK_A0301_Pos2_Lifter_Up"], ENO => #_w4);
   "BTrk_Presence"(Item := "BTrk".A0301."B"["BTRK_A0301_Pos2_Lifter_Dwn"], ENO => #_w5);
   "BTrk_Presence"(Item := "BTrk".A0301."B"["BTRK_A0301_Pos2_to_Pos3"], ENO => #_w6);
   "PTrk_Presence"(Item := "PTrk".A0301.P["PTRK_A0301_Pos1_Entry"], ENO => #_w7);
   "PTrk_Presence"(Item := "PTrk".A0301.P["PTRK_A0301_Pos1_Exit_To_Pos3"], ENO => #_w8);
   "PTrk_Presence"(Item := "PTrk".A0301.P["PTRK_A0301_Pos1_To_Pos3"], ENO => #_w9);
   #Ctrl.P2.Fermi.Rest := (#_w1 AND #CIn.P2.Sollevatore.Work) OR #_w2 OR #_w3 OR #_w4 OR #_w5 OR #_w6 OR (#_w7 AND #Ctrl.TRK.PTrk.Pos1_TO_Pos3) OR #_w8 OR #_w9;
   #Ctrl.P2.Fermi.Work := NOT #Ctrl.P2.Fermi.Rest;
END_REGION

REGION Network 49: [P2] Fermi - COut Manager
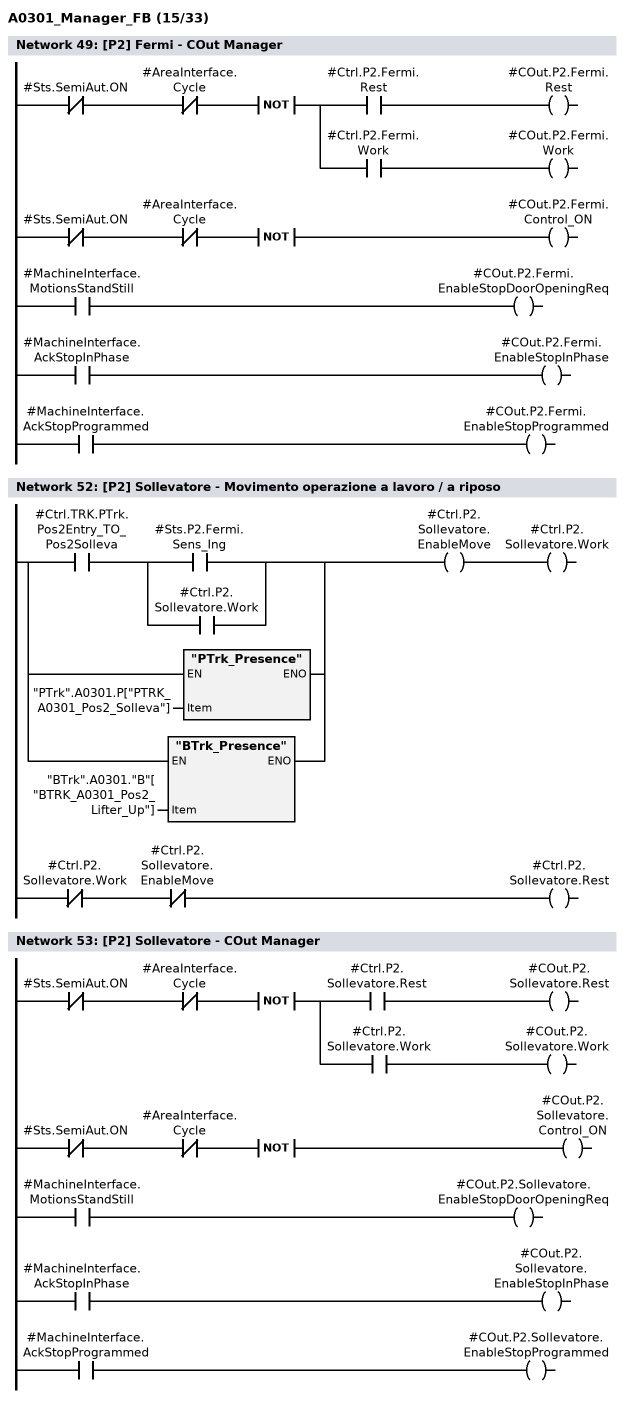
   RUNG wire#powerrail
      I_Contact( #Sts.SemiAut.ON )
      I_Contact( #AreaInterface.Cycle )
      Not()
      wire#w1
      Contact( #Ctrl.P2.Fermi.Rest )
      Coil( #COut.P2.Fermi.Rest )
   END_RUNG
   RUNG wire#w1
      Contact( #Ctrl.P2.Fermi.Work )
      Coil( #COut.P2.Fermi.Work )
   END_RUNG
   RUNG wire#powerrail
      I_Contact( #Sts.SemiAut.ON )
      I_Contact( #AreaInterface.Cycle )
      Not()
      Coil( #COut.P2.Fermi.Control_ON )
   END_RUNG
   RUNG wire#powerrail
      Contact( #MachineInterface.MotionsStandStill )
      Coil( #COut.P2.Fermi.EnableStopDoorOpeningReq )
   END_RUNG
   RUNG wire#powerrail
      Contact( #MachineInterface.AckStopInPhase )
      Coil( #COut.P2.Fermi.EnableStopInPhase )
   END_RUNG
   RUNG wire#powerrail
      Contact( #MachineInterface.AckStopProgrammed )
      Coil( #COut.P2.Fermi.EnableStopProgrammed )
   END_RUNG
   // the same network as SCL:
   #_w1 := NOT (NOT #Sts.SemiAut.ON AND NOT #AreaInterface.Cycle);
   #COut.P2.Fermi.Rest := #_w1 AND #Ctrl.P2.Fermi.Rest;
   #COut.P2.Fermi.Work := #_w1 AND #Ctrl.P2.Fermi.Work;
   #COut.P2.Fermi.Control_ON := NOT (NOT #Sts.SemiAut.ON AND NOT #AreaInterface.Cycle);
   #COut.P2.Fermi.EnableStopDoorOpeningReq := #MachineInterface.MotionsStandStill;
   #COut.P2.Fermi.EnableStopInPhase := #MachineInterface.AckStopInPhase;
   #COut.P2.Fermi.EnableStopProgrammed := #MachineInterface.AckStopProgrammed;
END_REGION

REGION Network 50: <+>
END_REGION

REGION Network 51: [P2] << GESTIONE MOVIMENTO SOLLEVATORE >>
END_REGION

REGION Network 52: [P2] Sollevatore - Movimento operazione a lavoro / a riposo
   RUNG wire#powerrail
      Contact( #Ctrl.TRK.PTrk.Pos2Entry_TO_Pos2Solleva )
      wire#w1
      Contact( #Sts.P2.Fermi.Sens_Ing )
      wire#w2
      Coil( #Ctrl.P2.Sollevatore.EnableMove )
      Coil( #Ctrl.P2.Sollevatore.Work )
   END_RUNG
   RUNG wire#w1
      Contact( #Ctrl.P2.Sollevatore.Work )
   END_RUNG wire#w2
   RUNG wire#powerrail
      "PTrk_Presence"(Item := "PTrk".A0301.P["PTRK_A0301_Pos2_Solleva"])
   END_RUNG wire#w2
   RUNG wire#powerrail
      "BTrk_Presence"(Item := "BTrk".A0301."B"["BTRK_A0301_Pos2_Lifter_Up"])
   END_RUNG wire#w2
   RUNG wire#powerrail
      I_Contact( #Ctrl.P2.Sollevatore.Work )
      I_Contact( #Ctrl.P2.Sollevatore.EnableMove )
      Coil( #Ctrl.P2.Sollevatore.Rest )
   END_RUNG
   // the same network as SCL:
   "PTrk_Presence"(Item := "PTrk".A0301.P["PTRK_A0301_Pos2_Solleva"], ENO => #_w1);
   "BTrk_Presence"(Item := "BTrk".A0301."B"["BTRK_A0301_Pos2_Lifter_Up"], ENO => #_w2);
   #Ctrl.P2.Sollevatore.EnableMove := (#Ctrl.TRK.PTrk.Pos2Entry_TO_Pos2Solleva AND (#Sts.P2.Fermi.Sens_Ing OR #Ctrl.P2.Sollevatore.Work)) OR #_w1 OR #_w2;
   #Ctrl.P2.Sollevatore.Work := #Ctrl.P2.Sollevatore.EnableMove;
   #Ctrl.P2.Sollevatore.Rest := NOT #Ctrl.P2.Sollevatore.Work AND NOT #Ctrl.P2.Sollevatore.EnableMove;
END_REGION

REGION Network 53: [P2] Sollevatore - COut Manager
   RUNG wire#powerrail
      I_Contact( #Sts.SemiAut.ON )
      I_Contact( #AreaInterface.Cycle )
      Not()
      wire#w1
      Contact( #Ctrl.P2.Sollevatore.Rest )
      Coil( #COut.P2.Sollevatore.Rest )
   END_RUNG
   RUNG wire#w1
      Contact( #Ctrl.P2.Sollevatore.Work )
      Coil( #COut.P2.Sollevatore.Work )
   END_RUNG
   RUNG wire#powerrail
      I_Contact( #Sts.SemiAut.ON )
      I_Contact( #AreaInterface.Cycle )
      Not()
      Coil( #COut.P2.Sollevatore.Control_ON )
   END_RUNG
   RUNG wire#powerrail
      Contact( #MachineInterface.MotionsStandStill )
      Coil( #COut.P2.Sollevatore.EnableStopDoorOpeningReq )
   END_RUNG
   RUNG wire#powerrail
      Contact( #MachineInterface.AckStopInPhase )
      Coil( #COut.P2.Sollevatore.EnableStopInPhase )
   END_RUNG
   RUNG wire#powerrail
      Contact( #MachineInterface.AckStopProgrammed )
      Coil( #COut.P2.Sollevatore.EnableStopProgrammed )
   END_RUNG
   // the same network as SCL:
   #_w1 := NOT (NOT #Sts.SemiAut.ON AND NOT #AreaInterface.Cycle);
   #COut.P2.Sollevatore.Rest := #_w1 AND #Ctrl.P2.Sollevatore.Rest;
   #COut.P2.Sollevatore.Work := #_w1 AND #Ctrl.P2.Sollevatore.Work;
   #COut.P2.Sollevatore.Control_ON := NOT (NOT #Sts.SemiAut.ON AND NOT #AreaInterface.Cycle);
   #COut.P2.Sollevatore.EnableStopDoorOpeningReq := #MachineInterface.MotionsStandStill;
   #COut.P2.Sollevatore.EnableStopInPhase := #MachineInterface.AckStopInPhase;
   #COut.P2.Sollevatore.EnableStopProgrammed := #MachineInterface.AckStopProgrammed;
END_REGION

REGION Network 55: <<<<<<<<<<< POSIZIONE 3 >>>>>>>>>>>
END_REGION

REGION Network 56: [P3] << GESTIONE MOVIMENTO FERMI >>
END_REGION

REGION Network 57: [P3] Fermi - Movimento operazione a lavoro / a riposo
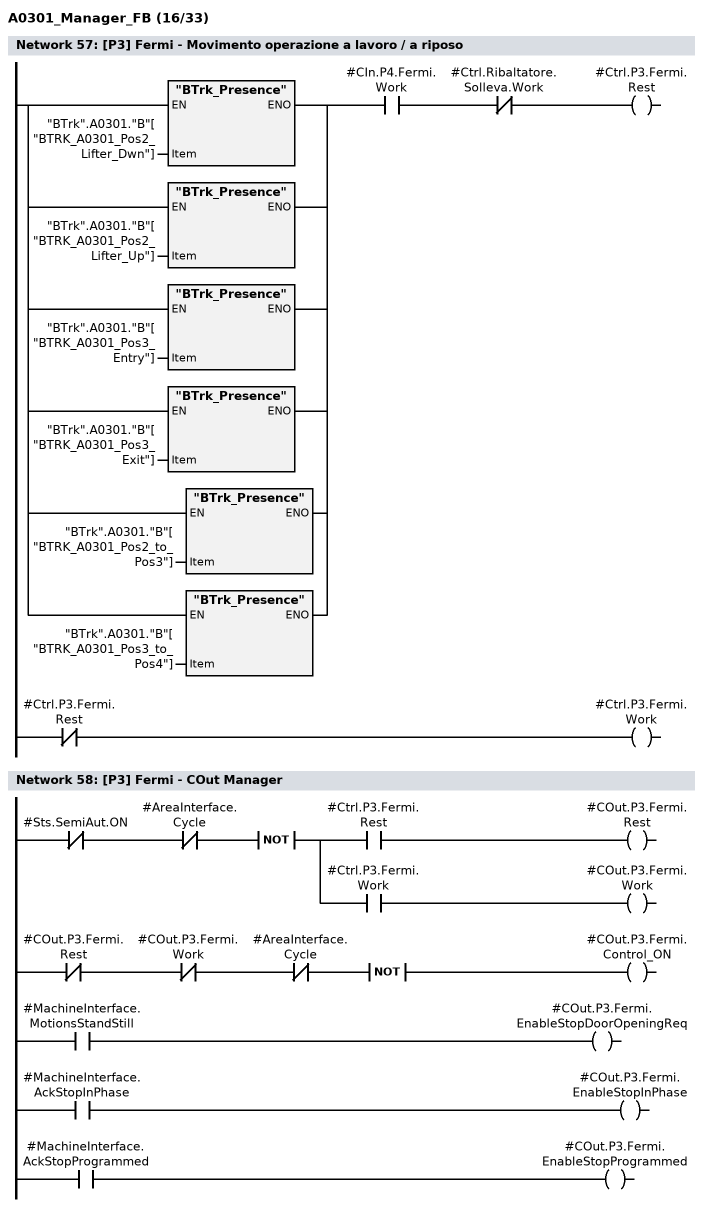
   RUNG wire#powerrail
      "BTrk_Presence"(Item := "BTrk".A0301."B"["BTRK_A0301_Pos2_Lifter_Dwn"])
      wire#w1
      Contact( #CIn.P4.Fermi.Work )
      I_Contact( #Ctrl.Ribaltatore.Solleva.Work )
      Coil( #Ctrl.P3.Fermi.Rest )
   END_RUNG
   RUNG wire#powerrail
      "BTrk_Presence"(Item := "BTrk".A0301."B"["BTRK_A0301_Pos2_Lifter_Up"])
   END_RUNG wire#w1
   RUNG wire#powerrail
      "BTrk_Presence"(Item := "BTrk".A0301."B"["BTRK_A0301_Pos3_Entry"])
   END_RUNG wire#w1
   RUNG wire#powerrail
      "BTrk_Presence"(Item := "BTrk".A0301."B"["BTRK_A0301_Pos3_Exit"])
   END_RUNG wire#w1
   RUNG wire#powerrail
      "BTrk_Presence"(Item := "BTrk".A0301."B"["BTRK_A0301_Pos2_to_Pos3"])
   END_RUNG wire#w1
   RUNG wire#powerrail
      "BTrk_Presence"(Item := "BTrk".A0301."B"["BTRK_A0301_Pos3_to_Pos4"])
   END_RUNG wire#w1
   RUNG wire#powerrail
      I_Contact( #Ctrl.P3.Fermi.Rest )
      Coil( #Ctrl.P3.Fermi.Work )
   END_RUNG
   // the same network as SCL:
   "BTrk_Presence"(Item := "BTrk".A0301."B"["BTRK_A0301_Pos2_Lifter_Dwn"], ENO => #_w1);
   "BTrk_Presence"(Item := "BTrk".A0301."B"["BTRK_A0301_Pos2_Lifter_Up"], ENO => #_w2);
   "BTrk_Presence"(Item := "BTrk".A0301."B"["BTRK_A0301_Pos3_Entry"], ENO => #_w3);
   "BTrk_Presence"(Item := "BTrk".A0301."B"["BTRK_A0301_Pos3_Exit"], ENO => #_w4);
   "BTrk_Presence"(Item := "BTrk".A0301."B"["BTRK_A0301_Pos2_to_Pos3"], ENO => #_w5);
   "BTrk_Presence"(Item := "BTrk".A0301."B"["BTRK_A0301_Pos3_to_Pos4"], ENO => #_w6);
   #Ctrl.P3.Fermi.Rest := (#_w1 OR #_w2 OR #_w3 OR #_w4 OR #_w5 OR #_w6) AND #CIn.P4.Fermi.Work AND NOT #Ctrl.Ribaltatore.Solleva.Work;
   #Ctrl.P3.Fermi.Work := NOT #Ctrl.P3.Fermi.Rest;
END_REGION

REGION Network 58: [P3] Fermi - COut Manager
   RUNG wire#powerrail
      I_Contact( #Sts.SemiAut.ON )
      I_Contact( #AreaInterface.Cycle )
      Not()
      wire#w1
      Contact( #Ctrl.P3.Fermi.Rest )
      Coil( #COut.P3.Fermi.Rest )
   END_RUNG
   RUNG wire#w1
      Contact( #Ctrl.P3.Fermi.Work )
      Coil( #COut.P3.Fermi.Work )
   END_RUNG
   RUNG wire#powerrail
      I_Contact( #COut.P3.Fermi.Rest )
      I_Contact( #COut.P3.Fermi.Work )
      I_Contact( #AreaInterface.Cycle )
      Not()
      Coil( #COut.P3.Fermi.Control_ON )
   END_RUNG
   RUNG wire#powerrail
      Contact( #MachineInterface.MotionsStandStill )
      Coil( #COut.P3.Fermi.EnableStopDoorOpeningReq )
   END_RUNG
   RUNG wire#powerrail
      Contact( #MachineInterface.AckStopInPhase )
      Coil( #COut.P3.Fermi.EnableStopInPhase )
   END_RUNG
   RUNG wire#powerrail
      Contact( #MachineInterface.AckStopProgrammed )
      Coil( #COut.P3.Fermi.EnableStopProgrammed )
   END_RUNG
   // the same network as SCL:
   #_w1 := NOT (NOT #Sts.SemiAut.ON AND NOT #AreaInterface.Cycle);
   #COut.P3.Fermi.Rest := #_w1 AND #Ctrl.P3.Fermi.Rest;
   #COut.P3.Fermi.Work := #_w1 AND #Ctrl.P3.Fermi.Work;
   #COut.P3.Fermi.Control_ON := NOT (NOT #COut.P3.Fermi.Rest AND NOT #COut.P3.Fermi.Work AND NOT #AreaInterface.Cycle);
   #COut.P3.Fermi.EnableStopDoorOpeningReq := #MachineInterface.MotionsStandStill;
   #COut.P3.Fermi.EnableStopInPhase := #MachineInterface.AckStopInPhase;
   #COut.P3.Fermi.EnableStopProgrammed := #MachineInterface.AckStopProgrammed;
END_REGION

REGION Network 60: <<<<<<<<<<< RIBALTATORE >>>>>>>>>>>
END_REGION

REGION Network 61: P [Solleva] Movimento solleva ribaltatore
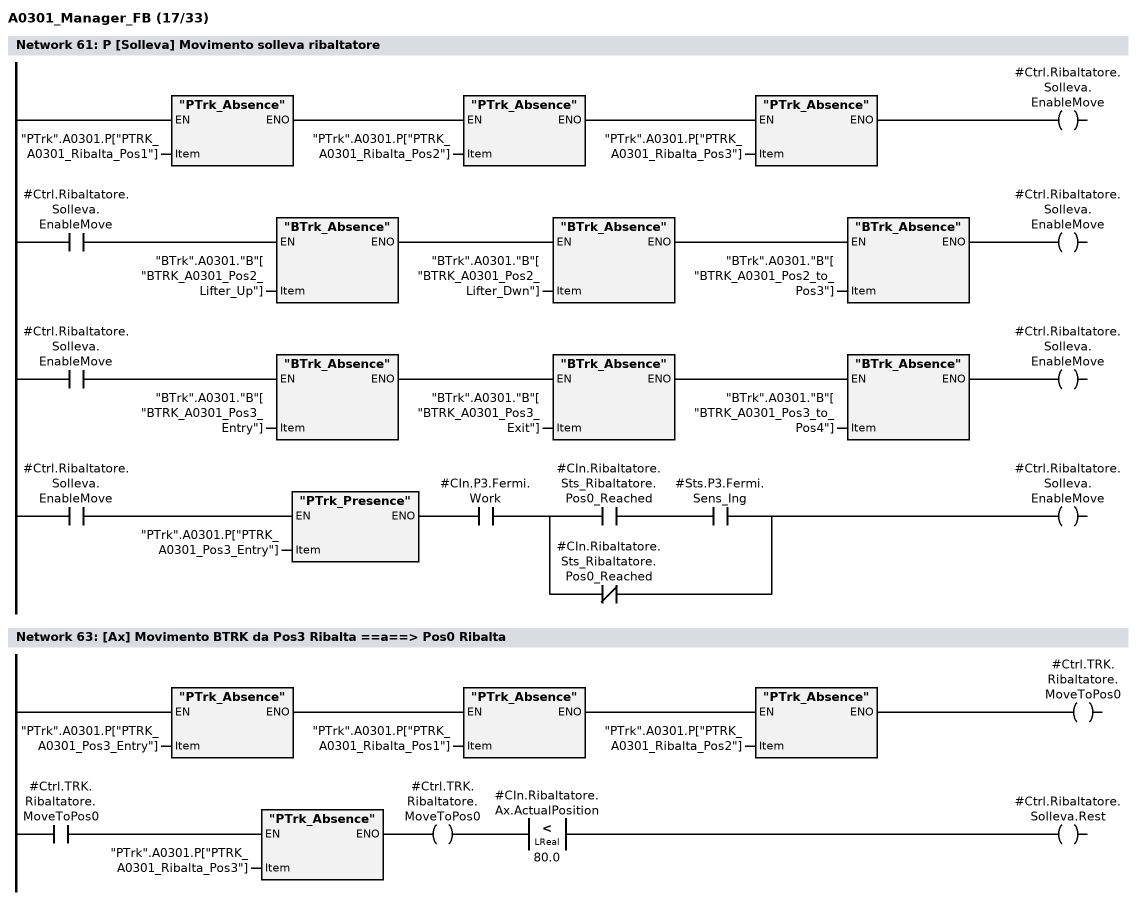
   RUNG wire#powerrail
      "PTrk_Absence"(Item := "PTrk".A0301.P["PTRK_A0301_Ribalta_Pos1"])
      "PTrk_Absence"(Item := "PTrk".A0301.P["PTRK_A0301_Ribalta_Pos2"])
      "PTrk_Absence"(Item := "PTrk".A0301.P["PTRK_A0301_Ribalta_Pos3"])
      Coil( #Ctrl.Ribaltatore.Solleva.EnableMove )
   END_RUNG
   RUNG wire#powerrail
      Contact( #Ctrl.Ribaltatore.Solleva.EnableMove )
      "BTrk_Absence"(Item := "BTrk".A0301."B"["BTRK_A0301_Pos2_Lifter_Up"])
      "BTrk_Absence"(Item := "BTrk".A0301."B"["BTRK_A0301_Pos2_Lifter_Dwn"])
      "BTrk_Absence"(Item := "BTrk".A0301."B"["BTRK_A0301_Pos2_to_Pos3"])
      Coil( #Ctrl.Ribaltatore.Solleva.EnableMove )
   END_RUNG
   RUNG wire#powerrail
      Contact( #Ctrl.Ribaltatore.Solleva.EnableMove )
      "BTrk_Absence"(Item := "BTrk".A0301."B"["BTRK_A0301_Pos3_Entry"])
      "BTrk_Absence"(Item := "BTrk".A0301."B"["BTRK_A0301_Pos3_Exit"])
      "BTrk_Absence"(Item := "BTrk".A0301."B"["BTRK_A0301_Pos3_to_Pos4"])
      Coil( #Ctrl.Ribaltatore.Solleva.EnableMove )
   END_RUNG
   RUNG wire#powerrail
      Contact( #Ctrl.Ribaltatore.Solleva.EnableMove )
      "PTrk_Presence"(Item := "PTrk".A0301.P["PTRK_A0301_Pos3_Entry"])
      Contact( #CIn.P3.Fermi.Work )
      wire#w1
      Contact( #CIn.Ribaltatore.Sts_Ribaltatore.Pos0_Reached )
      Contact( #Sts.P3.Fermi.Sens_Ing )
      wire#w2
      Coil( #Ctrl.Ribaltatore.Solleva.EnableMove )
   END_RUNG
   RUNG wire#w1
      I_Contact( #CIn.Ribaltatore.Sts_Ribaltatore.Pos0_Reached )
   END_RUNG wire#w2
   // the same network as SCL:
   "PTrk_Absence"(Item := "PTrk".A0301.P["PTRK_A0301_Ribalta_Pos1"], ENO => #_w1);
   "PTrk_Absence"(EN := #_w1, Item := "PTrk".A0301.P["PTRK_A0301_Ribalta_Pos2"], ENO => #_w2);
   "PTrk_Absence"(EN := #_w2, Item := "PTrk".A0301.P["PTRK_A0301_Ribalta_Pos3"], ENO => #_w3);
   #Ctrl.Ribaltatore.Solleva.EnableMove := #_w3;
   "BTrk_Absence"(EN := #Ctrl.Ribaltatore.Solleva.EnableMove,
                  Item := "BTrk".A0301."B"["BTRK_A0301_Pos2_Lifter_Up"],
                  ENO => #_w4);
   "BTrk_Absence"(EN := #_w4, Item := "BTrk".A0301."B"["BTRK_A0301_Pos2_Lifter_Dwn"], ENO => #_w5);
   "BTrk_Absence"(EN := #_w5, Item := "BTrk".A0301."B"["BTRK_A0301_Pos2_to_Pos3"], ENO => #_w6);
   #Ctrl.Ribaltatore.Solleva.EnableMove := #_w6;
   "BTrk_Absence"(EN := #Ctrl.Ribaltatore.Solleva.EnableMove,
                  Item := "BTrk".A0301."B"["BTRK_A0301_Pos3_Entry"],
                  ENO => #_w7);
   "BTrk_Absence"(EN := #_w7, Item := "BTrk".A0301."B"["BTRK_A0301_Pos3_Exit"], ENO => #_w8);
   "BTrk_Absence"(EN := #_w8, Item := "BTrk".A0301."B"["BTRK_A0301_Pos3_to_Pos4"], ENO => #_w9);
   #Ctrl.Ribaltatore.Solleva.EnableMove := #_w9;
   "PTrk_Presence"(EN := #Ctrl.Ribaltatore.Solleva.EnableMove,
                   Item := "PTrk".A0301.P["PTRK_A0301_Pos3_Entry"],
                   ENO => #_w10);
   #Ctrl.Ribaltatore.Solleva.EnableMove := #_w10 AND #CIn.P3.Fermi.Work AND ((#CIn.Ribaltatore.Sts_Ribaltatore.Pos0_Reached AND #Sts.P3.Fermi.Sens_Ing) OR NOT #CIn.Ribaltatore.Sts_Ribaltatore.Pos0_Reached);
END_REGION

REGION Network 62: <+>
END_REGION

REGION Network 63: [Ax] Movimento BTRK da Pos3 Ribalta ==a==> Pos0 Ribalta
   RUNG wire#powerrail
      "PTrk_Absence"(Item := "PTrk".A0301.P["PTRK_A0301_Pos3_Entry"])
      "PTrk_Absence"(Item := "PTrk".A0301.P["PTRK_A0301_Ribalta_Pos1"])
      "PTrk_Absence"(Item := "PTrk".A0301.P["PTRK_A0301_Ribalta_Pos2"])
      Coil( #Ctrl.TRK.Ribaltatore.MoveToPos0 )
   END_RUNG
   RUNG wire#powerrail
      Contact( #Ctrl.TRK.Ribaltatore.MoveToPos0 )
      "PTrk_Absence"(Item := "PTrk".A0301.P["PTRK_A0301_Ribalta_Pos3"])
      Coil( #Ctrl.TRK.Ribaltatore.MoveToPos0 )
      { S7_Templates := "SrcType := LReal" } LT_Contact(in1 := #CIn.Ribaltatore.Ax.ActualPosition, in2 := 80.0)
      Coil( #Ctrl.Ribaltatore.Solleva.Rest )
   END_RUNG
   // the same network as SCL:
   "PTrk_Absence"(Item := "PTrk".A0301.P["PTRK_A0301_Pos3_Entry"], ENO => #_w1);
   "PTrk_Absence"(EN := #_w1, Item := "PTrk".A0301.P["PTRK_A0301_Ribalta_Pos1"], ENO => #_w2);
   "PTrk_Absence"(EN := #_w2, Item := "PTrk".A0301.P["PTRK_A0301_Ribalta_Pos2"], ENO => #_w3);
   #Ctrl.TRK.Ribaltatore.MoveToPos0 := #_w3;
   "PTrk_Absence"(EN := #Ctrl.TRK.Ribaltatore.MoveToPos0,
                  Item := "PTrk".A0301.P["PTRK_A0301_Ribalta_Pos3"],
                  ENO => #_w4);
   #Ctrl.TRK.Ribaltatore.MoveToPos0 := #_w4;
   #Ctrl.Ribaltatore.Solleva.Rest := #_w4 AND (#CIn.Ribaltatore.Ax.ActualPosition < 80.0);
END_REGION

REGION Network 64: [Ax] Movimento PTRK da Pos3 Entry ==a==> Pos1 Ribalta
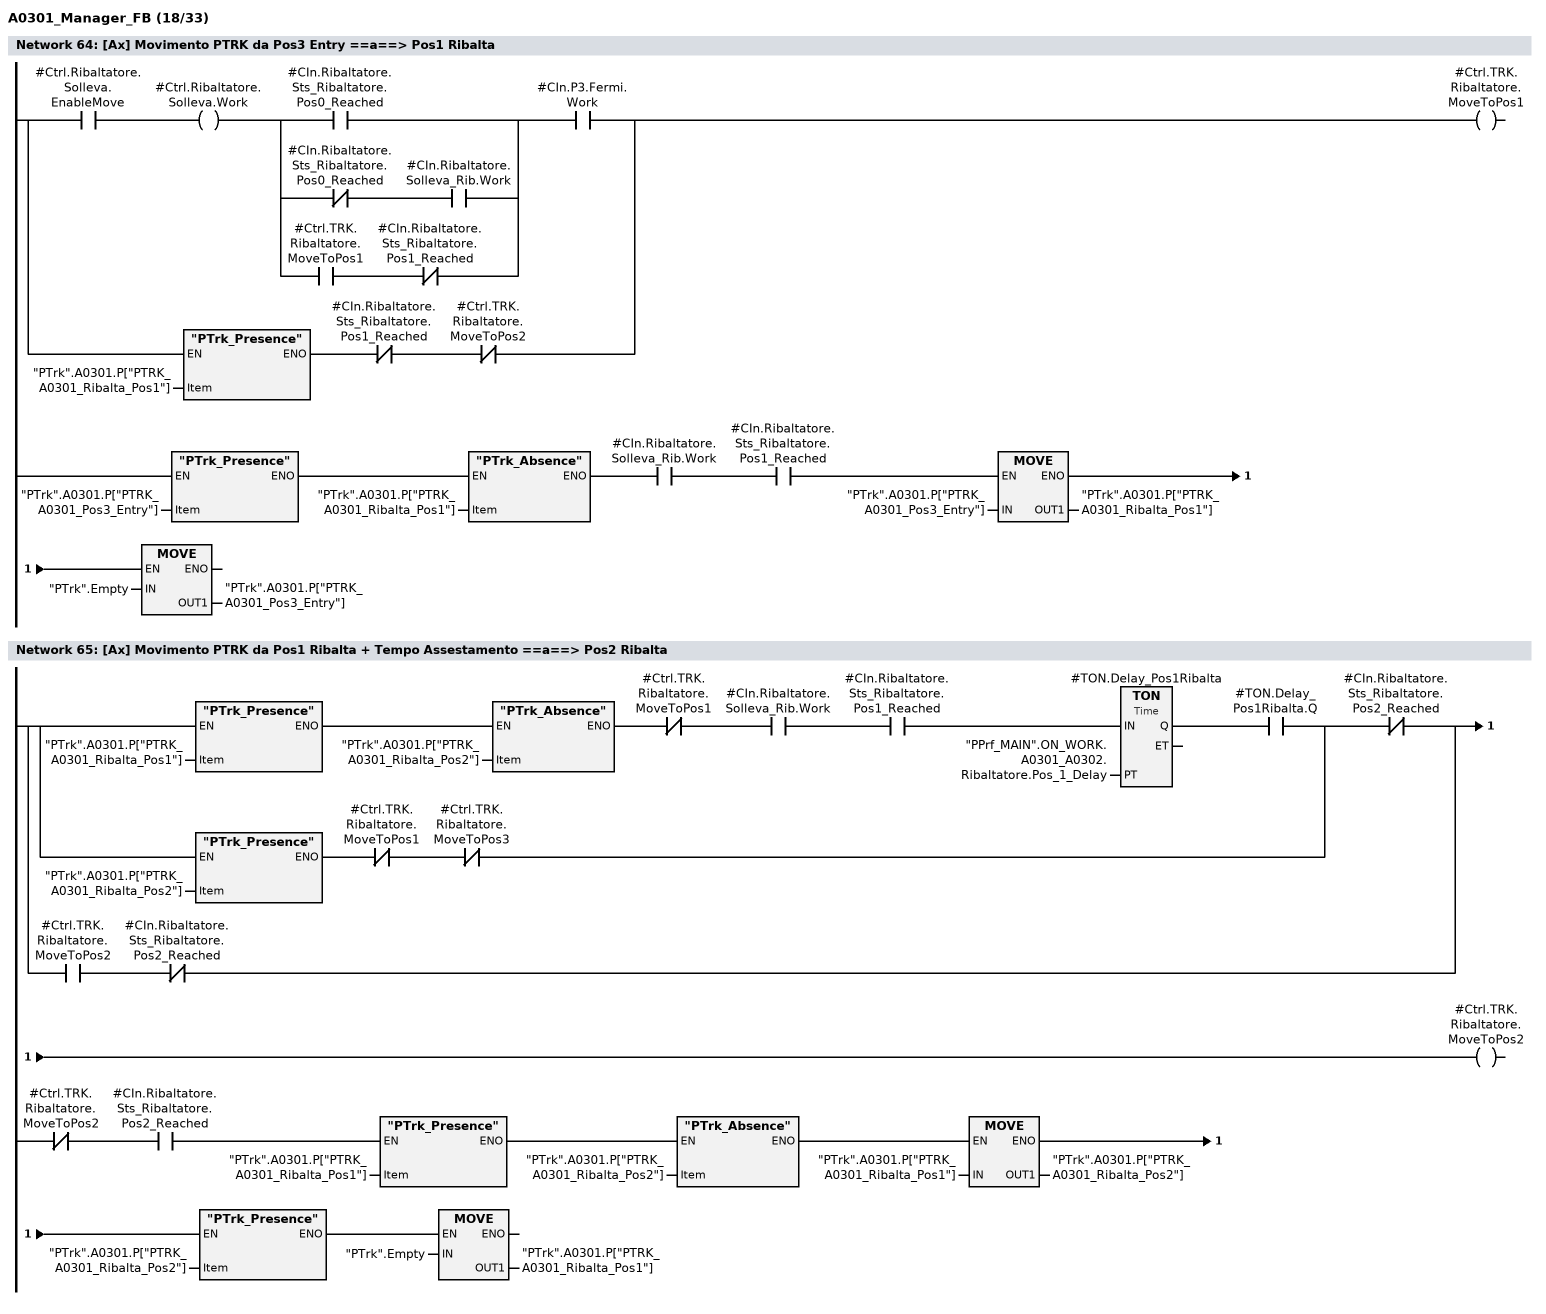
   RUNG wire#powerrail
      Contact( #Ctrl.Ribaltatore.Solleva.EnableMove )
      Coil( #Ctrl.Ribaltatore.Solleva.Work )
      wire#w1
      Contact( #CIn.Ribaltatore.Sts_Ribaltatore.Pos0_Reached )
      wire#w2
      Contact( #CIn.P3.Fermi.Work )
      wire#w3
      Coil( #Ctrl.TRK.Ribaltatore.MoveToPos1 )
   END_RUNG
   RUNG wire#w1
      I_Contact( #CIn.Ribaltatore.Sts_Ribaltatore.Pos0_Reached )
      Contact( #CIn.Ribaltatore.Solleva_Rib.Work )
   END_RUNG wire#w2
   RUNG wire#w1
      Contact( #Ctrl.TRK.Ribaltatore.MoveToPos1 )
      I_Contact( #CIn.Ribaltatore.Sts_Ribaltatore.Pos1_Reached )
   END_RUNG wire#w2
   RUNG wire#powerrail
      "PTrk_Presence"(Item := "PTrk".A0301.P["PTRK_A0301_Ribalta_Pos1"])
      I_Contact( #CIn.Ribaltatore.Sts_Ribaltatore.Pos1_Reached )
      I_Contact( #Ctrl.TRK.Ribaltatore.MoveToPos2 )
   END_RUNG wire#w3
   RUNG wire#powerrail
      "PTrk_Presence"(Item := "PTrk".A0301.P["PTRK_A0301_Pos3_Entry"])
      "PTrk_Absence"(Item := "PTrk".A0301.P["PTRK_A0301_Ribalta_Pos1"])
      Contact( #CIn.Ribaltatore.Solleva_Rib.Work )
      Contact( #CIn.Ribaltatore.Sts_Ribaltatore.Pos1_Reached )
      Move(in := "PTrk".A0301.P["PTRK_A0301_Pos3_Entry"], out1 => "PTrk".A0301.P["PTRK_A0301_Ribalta_Pos1"])
      Move(in := "PTrk".Empty, out1 => "PTrk".A0301.P["PTRK_A0301_Pos3_Entry"])
   END_RUNG
   // the same network as SCL:
   #Ctrl.Ribaltatore.Solleva.Work := #Ctrl.Ribaltatore.Solleva.EnableMove;
   "PTrk_Presence"(Item := "PTrk".A0301.P["PTRK_A0301_Ribalta_Pos1"], ENO => #_w1);
   #Ctrl.TRK.Ribaltatore.MoveToPos1 := (#Ctrl.Ribaltatore.Solleva.EnableMove AND (#CIn.Ribaltatore.Sts_Ribaltatore.Pos0_Reached OR (NOT #CIn.Ribaltatore.Sts_Ribaltatore.Pos0_Reached AND #CIn.Ribaltatore.Solleva_Rib.Work) OR (#Ctrl.TRK.Ribaltatore.MoveToPos1 AND NOT #CIn.Ribaltatore.Sts_Ribaltatore.Pos1_Reached)) AND #CIn.P3.Fermi.Work) OR (#_w1 AND NOT #CIn.Ribaltatore.Sts_Ribaltatore.Pos1_Reached AND NOT #Ctrl.TRK.Ribaltatore.MoveToPos2);
   "PTrk_Presence"(Item := "PTrk".A0301.P["PTRK_A0301_Pos3_Entry"], ENO => #_w2);
   "PTrk_Absence"(EN := #_w2, Item := "PTrk".A0301.P["PTRK_A0301_Ribalta_Pos1"], ENO => #_w3);
   IF #_w3 AND #CIn.Ribaltatore.Solleva_Rib.Work AND #CIn.Ribaltatore.Sts_Ribaltatore.Pos1_Reached THEN
       "PTrk".A0301.P["PTRK_A0301_Ribalta_Pos1"] := "PTrk".A0301.P["PTRK_A0301_Pos3_Entry"];
       "PTrk".A0301.P["PTRK_A0301_Pos3_Entry"] := "PTrk".Empty;
   END_IF;
END_REGION

